   ELSE
       "DB198_eventos_generados_routing_JDT1".evento[#posicion] :=CONCAT(IN1 := '{WARN[RUET]', IN2 := #codigo_string, IN3 := '[ERRO]BBDD[MOTI]FULL',  IN4 := "DB921_DATOS_FECHA_HORA".TIME_STAMP, IN5 := '}');

   END_IF;
END_REGION
END_FUNCTION

FUNCTION "FC887_Obtener_StringDelAtributo_Ulint" : Void   // FC887, LAD
TITLE = "ObtenerStringAtributo" - Convertir a String un Doble Entero
{ S7_Optimized_Access := 'FALSE' }
AUTHOR : TRACKING
NAME : 20130301
VERSION : 3.0
// stored: AutoNumber false, SetENOAutomatically false
   VAR_INPUT
      DB_String : UInt;   // DB donde esta la String
      OffsetIni : UInt;   // Numero de byte de la String donde empieza
      Valor : ULInt;   // Valor a Convertir
   END_VAR
   VAR_OUTPUT
      OffsetFin : UInt;   // Numero de byte de la String donde acaba
   END_VAR
   VAR_TEMP
      PunteroDB : DWord;   // Puntero al DB de la String
      NumDB : Word;   // Num. del DB de la String
      ValorRestante : ULInt;   // Valor a convertir que va quedando
      OffsetActual : UInt;   // Numero de byte que estoy desplazando de la String
      Digito : UInt;   // Valor Convertiodo a Guardar en la String
      Temporal : UInt;
      TEMP_OffsetFin : UInt;
      fin_conversion : Bool;
   END_VAR
BEGIN

REGION Network 1 (SCL): INICIALIZACIONES
   #ValorRestante := #Valor;
   #NumDB := #DB_String;
   #OffsetActual := #TEMP_OffsetFin := #OffsetIni;
   #fin_conversion := false;
END_REGION

NETWORK
TITLE = 
InicioBucle:NOP   0;



REGION Network 3 (SCL): Valor Convertiodo a Guardar en la String

   #Digito := (#ValorRestante MOD 10) + 48;
   // le sumo 48 porque en la tabla ASCII el 0 caracter en decimal es 48 (o 30 en hexadecimal)
END_REGION

NETWORK
TITLE = Conversion
// - Mirar si queda numero a convertir
// - Coger digito
// - Guardarlo en la String
// - Conseguir el Valor Restante


// -----------------------------------------------------------------------------------------------
// Guardarlo en la String

      OPN   DB [#NumDB];

      L     #OffsetIni;  // Miro si es el Primer digito
      L     #TEMP_OffsetFin;
      ==I;
      JC    FinalDesplazar;  // Lo es

// Despalzar en la String para meter un nuevo digito

      L     #TEMP_OffsetFin;  // Inicializo al final
      T     #OffsetActual;  // Primer destino del desplazamiento
InicioDesPlazar:L     #OffsetActual;  // Recogo el dato del Byte Origen
      L     1;
      -I;
      SLD   3;
      T     #PunteroDB;
      L     DBB [#PunteroDB];
      T     #Temporal;

      L     #OffsetActual;  // Dejo el dato del Byte Destino
      SLD   3;
      T     #PunteroDB;
      L     #Temporal;
      T     DBB [#PunteroDB];

      L     #OffsetActual;  // Quito un digito para pasra el Siguiente
      L     1;
      -I;
      T     #OffsetActual;

      L     #OffsetActual;  // Se mira si estan todos desplazados
      L     #OffsetIni;
      ==I;
      JC    FinalDesplazar;  // Si estan todos
      JU    InicioDesPlazar;

// Guardo el ultimo digito guardado - Es el más significativo por ahora

FinalDesplazar:L     #OffsetIni;  // Guardo el digito convertido
      SLD   3;
      T     #PunteroDB;
      L     #Digito;
      T     DBB [#PunteroDB];

      L     #TEMP_OffsetFin;  // Incremento el Puntero Final de la String
      L     1;
      +I;
      T     #TEMP_OffsetFin;



REGION Network 5 (SCL): Valor a convertir que va quedando
   #ValorRestante := #ValorRestante / 10;

   IF #ValorRestante <= 0 THEN
       #fin_conversion := TRUE;
   END_IF;
END_REGION

NETWORK
TITLE = 
      SET;
      A     #fin_conversion;
      JC    Final;

      JU    InicioBucle;


NETWORK
TITLE = Final
// Final de la Funcion
Final:NOP   0;

      L     #TEMP_OffsetFin;  // - Devuelvo el Offset Temporal
      T     #OffsetFin;


END_FUNCTION

FUNCTION_BLOCK "FB101_GIRO_Mesa"   // FB101, LAD
TITLE = FB101
{ S7_Optimized_Access := 'FALSE' }
// FB complementaria a cualquier FB de mesa, solo gestiona el giro.
// stored: AutoNumber false, SetENOAutomatically false
   VAR_INPUT
      Mesa : UInt;   // Mesa de la FB
      Error_Tx : Bool;   // Error en el Tx
      EnTension : Bool;   // Existe Tension en la Mesa
      FalloVar_MG : Bool;   // Señal VAR ok
      MG_EnMovimiento : Bool;   // Señal VAR giro en curso
      PosMG_0 : Bool;   // Detector Posicion 0
      PosMG_90 : Bool;   // Detector Posicion 90
      PosMG_180 : Bool;   // Detector Posicion 180
      PosMG_270 : Bool;   // Detector Posicion 270
      pHsPR : Bool;   // pHs de Protrusion de la Mesa. Nota: No existe >> ON
      Movhabi0_90 : Bool;   // Habilitar zona movimiento entre 0 y 90º
      Movhabi90_180 : Bool;   // Habilitar zona movimiento entre 90 y 180º
      Movhabi180_270 : Bool;   // Habilitar zona movimiento entre 180 y 270º
      Movhabi270_0 : Bool;   // Habilitar zona movimiento entre 270 y 0º
      Mx_VelocidadLenta_In : Bool;   // Forzar velocidad lenta
      OrdPos_0 : Bool;   // Orden ir a Posicion 0
      OrdPos_90 : Bool;   // Orden ir a Posicion 90
      OrdPos_180 : Bool;   // Orden ir a Posicion 180
      OrdPos_270 : Bool;   // Orden ir a Posicion 270
      V_TOut_MG_90º : Int := 15;   // Timeout para un movimiento de 90º
      V_TOut_MG_180º : Int := 30;   // Timeout para un movimiento de 180º
      V_TOut_MG_270º : Int := 45;   // Timeout para un movimiento de 270º
      V_TOut_MG_BusqPos : Int := 15;   // Timeout para busqueda de posición en velo lenta
      V_CNT_PerdidaPos : Int := 5000;   // Perdida de posición
      V_PasoLenta_Mov90 : Int := 800;   // Cambio de velocidad durante un movimiento de 90º
      V_PasoLenta_Mov180 : Int := 1800;   // Cambio de velocidad durante un movimiento de 180º
      V_PasoLenta_Mov270 : Int := 2800;   // Cambio de velocidad durante un movimiento de 270º
      V_CNTSeg_AusPos : Int := 3000;   // Contador de seguridade posicionamiento
   END_VAR
   VAR
      MGiro_EnPos0 : Bool;   // Mesa Giro en posición 0º
      MGiro_EnPos90 : Bool;   // Mesa Giro en posición 90º
      MGiro_EnPos180 : Bool;   // Mesa Giro en posición 180º
      MGiro_EnPos270 : Bool;   // Mesa Giro en posición 270º
      PosOK { ExternalVisible := 'False'} : Bool;
      Orden_AvGiro : Bool;   // Orden de Avance (sentido agujas reloj)
      Orden_RtGiro : Bool;   // Orden de Retroceso (sentido inverso agujas reloj)
      DestinoPos0 : Bool;   // Destino a la posición 0º
      DestinoPos90 : Bool;   // Destino a la posición 90º
      DestinoPos180 : Bool;   // Destino a la posición 180º
      DestinoPos270 : Bool;   // Destino a la posición 270º
      Giro90º : Bool;   // Distancia de giro en grados desde origen hasta destino
      Giro180º : Bool;   // Distancia de giro en grados desde origen hasta destino
      Giro270º : Bool;   // Distancia de giro en grados desde origen hasta destino
      Pos_Desconocida : Bool;
      Pos_Conocida : Bool;
      Destino_Desconocido : Bool;
      Busq_Posicion : Bool;
      Mem_Busq_Posicion : Bool;
      VelocidadLenta { ExternalAccessible := 'False'; ExternalVisible := 'False'; ExternalWritable := 'False'} : Bool;
      MA_Avance_MG : Bool;   // Avance = ir de 0º a 360º
      MA_Retroceso_MG : Bool;   // Retroceso = volver de 360º a 0
      VelocidadRapida_MG : Bool;
      CNT_Paso_Lenta : Int;
      CNTSeg_AusPos { S7_SetPoint := 'True'} : "FB910_CNT_UHS";
      TMP_EnTension { S7_SetPoint := 'True'} : "FB910_CNT_UHS";
      TOut_MG { S7_SetPoint := 'True'} : "FB910_CNT_UHS";
      TOut_MG_BusPos { S7_SetPoint := 'True'} : "FB910_CNT_UHS";
      CNT_PerdidaPos { S7_SetPoint := 'True'} : "FB910_CNT_UHS";
   END_VAR
   VAR_TEMP
      EstadoZona : "EstadoZona";   // Estado de Zona de la Mesa
      EstadoVI : "EstadosMesa";   // Estado del Vehiculo Inteliguente de la Mesa
      ConfigFB : "UDT_ConfigFB";   // Configuracion de la FB de la Mesa
      V_TOut_MG : Int;
      Basura : Bool;
   END_VAR
   VAR_TEMP   // added for the SCL form of the ladder/FBD networks
      _w1 : Bool;
   END_VAR
BEGIN

REGION Network 1: INICIALIZAR - Recoger las Variables de Estado de la Mesa
   // Se recoge - Estado_CBx
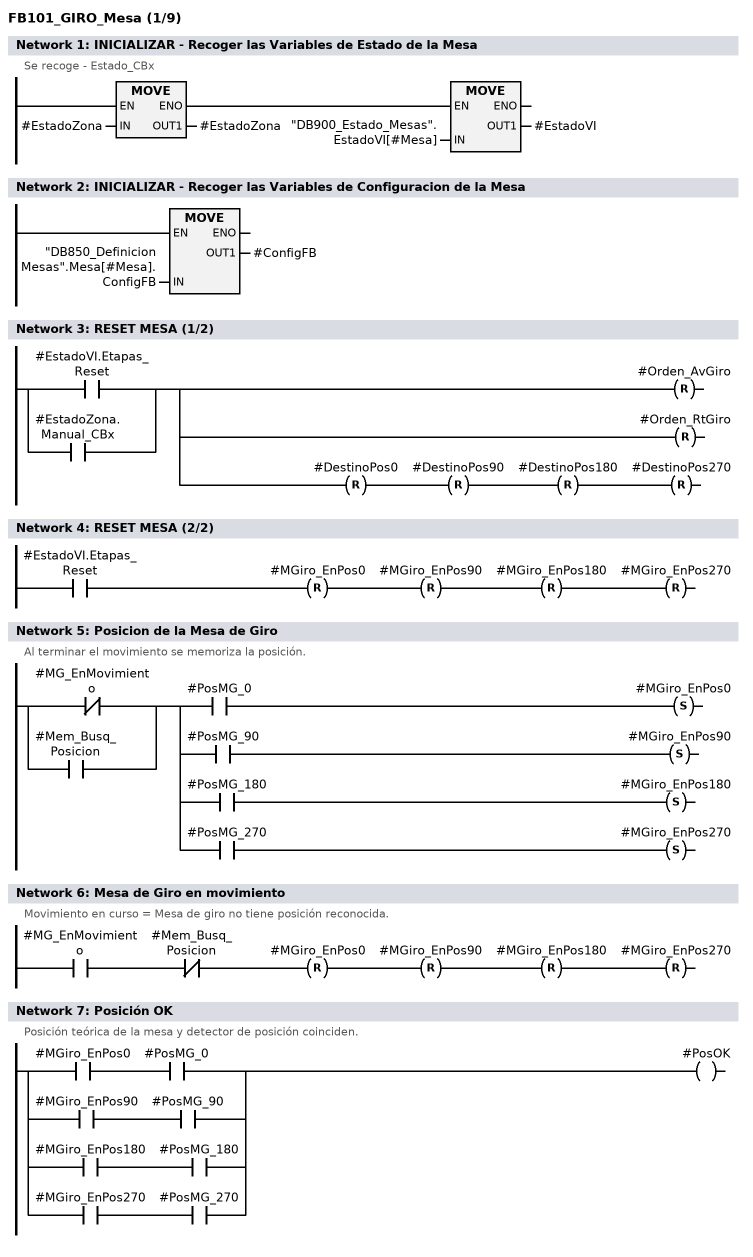
   RUNG wire#powerrail
      Move(in := #EstadoZona, out1 => #EstadoZona)
      Move(in := "DB900_Estado_Mesas".EstadoVI[#Mesa], out1 => #EstadoVI)
   END_RUNG
   // the same network as SCL:
   #EstadoZona := #EstadoZona;
   #EstadoVI := "DB900_Estado_Mesas".EstadoVI[#Mesa];
END_REGION

REGION Network 2: INICIALIZAR - Recoger las Variables de Configuracion de la Mesa
   RUNG wire#powerrail
      Move(in := "DB850_DefinicionMesas".Mesa[#Mesa].ConfigFB, out1 => #ConfigFB)
   END_RUNG
   // the same network as SCL:
   #ConfigFB := "DB850_DefinicionMesas".Mesa[#Mesa].ConfigFB;
END_REGION

REGION Network 3: RESET MESA (1/2)
   RUNG wire#powerrail
      Contact( #EstadoVI.Etapas_Reset )
      wire#w1
      R_Coil( #Orden_AvGiro )
   END_RUNG
   RUNG wire#powerrail
      Contact( #EstadoZona.Manual_CBx )
   END_RUNG wire#w1
   RUNG wire#w1
      R_Coil( #Orden_RtGiro )
   END_RUNG
   RUNG wire#w1
      R_Coil( #DestinoPos0 )
      R_Coil( #DestinoPos90 )
      R_Coil( #DestinoPos180 )
      R_Coil( #DestinoPos270 )
   END_RUNG
   // the same network as SCL:
   IF #EstadoVI.Etapas_Reset OR #EstadoZona.Manual_CBx THEN
       #Orden_AvGiro := FALSE;
       #Orden_RtGiro := FALSE;
       #DestinoPos0 := FALSE;
       #DestinoPos90 := FALSE;
       #DestinoPos180 := FALSE;
       #DestinoPos270 := FALSE;
   END_IF;
END_REGION

REGION Network 4: RESET MESA (2/2)
   RUNG wire#powerrail
      Contact( #EstadoVI.Etapas_Reset )
      R_Coil( #MGiro_EnPos0 )
      R_Coil( #MGiro_EnPos90 )
      R_Coil( #MGiro_EnPos180 )
      R_Coil( #MGiro_EnPos270 )
   END_RUNG
   // the same network as SCL:
   IF #EstadoVI.Etapas_Reset THEN
       #MGiro_EnPos0 := FALSE;
       #MGiro_EnPos90 := FALSE;
       #MGiro_EnPos180 := FALSE;
       #MGiro_EnPos270 := FALSE;
   END_IF;
END_REGION

REGION Network 5: Posicion de la Mesa de Giro
   // Al terminar el movimiento se memoriza la posición.
   RUNG wire#powerrail
      I_Contact( #MG_EnMovimiento )
      wire#w1
      Contact( #PosMG_0 )
      S_Coil( #MGiro_EnPos0 )
   END_RUNG
   RUNG wire#powerrail
      Contact( #Mem_Busq_Posicion )
   END_RUNG wire#w1
   RUNG wire#w1
      Contact( #PosMG_90 )
      S_Coil( #MGiro_EnPos90 )
   END_RUNG
   RUNG wire#w1
      Contact( #PosMG_180 )
      S_Coil( #MGiro_EnPos180 )
   END_RUNG
   RUNG wire#w1
      Contact( #PosMG_270 )
      S_Coil( #MGiro_EnPos270 )
   END_RUNG
   // the same network as SCL:
   #_w1 := NOT #MG_EnMovimiento OR #Mem_Busq_Posicion;
   IF #_w1 AND #PosMG_0 THEN #MGiro_EnPos0 := TRUE; END_IF;
   IF #_w1 AND #PosMG_90 THEN #MGiro_EnPos90 := TRUE; END_IF;
   IF #_w1 AND #PosMG_180 THEN #MGiro_EnPos180 := TRUE; END_IF;
   IF #_w1 AND #PosMG_270 THEN #MGiro_EnPos270 := TRUE; END_IF;
END_REGION

REGION Network 6: Mesa de Giro en movimiento
   // Movimiento en curso = Mesa de giro no tiene posición reconocida.
   RUNG wire#powerrail
      Contact( #MG_EnMovimiento )
      I_Contact( #Mem_Busq_Posicion )
      R_Coil( #MGiro_EnPos0 )
      R_Coil( #MGiro_EnPos90 )
      R_Coil( #MGiro_EnPos180 )
      R_Coil( #MGiro_EnPos270 )
   END_RUNG
   // the same network as SCL:
   IF #MG_EnMovimiento AND NOT #Mem_Busq_Posicion THEN
       #MGiro_EnPos0 := FALSE;
       #MGiro_EnPos90 := FALSE;
       #MGiro_EnPos180 := FALSE;
       #MGiro_EnPos270 := FALSE;
   END_IF;
END_REGION

REGION Network 7: Posición OK
   // Posición teórica de la mesa y detector de posición coinciden.
   RUNG wire#powerrail
      Contact( #MGiro_EnPos0 )
      Contact( #PosMG_0 )
      wire#w1
      Coil( #PosOK )
   END_RUNG
   RUNG wire#powerrail
      Contact( #MGiro_EnPos90 )
      Contact( #PosMG_90 )
   END_RUNG wire#w1
   RUNG wire#powerrail
      Contact( #MGiro_EnPos180 )
      Contact( #PosMG_180 )
   END_RUNG wire#w1
   RUNG wire#powerrail
      Contact( #MGiro_EnPos270 )
      Contact( #PosMG_270 )
   END_RUNG wire#w1
   // the same network as SCL:
   #PosOK := (#MGiro_EnPos0 AND #PosMG_0) OR (#MGiro_EnPos90 AND #PosMG_90) OR (#MGiro_EnPos180 AND #PosMG_180) OR (#MGiro_EnPos270 AND #PosMG_270);
END_REGION

REGION Network 8: Destino Desconocido // Posicion desconocida // Posicion Conocida
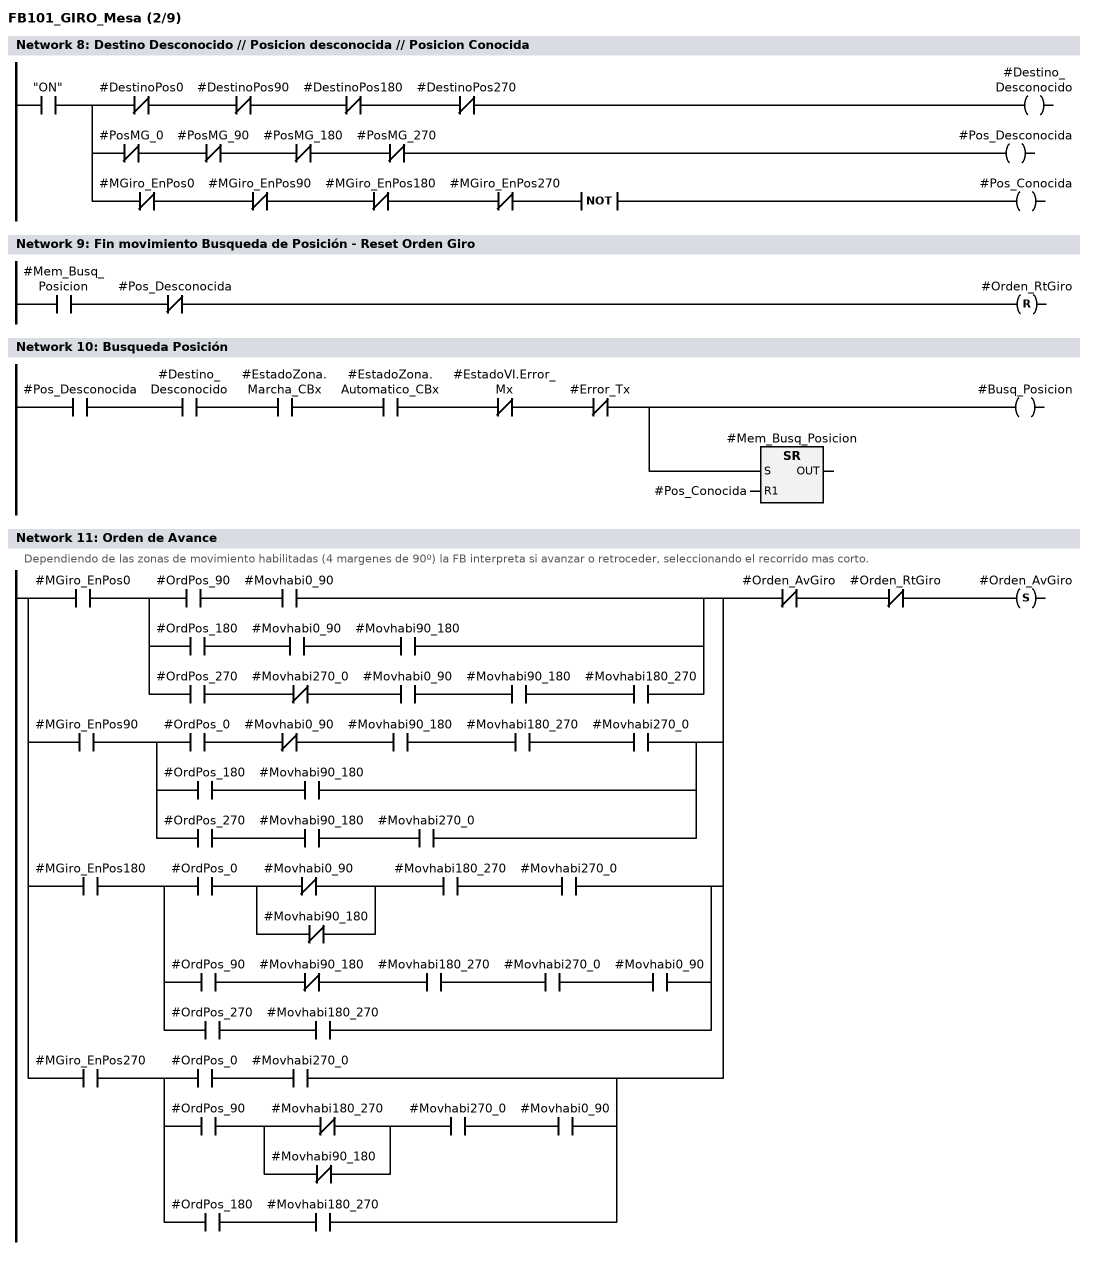
   RUNG wire#powerrail
      Contact( "ON" )
      wire#w1
      I_Contact( #DestinoPos0 )
      I_Contact( #DestinoPos90 )
      I_Contact( #DestinoPos180 )
      I_Contact( #DestinoPos270 )
      Coil( #Destino_Desconocido )
   END_RUNG
   RUNG wire#w1
      I_Contact( #PosMG_0 )
      I_Contact( #PosMG_90 )
      I_Contact( #PosMG_180 )
      I_Contact( #PosMG_270 )
      Coil( #Pos_Desconocida )
   END_RUNG
   RUNG wire#w1
      I_Contact( #MGiro_EnPos0 )
      I_Contact( #MGiro_EnPos90 )
      I_Contact( #MGiro_EnPos180 )
      I_Contact( #MGiro_EnPos270 )
      Not()
      Coil( #Pos_Conocida )
   END_RUNG
   // the same network as SCL:
   #Destino_Desconocido := "ON" AND NOT #DestinoPos0 AND NOT #DestinoPos90 AND NOT #DestinoPos180 AND NOT #DestinoPos270;
   #Pos_Desconocida := "ON" AND NOT #PosMG_0 AND NOT #PosMG_90 AND NOT #PosMG_180 AND NOT #PosMG_270;
   #Pos_Conocida := NOT ("ON" AND NOT #MGiro_EnPos0 AND NOT #MGiro_EnPos90 AND NOT #MGiro_EnPos180 AND NOT #MGiro_EnPos270);
END_REGION

REGION Network 9: Fin movimiento Busqueda de Posición - Reset Orden Giro
   RUNG wire#powerrail
      Contact( #Mem_Busq_Posicion )
      I_Contact( #Pos_Desconocida )
      R_Coil( #Orden_RtGiro )
   END_RUNG
   // the same network as SCL:
   IF #Mem_Busq_Posicion AND NOT #Pos_Desconocida THEN #Orden_RtGiro := FALSE; END_IF;
END_REGION

REGION Network 10: Busqueda Posición
   RUNG wire#powerrail
      Contact( #Pos_Desconocida )
      Contact( #Destino_Desconocido )
      Contact( #EstadoZona.Marcha_CBx )
      Contact( #EstadoZona.Automatico_CBx )
      I_Contact( #EstadoVI.Error_Mx )
      I_Contact( #Error_Tx )
      wire#w1
      Coil( #Busq_Posicion )
   END_RUNG
   RUNG wire#w1
      S_SR(operand := #Mem_Busq_Posicion, r1 := #Pos_Conocida)
   END_RUNG
   // the same network as SCL:
   #Busq_Posicion := #Pos_Desconocida AND #Destino_Desconocido AND #EstadoZona.Marcha_CBx AND #EstadoZona.Automatico_CBx AND NOT #EstadoVI.Error_Mx AND NOT #Error_Tx;
   IF #Busq_Posicion THEN
       #Mem_Busq_Posicion := TRUE;   // SR flip-flop
   END_IF;
   IF #Pos_Conocida THEN #Mem_Busq_Posicion := FALSE; END_IF;
END_REGION

REGION Network 11: Orden de Avance
   // Dependiendo de las zonas de movimiento habilitadas (4 margenes de 90º) la FB interpreta si avanzar o retroceder, seleccionando el recorrido mas corto.
   RUNG wire#powerrail
      Contact( #MGiro_EnPos0 )
      wire#w1
      Contact( #OrdPos_90 )
      Contact( #Movhabi0_90 )
      wire#w2
      I_Contact( #Orden_AvGiro )
      I_Contact( #Orden_RtGiro )
      S_Coil( #Orden_AvGiro )
   END_RUNG
   RUNG wire#w1
      Contact( #OrdPos_180 )
      Contact( #Movhabi0_90 )
      Contact( #Movhabi90_180 )
   END_RUNG wire#w2
   RUNG wire#w1
      Contact( #OrdPos_270 )
      I_Contact( #Movhabi270_0 )
      Contact( #Movhabi0_90 )
      Contact( #Movhabi90_180 )
      Contact( #Movhabi180_270 )
   END_RUNG wire#w2
   RUNG wire#powerrail
      Contact( #MGiro_EnPos90 )
      wire#w3
      Contact( #OrdPos_0 )
      I_Contact( #Movhabi0_90 )
      Contact( #Movhabi90_180 )
      Contact( #Movhabi180_270 )
      Contact( #Movhabi270_0 )
   END_RUNG wire#w2
   RUNG wire#w3
      Contact( #OrdPos_180 )
      Contact( #Movhabi90_180 )
   END_RUNG wire#w2
   RUNG wire#w3
      Contact( #OrdPos_270 )
      Contact( #Movhabi90_180 )
      Contact( #Movhabi270_0 )
   END_RUNG wire#w2
   RUNG wire#powerrail
      Contact( #MGiro_EnPos180 )
      wire#w4
      Contact( #OrdPos_0 )
      wire#w5
      I_Contact( #Movhabi0_90 )
      wire#w6
      Contact( #Movhabi180_270 )
      Contact( #Movhabi270_0 )
   END_RUNG wire#w2
   RUNG wire#w5
      I_Contact( #Movhabi90_180 )
   END_RUNG wire#w6
   RUNG wire#w4
      Contact( #OrdPos_90 )
      I_Contact( #Movhabi90_180 )
      Contact( #Movhabi180_270 )
      Contact( #Movhabi270_0 )
      Contact( #Movhabi0_90 )
   END_RUNG wire#w2
   RUNG wire#w4
      Contact( #OrdPos_270 )
      Contact( #Movhabi180_270 )
   END_RUNG wire#w2
   RUNG wire#powerrail
      Contact( #MGiro_EnPos270 )
      wire#w7
      Contact( #OrdPos_0 )
      Contact( #Movhabi270_0 )
   END_RUNG wire#w2
   RUNG wire#w7
      Contact( #OrdPos_90 )
      wire#w8
      I_Contact( #Movhabi180_270 )
      wire#w9
      Contact( #Movhabi270_0 )
      Contact( #Movhabi0_90 )
   END_RUNG wire#w2
   RUNG wire#w8
      I_Contact( #Movhabi90_180 )
   END_RUNG wire#w9
   RUNG wire#w7
      Contact( #OrdPos_180 )
      Contact( #Movhabi180_270 )
   END_RUNG wire#w2
   // the same network as SCL:
   IF ((#MGiro_EnPos0 AND ((#OrdPos_90 AND #Movhabi0_90) OR (#OrdPos_180 AND #Movhabi0_90 AND #Movhabi90_180) OR (#OrdPos_270 AND NOT #Movhabi270_0 AND #Movhabi0_90 AND #Movhabi90_180 AND #Movhabi180_270))) OR (#MGiro_EnPos90 AND ((#OrdPos_0 AND NOT #Movhabi0_90 AND #Movhabi90_180 AND #Movhabi180_270 AND #Movhabi270_0) OR (#OrdPos_180 AND #Movhabi90_180) OR (#OrdPos_270 AND #Movhabi90_180 AND #Movhabi270_0))) OR (#MGiro_EnPos180 AND ((#OrdPos_0 AND (NOT #Movhabi0_90 OR NOT #Movhabi90_180) AND #Movhabi180_270 AND #Movhabi270_0) OR (#OrdPos_90 AND NOT #Movhabi90_180 AND #Movhabi180_270 AND #Movhabi270_0 AND #Movhabi0_90) OR (#OrdPos_270 AND #Movhabi180_270))) OR (#MGiro_EnPos270 AND ((#OrdPos_0 AND #Movhabi270_0) OR (#OrdPos_90 AND (NOT #Movhabi180_270 OR NOT #Movhabi90_180) AND #Movhabi270_0 AND #Movhabi0_90) OR (#OrdPos_180 AND #Movhabi180_270)))) AND NOT #Orden_AvGiro AND NOT #Orden_RtGiro THEN
       #Orden_AvGiro := TRUE;
   END_IF;
END_REGION

REGION Network 12: Orden de Retroceso
   // Dependiendo de las zonas de movimiento habilitadas (4 margenes de 90º) la FB interpreta si avanzar o retroceder, seleccionando el recorrido mas corto.
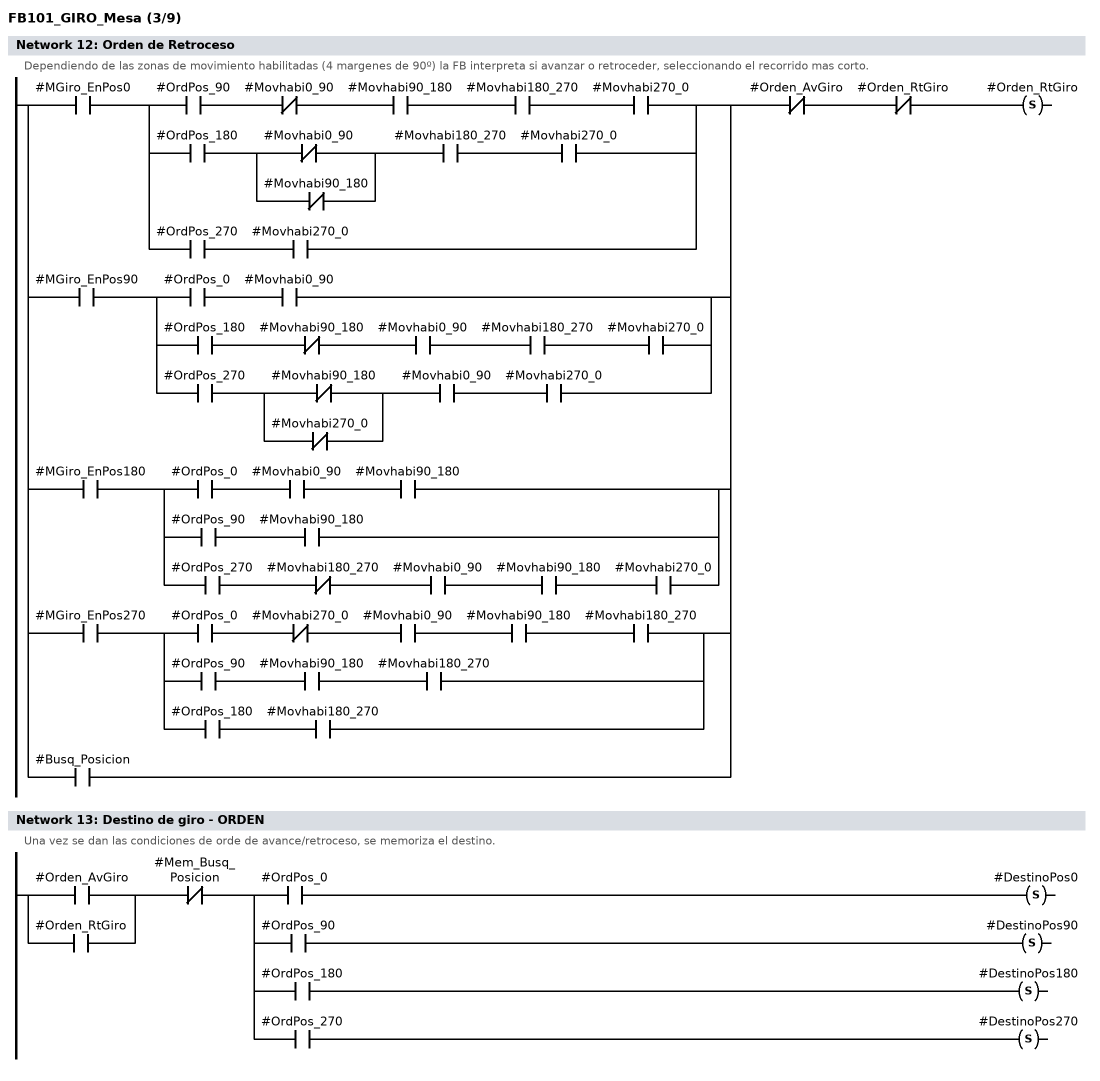
   RUNG wire#powerrail
      Contact( #MGiro_EnPos0 )
      wire#w1
      Contact( #OrdPos_90 )
      I_Contact( #Movhabi0_90 )
      Contact( #Movhabi90_180 )
      Contact( #Movhabi180_270 )
      Contact( #Movhabi270_0 )
      wire#w2
      I_Contact( #Orden_AvGiro )
      I_Contact( #Orden_RtGiro )
      S_Coil( #Orden_RtGiro )
   END_RUNG
   RUNG wire#w1
      Contact( #OrdPos_180 )
      wire#w3
      I_Contact( #Movhabi0_90 )
      wire#w4
      Contact( #Movhabi180_270 )
      Contact( #Movhabi270_0 )
   END_RUNG wire#w2
   RUNG wire#w3
      I_Contact( #Movhabi90_180 )
   END_RUNG wire#w4
   RUNG wire#w1
      Contact( #OrdPos_270 )
      Contact( #Movhabi270_0 )
   END_RUNG wire#w2
   RUNG wire#powerrail
      Contact( #MGiro_EnPos90 )
      wire#w5
      Contact( #OrdPos_0 )
      Contact( #Movhabi0_90 )
   END_RUNG wire#w2
   RUNG wire#w5
      Contact( #OrdPos_180 )
      I_Contact( #Movhabi90_180 )
      Contact( #Movhabi0_90 )
      Contact( #Movhabi180_270 )
      Contact( #Movhabi270_0 )
   END_RUNG wire#w2
   RUNG wire#w5
      Contact( #OrdPos_270 )
      wire#w6
      I_Contact( #Movhabi90_180 )
      wire#w7
      Contact( #Movhabi0_90 )
      Contact( #Movhabi270_0 )
   END_RUNG wire#w2
   RUNG wire#w6
      I_Contact( #Movhabi270_0 )
   END_RUNG wire#w7
   RUNG wire#powerrail
      Contact( #MGiro_EnPos180 )
      wire#w8
      Contact( #OrdPos_0 )
      Contact( #Movhabi0_90 )
      Contact( #Movhabi90_180 )
   END_RUNG wire#w2
   RUNG wire#w8
      Contact( #OrdPos_90 )
      Contact( #Movhabi90_180 )
   END_RUNG wire#w2
   RUNG wire#w8
      Contact( #OrdPos_270 )
      I_Contact( #Movhabi180_270 )
      Contact( #Movhabi0_90 )
      Contact( #Movhabi90_180 )
      Contact( #Movhabi270_0 )
   END_RUNG wire#w2
   RUNG wire#powerrail
      Contact( #MGiro_EnPos270 )
      wire#w9
      Contact( #OrdPos_0 )
      I_Contact( #Movhabi270_0 )
      Contact( #Movhabi0_90 )
      Contact( #Movhabi90_180 )
      Contact( #Movhabi180_270 )
   END_RUNG wire#w2
   RUNG wire#w9
      Contact( #OrdPos_90 )
      Contact( #Movhabi90_180 )
      Contact( #Movhabi180_270 )
   END_RUNG wire#w2
   RUNG wire#w9
      Contact( #OrdPos_180 )
      Contact( #Movhabi180_270 )
   END_RUNG wire#w2
   RUNG wire#powerrail
      Contact( #Busq_Posicion )
   END_RUNG wire#w2
   // the same network as SCL:
   IF ((#MGiro_EnPos0 AND ((#OrdPos_90 AND NOT #Movhabi0_90 AND #Movhabi90_180 AND #Movhabi180_270 AND #Movhabi270_0) OR (#OrdPos_180 AND (NOT #Movhabi0_90 OR NOT #Movhabi90_180) AND #Movhabi180_270 AND #Movhabi270_0) OR (#OrdPos_270 AND #Movhabi270_0))) OR (#MGiro_EnPos90 AND ((#OrdPos_0 AND #Movhabi0_90) OR (#OrdPos_180 AND NOT #Movhabi90_180 AND #Movhabi0_90 AND #Movhabi180_270 AND #Movhabi270_0) OR (#OrdPos_270 AND (NOT #Movhabi90_180 OR NOT #Movhabi270_0) AND #Movhabi0_90 AND #Movhabi270_0))) OR (#MGiro_EnPos180 AND ((#OrdPos_0 AND #Movhabi0_90 AND #Movhabi90_180) OR (#OrdPos_90 AND #Movhabi90_180) OR (#OrdPos_270 AND NOT #Movhabi180_270 AND #Movhabi0_90 AND #Movhabi90_180 AND #Movhabi270_0))) OR (#MGiro_EnPos270 AND ((#OrdPos_0 AND NOT #Movhabi270_0 AND #Movhabi0_90 AND #Movhabi90_180 AND #Movhabi180_270) OR (#OrdPos_90 AND #Movhabi90_180 AND #Movhabi180_270) OR (#OrdPos_180 AND #Movhabi180_270))) OR #Busq_Posicion) AND NOT #Orden_AvGiro AND NOT #Orden_RtGiro THEN
       #Orden_RtGiro := TRUE;
   END_IF;
END_REGION

REGION Network 13: Destino de giro - ORDEN
   // Una vez se dan las condiciones de orde de avance/retroceso, se memoriza el destino.
   RUNG wire#powerrail
      Contact( #Orden_AvGiro )
      wire#w1
      I_Contact( #Mem_Busq_Posicion )
      wire#w2
      Contact( #OrdPos_0 )
      S_Coil( #DestinoPos0 )
   END_RUNG
   RUNG wire#powerrail
      Contact( #Orden_RtGiro )
   END_RUNG wire#w1
   RUNG wire#w2
      Contact( #OrdPos_90 )
      S_Coil( #DestinoPos90 )
   END_RUNG
   RUNG wire#w2
      Contact( #OrdPos_180 )
      S_Coil( #DestinoPos180 )
   END_RUNG
   RUNG wire#w2
      Contact( #OrdPos_270 )
      S_Coil( #DestinoPos270 )
   END_RUNG
   // the same network as SCL:
   #_w1 := (#Orden_AvGiro OR #Orden_RtGiro) AND NOT #Mem_Busq_Posicion;
   IF #_w1 AND #OrdPos_0 THEN #DestinoPos0 := TRUE; END_IF;
   IF #_w1 AND #OrdPos_90 THEN #DestinoPos90 := TRUE; END_IF;
   IF #_w1 AND #OrdPos_180 THEN #DestinoPos180 := TRUE; END_IF;
   IF #_w1 AND #OrdPos_270 THEN #DestinoPos270 := TRUE; END_IF;
END_REGION

REGION Network 14: Destino de giro - FIN
   // Al llegar a posición el destino se borra.
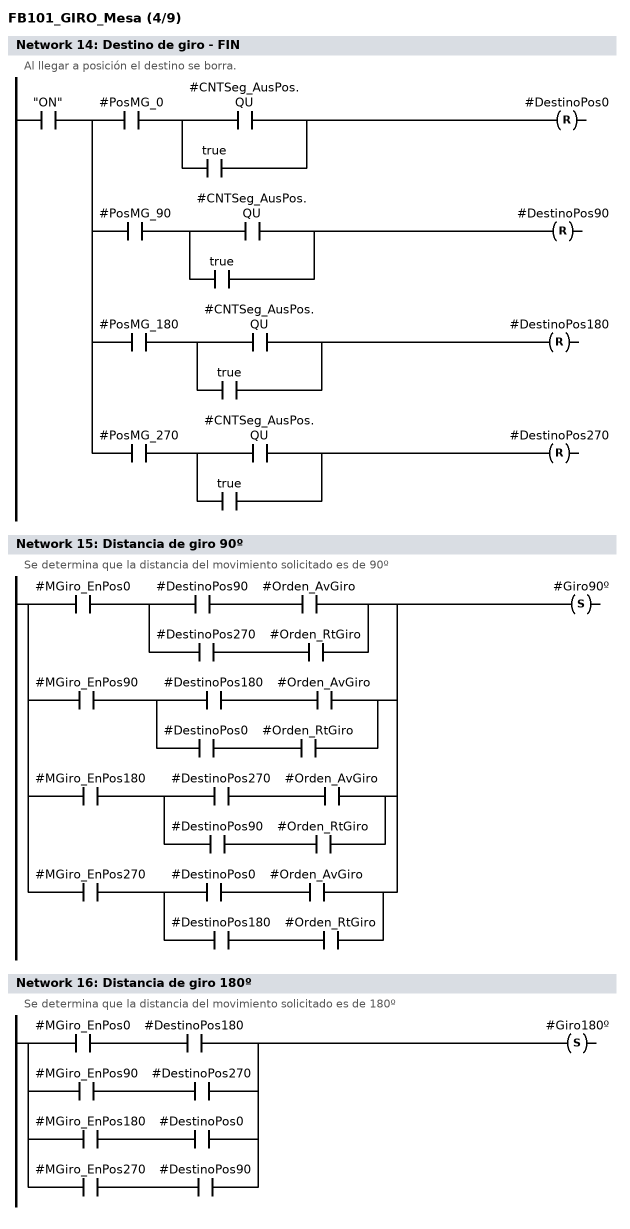
   RUNG wire#powerrail
      Contact( "ON" )
      wire#w1
      Contact( #PosMG_0 )
      wire#w2
      Contact( #CNTSeg_AusPos.QU )
      wire#w3
      R_Coil( #DestinoPos0 )
   END_RUNG
   RUNG wire#w2
      Contact( true )
   END_RUNG wire#w3
   RUNG wire#w1
      Contact( #PosMG_90 )
      wire#w4
      Contact( #CNTSeg_AusPos.QU )
      wire#w5
      R_Coil( #DestinoPos90 )
   END_RUNG
   RUNG wire#w4
      Contact( true )
   END_RUNG wire#w5
   RUNG wire#w1
      Contact( #PosMG_180 )
      wire#w6
      Contact( #CNTSeg_AusPos.QU )
      wire#w7
      R_Coil( #DestinoPos180 )
   END_RUNG
   RUNG wire#w6
      Contact( true )
   END_RUNG wire#w7
   RUNG wire#w1
      Contact( #PosMG_270 )
      wire#w8
      Contact( #CNTSeg_AusPos.QU )
      wire#w9
      R_Coil( #DestinoPos270 )
   END_RUNG
   RUNG wire#w8
      Contact( true )
   END_RUNG wire#w9
   // the same network as SCL:
   IF "ON" AND #PosMG_0 AND (#CNTSeg_AusPos.QU OR true) THEN #DestinoPos0 := FALSE; END_IF;
   IF "ON" AND #PosMG_90 AND (#CNTSeg_AusPos.QU OR true) THEN #DestinoPos90 := FALSE; END_IF;
   IF "ON" AND #PosMG_180 AND (#CNTSeg_AusPos.QU OR true) THEN #DestinoPos180 := FALSE; END_IF;
   IF "ON" AND #PosMG_270 AND (#CNTSeg_AusPos.QU OR true) THEN #DestinoPos270 := FALSE; END_IF;
END_REGION

REGION Network 15: Distancia de giro 90º
   // Se determina que la distancia del movimiento solicitado es de 90º
   RUNG wire#powerrail
      Contact( #MGiro_EnPos0 )
      wire#w1
      Contact( #DestinoPos90 )
      Contact( #Orden_AvGiro )
      wire#w2
      S_Coil( #Giro90º )
   END_RUNG
   RUNG wire#w1
      Contact( #DestinoPos270 )
      Contact( #Orden_RtGiro )
   END_RUNG wire#w2
   RUNG wire#powerrail
      Contact( #MGiro_EnPos90 )
      wire#w3
      Contact( #DestinoPos180 )
      Contact( #Orden_AvGiro )
   END_RUNG wire#w2
   RUNG wire#w3
      Contact( #DestinoPos0 )
      Contact( #Orden_RtGiro )
   END_RUNG wire#w2
   RUNG wire#powerrail
      Contact( #MGiro_EnPos180 )
      wire#w4
      Contact( #DestinoPos270 )
      Contact( #Orden_AvGiro )
   END_RUNG wire#w2
   RUNG wire#w4
      Contact( #DestinoPos90 )
      Contact( #Orden_RtGiro )
   END_RUNG wire#w2
   RUNG wire#powerrail
      Contact( #MGiro_EnPos270 )
      wire#w5
      Contact( #DestinoPos0 )
      Contact( #Orden_AvGiro )
   END_RUNG wire#w2
   RUNG wire#w5
      Contact( #DestinoPos180 )
      Contact( #Orden_RtGiro )
   END_RUNG wire#w2
   // the same network as SCL:
   IF (#MGiro_EnPos0 AND ((#DestinoPos90 AND #Orden_AvGiro) OR (#DestinoPos270 AND #Orden_RtGiro))) OR (#MGiro_EnPos90 AND ((#DestinoPos180 AND #Orden_AvGiro) OR (#DestinoPos0 AND #Orden_RtGiro))) OR (#MGiro_EnPos180 AND ((#DestinoPos270 AND #Orden_AvGiro) OR (#DestinoPos90 AND #Orden_RtGiro))) OR (#MGiro_EnPos270 AND ((#DestinoPos0 AND #Orden_AvGiro) OR (#DestinoPos180 AND #Orden_RtGiro))) THEN
       #Giro90º := TRUE;
   END_IF;
END_REGION

REGION Network 16: Distancia de giro 180º
   // Se determina que la distancia del movimiento solicitado es de 180º
   RUNG wire#powerrail
      Contact( #MGiro_EnPos0 )
      Contact( #DestinoPos180 )
      wire#w1
      S_Coil( #Giro180º )
   END_RUNG
   RUNG wire#powerrail
      Contact( #MGiro_EnPos90 )
      Contact( #DestinoPos270 )
   END_RUNG wire#w1
   RUNG wire#powerrail
      Contact( #MGiro_EnPos180 )
      Contact( #DestinoPos0 )
   END_RUNG wire#w1
   RUNG wire#powerrail
      Contact( #MGiro_EnPos270 )
      Contact( #DestinoPos90 )
   END_RUNG wire#w1
   // the same network as SCL:
   IF (#MGiro_EnPos0 AND #DestinoPos180) OR (#MGiro_EnPos90 AND #DestinoPos270) OR (#MGiro_EnPos180 AND #DestinoPos0) OR (#MGiro_EnPos270 AND #DestinoPos90) THEN
       #Giro180º := TRUE;
   END_IF;
END_REGION

REGION Network 17: Distancia de giro 270º
   // Se determina que la distancia del movimiento solicitado es de 270º
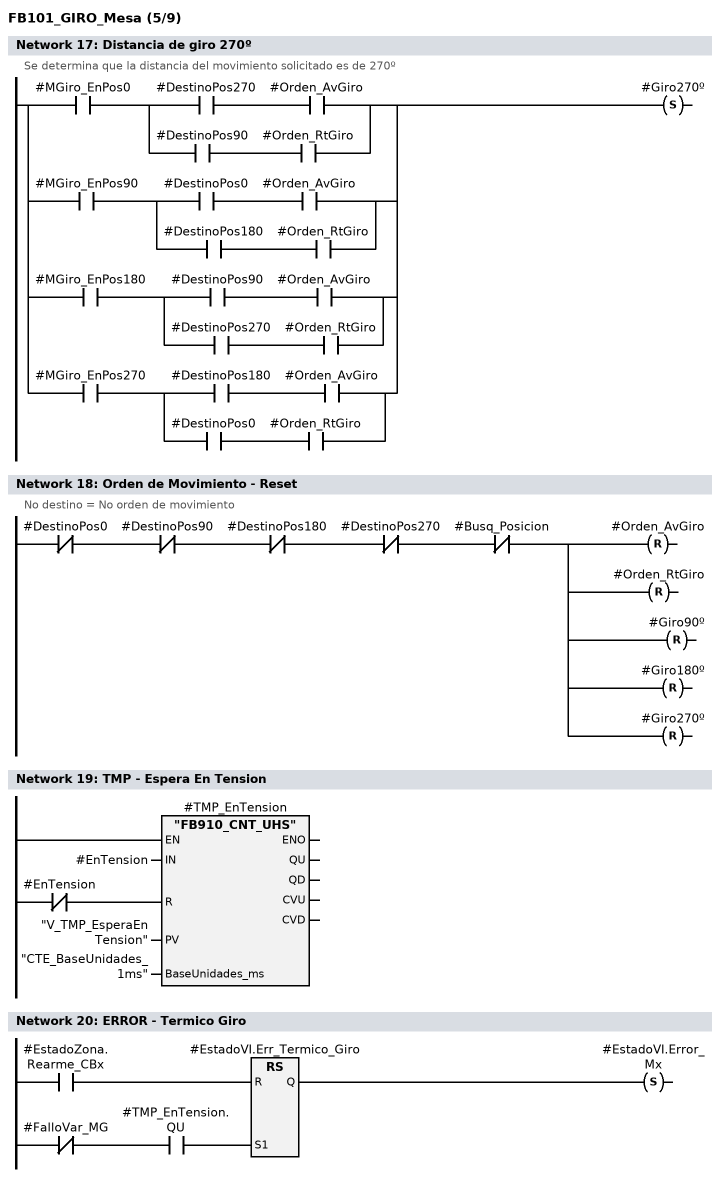
   RUNG wire#powerrail
      Contact( #MGiro_EnPos0 )
      wire#w1
      Contact( #DestinoPos270 )
      Contact( #Orden_AvGiro )
      wire#w2
      S_Coil( #Giro270º )
   END_RUNG
   RUNG wire#w1
      Contact( #DestinoPos90 )
      Contact( #Orden_RtGiro )
   END_RUNG wire#w2
   RUNG wire#powerrail
      Contact( #MGiro_EnPos90 )
      wire#w3
      Contact( #DestinoPos0 )
      Contact( #Orden_AvGiro )
   END_RUNG wire#w2
   RUNG wire#w3
      Contact( #DestinoPos180 )
      Contact( #Orden_RtGiro )
   END_RUNG wire#w2
   RUNG wire#powerrail
      Contact( #MGiro_EnPos180 )
      wire#w4
      Contact( #DestinoPos90 )
      Contact( #Orden_AvGiro )
   END_RUNG wire#w2
   RUNG wire#w4
      Contact( #DestinoPos270 )
      Contact( #Orden_RtGiro )
   END_RUNG wire#w2
   RUNG wire#powerrail
      Contact( #MGiro_EnPos270 )
      wire#w5
      Contact( #DestinoPos180 )
      Contact( #Orden_AvGiro )
   END_RUNG wire#w2
   RUNG wire#w5
      Contact( #DestinoPos0 )
      Contact( #Orden_RtGiro )
   END_RUNG wire#w2
   // the same network as SCL:
   IF (#MGiro_EnPos0 AND ((#DestinoPos270 AND #Orden_AvGiro) OR (#DestinoPos90 AND #Orden_RtGiro))) OR (#MGiro_EnPos90 AND ((#DestinoPos0 AND #Orden_AvGiro) OR (#DestinoPos180 AND #Orden_RtGiro))) OR (#MGiro_EnPos180 AND ((#DestinoPos90 AND #Orden_AvGiro) OR (#DestinoPos270 AND #Orden_RtGiro))) OR (#MGiro_EnPos270 AND ((#DestinoPos180 AND #Orden_AvGiro) OR (#DestinoPos0 AND #Orden_RtGiro))) THEN
       #Giro270º := TRUE;
   END_IF;
END_REGION

REGION Network 18: Orden de Movimiento - Reset
   // No destino = No orden de movimiento
   RUNG wire#powerrail
      I_Contact( #DestinoPos0 )
      I_Contact( #DestinoPos90 )
      I_Contact( #DestinoPos180 )
      I_Contact( #DestinoPos270 )
      I_Contact( #Busq_Posicion )
      wire#w1
      R_Coil( #Orden_AvGiro )
   END_RUNG
   RUNG wire#w1
      R_Coil( #Orden_RtGiro )
   END_RUNG
   RUNG wire#w1
      R_Coil( #Giro90º )
   END_RUNG
   RUNG wire#w1
      R_Coil( #Giro180º )
   END_RUNG
   RUNG wire#w1
      R_Coil( #Giro270º )
   END_RUNG
   // the same network as SCL:
   IF NOT #DestinoPos0 AND NOT #DestinoPos90 AND NOT #DestinoPos180 AND NOT #DestinoPos270 AND NOT #Busq_Posicion THEN
       #Orden_AvGiro := FALSE;
       #Orden_RtGiro := FALSE;
       #Giro90º := FALSE;
       #Giro180º := FALSE;
       #Giro270º := FALSE;
   END_IF;
END_REGION

REGION Network 19: TMP - Espera En Tension
   RUNG wire#powerrail
      #TMP_EnTension(R := wire#w1, IN := #EnTension, PV := "V_TMP_EsperaEnTension", BaseUnidades_ms := "CTE_BaseUnidades_1ms", QU =>, QD =>, CVU =>, CVD =>)
   END_RUNG
   RUNG wire#powerrail
      I_Contact( #EnTension )
   END_RUNG wire#w1
   // the same network as SCL:
   #TMP_EnTension(IN := #EnTension,   // "FB910_CNT_UHS"
                  R := NOT #EnTension,
                  PV := "V_TMP_EsperaEnTension",
                  BaseUnidades_ms := "CTE_BaseUnidades_1ms");
END_REGION

REGION Network 20: ERROR - Termico Giro
   RUNG wire#powerrail
      Contact( #EstadoZona.Rearme_CBx )
      S_RS(operand := #EstadoVI.Err_Termico_Giro, s1 := wire#w1)
      S_Coil( #EstadoVI.Error_Mx )
   END_RUNG
   RUNG wire#powerrail
      I_Contact( #FalloVar_MG )
      Contact( #TMP_EnTension.QU )
   END_RUNG wire#w1
   // the same network as SCL:
   IF #EstadoZona.Rearme_CBx THEN
       #EstadoVI.Err_Termico_Giro := FALSE;   // RS flip-flop
   END_IF;
   IF NOT #FalloVar_MG AND #TMP_EnTension.QU THEN #EstadoVI.Err_Termico_Giro := TRUE; END_IF;
   IF #EstadoVI.Err_Termico_Giro THEN #EstadoVI.Error_Mx := TRUE; END_IF;
END_REGION

REGION Network 21: ERROR - Protusion
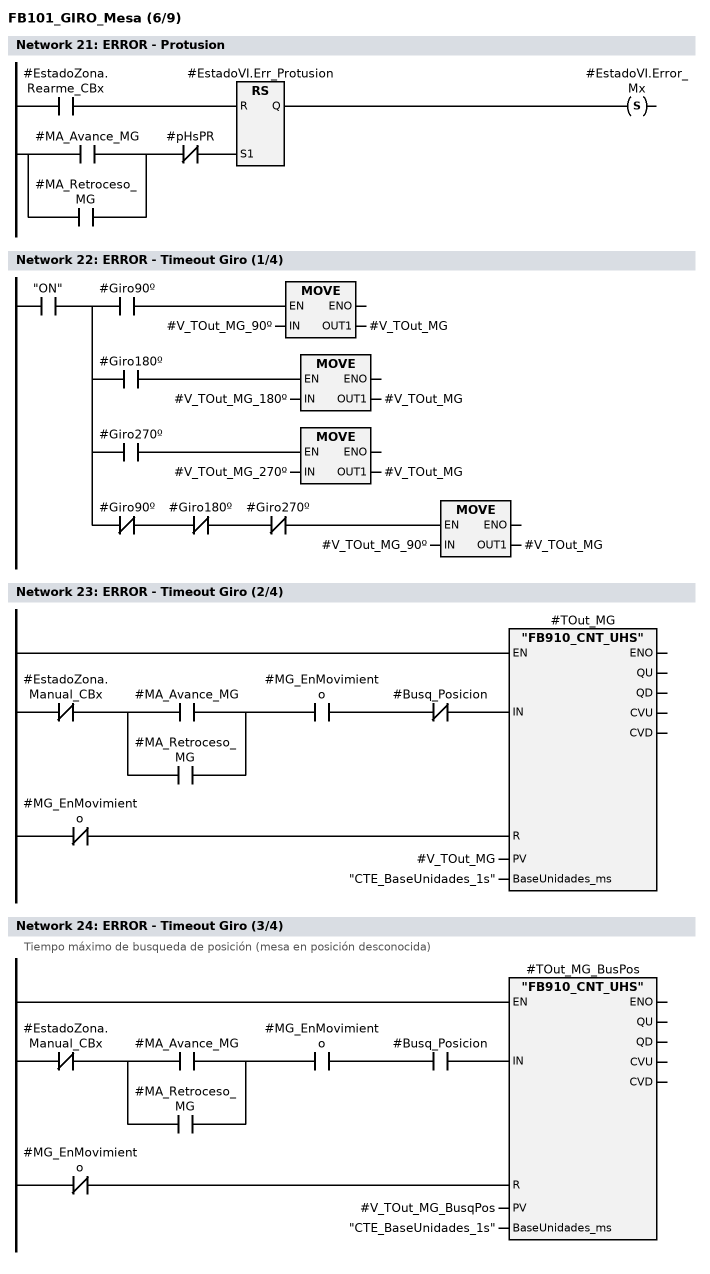
   RUNG wire#powerrail
      Contact( #EstadoZona.Rearme_CBx )
      S_RS(operand := #EstadoVI.Err_Protusion, s1 := wire#w2)
      S_Coil( #EstadoVI.Error_Mx )
   END_RUNG
   RUNG wire#powerrail
      Contact( #MA_Avance_MG )
      wire#w1
      I_Contact( #pHsPR )
   END_RUNG wire#w2
   RUNG wire#powerrail
      Contact( #MA_Retroceso_MG )
   END_RUNG wire#w1
   // the same network as SCL:
   IF #EstadoZona.Rearme_CBx THEN
       #EstadoVI.Err_Protusion := FALSE;   // RS flip-flop
   END_IF;
   IF (#MA_Avance_MG OR #MA_Retroceso_MG) AND NOT #pHsPR THEN #EstadoVI.Err_Protusion := TRUE; END_IF;
   IF #EstadoVI.Err_Protusion THEN #EstadoVI.Error_Mx := TRUE; END_IF;
END_REGION

REGION Network 22: ERROR - Timeout Giro (1/4)
   RUNG wire#powerrail
      Contact( "ON" )
      wire#w1
      Contact( #Giro90º )
      Move(in := #V_TOut_MG_90º, out1 => #V_TOut_MG)
   END_RUNG
   RUNG wire#w1
      Contact( #Giro180º )
      Move(in := #V_TOut_MG_180º, out1 => #V_TOut_MG)
   END_RUNG
   RUNG wire#w1
      Contact( #Giro270º )
      Move(in := #V_TOut_MG_270º, out1 => #V_TOut_MG)
   END_RUNG
   RUNG wire#w1
      I_Contact( #Giro90º )
      I_Contact( #Giro180º )
      I_Contact( #Giro270º )
      Move(in := #V_TOut_MG_90º, out1 => #V_TOut_MG)
   END_RUNG
   // the same network as SCL:
   IF "ON" AND #Giro90º THEN #V_TOut_MG := #V_TOut_MG_90º; END_IF;
   IF "ON" AND #Giro180º THEN #V_TOut_MG := #V_TOut_MG_180º; END_IF;
   IF "ON" AND #Giro270º THEN #V_TOut_MG := #V_TOut_MG_270º; END_IF;
   IF "ON" AND NOT #Giro90º AND NOT #Giro180º AND NOT #Giro270º THEN #V_TOut_MG := #V_TOut_MG_90º; END_IF;
END_REGION

REGION Network 23: ERROR - Timeout Giro (2/4)
   RUNG wire#powerrail
      #TOut_MG(IN := wire#w3, R := wire#w4, PV := #V_TOut_MG, BaseUnidades_ms := "CTE_BaseUnidades_1s", QU =>, QD =>, CVU =>, CVD =>)
   END_RUNG
   RUNG wire#powerrail
      I_Contact( #EstadoZona.Manual_CBx )
      wire#w1
      Contact( #MA_Avance_MG )
      wire#w2
      Contact( #MG_EnMovimiento )
      I_Contact( #Busq_Posicion )
   END_RUNG wire#w3
   RUNG wire#w1
      Contact( #MA_Retroceso_MG )
   END_RUNG wire#w2
   RUNG wire#powerrail
      I_Contact( #MG_EnMovimiento )
   END_RUNG wire#w4
   // the same network as SCL:
   #TOut_MG(IN := NOT #EstadoZona.Manual_CBx AND (#MA_Avance_MG OR #MA_Retroceso_MG) AND #MG_EnMovimiento AND NOT #Busq_Posicion,   // "FB910_CNT_UHS"
            R := NOT #MG_EnMovimiento,
            PV := #V_TOut_MG,
            BaseUnidades_ms := "CTE_BaseUnidades_1s");
END_REGION

REGION Network 24: ERROR - Timeout Giro (3/4)
   // Tiempo máximo de busqueda de posición (mesa en posición desconocida)
   RUNG wire#powerrail
      #TOut_MG_BusPos(IN := wire#w3, R := wire#w4, PV := #V_TOut_MG_BusqPos, BaseUnidades_ms := "CTE_BaseUnidades_1s", QU =>, QD =>, CVU =>, CVD =>)
   END_RUNG
   RUNG wire#powerrail
      I_Contact( #EstadoZona.Manual_CBx )
      wire#w1
      Contact( #MA_Avance_MG )
      wire#w2
      Contact( #MG_EnMovimiento )
      Contact( #Busq_Posicion )
   END_RUNG wire#w3
   RUNG wire#w1
      Contact( #MA_Retroceso_MG )
   END_RUNG wire#w2
   RUNG wire#powerrail
      I_Contact( #MG_EnMovimiento )
   END_RUNG wire#w4
   // the same network as SCL:
   #TOut_MG_BusPos(IN := NOT #EstadoZona.Manual_CBx AND (#MA_Avance_MG OR #MA_Retroceso_MG) AND #MG_EnMovimiento AND #Busq_Posicion,   // "FB910_CNT_UHS"
                   R := NOT #MG_EnMovimiento,
                   PV := #V_TOut_MG_BusqPos,
                   BaseUnidades_ms := "CTE_BaseUnidades_1s");
END_REGION

REGION Network 25: ERROR - Timeout Giro (4/4)
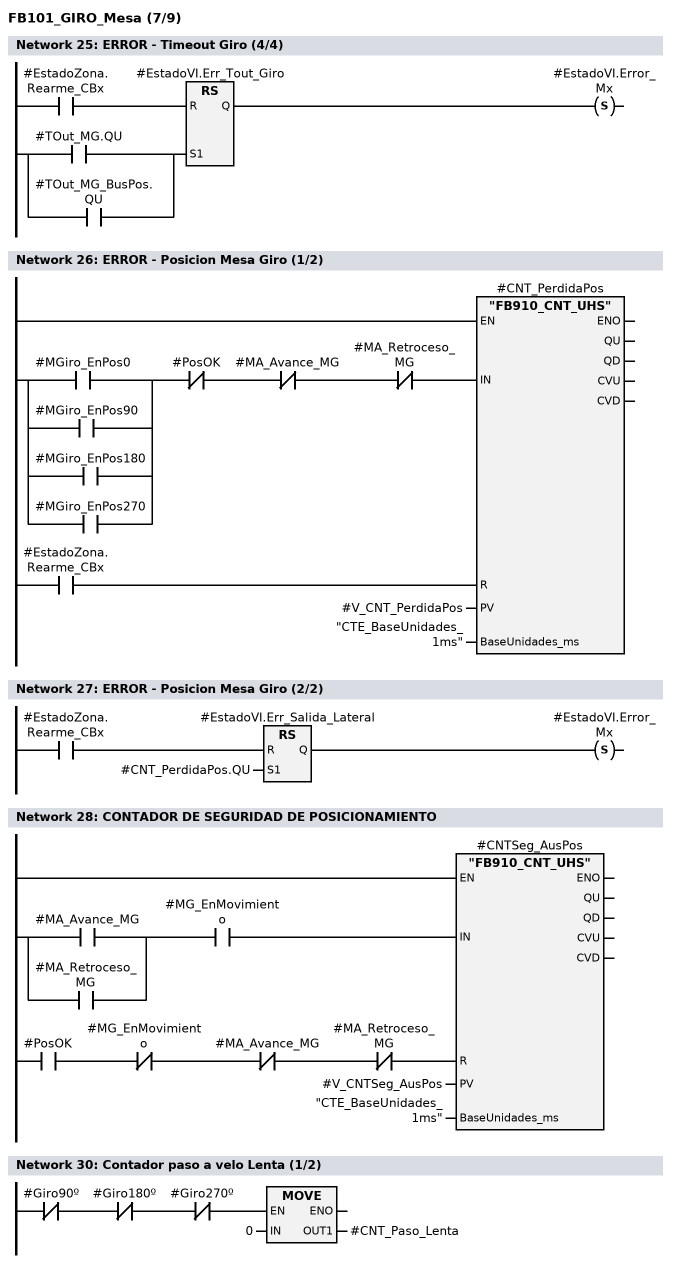
   RUNG wire#powerrail
      Contact( #EstadoZona.Rearme_CBx )
      S_RS(operand := #EstadoVI.Err_Tout_Giro, s1 := wire#w1)
      S_Coil( #EstadoVI.Error_Mx )
   END_RUNG
   RUNG wire#powerrail
      Contact( #TOut_MG.QU )
   END_RUNG wire#w1
   RUNG wire#powerrail
      Contact( #TOut_MG_BusPos.QU )
   END_RUNG wire#w1
   // the same network as SCL:
   IF #EstadoZona.Rearme_CBx THEN
       #EstadoVI.Err_Tout_Giro := FALSE;   // RS flip-flop
   END_IF;
   IF #TOut_MG.QU OR #TOut_MG_BusPos.QU THEN #EstadoVI.Err_Tout_Giro := TRUE; END_IF;
   IF #EstadoVI.Err_Tout_Giro THEN #EstadoVI.Error_Mx := TRUE; END_IF;
END_REGION

REGION Network 26: ERROR - Posicion Mesa Giro (1/2)
   RUNG wire#powerrail
      #CNT_PerdidaPos(IN := wire#w2, R := wire#w3, PV := #V_CNT_PerdidaPos, BaseUnidades_ms := "CTE_BaseUnidades_1ms", QU =>, QD =>, CVU =>, CVD =>)
   END_RUNG
   RUNG wire#powerrail
      Contact( #MGiro_EnPos0 )
      wire#w1
      I_Contact( #PosOK )
      I_Contact( #MA_Avance_MG )
      I_Contact( #MA_Retroceso_MG )
   END_RUNG wire#w2
   RUNG wire#powerrail
      Contact( #MGiro_EnPos90 )
   END_RUNG wire#w1
   RUNG wire#powerrail
      Contact( #MGiro_EnPos180 )
   END_RUNG wire#w1
   RUNG wire#powerrail
      Contact( #MGiro_EnPos270 )
   END_RUNG wire#w1
   RUNG wire#powerrail
      Contact( #EstadoZona.Rearme_CBx )
   END_RUNG wire#w3
   // the same network as SCL:
   #CNT_PerdidaPos(IN := (#MGiro_EnPos0 OR #MGiro_EnPos90 OR #MGiro_EnPos180 OR #MGiro_EnPos270) AND NOT #PosOK AND NOT #MA_Avance_MG AND NOT #MA_Retroceso_MG,   // "FB910_CNT_UHS"
                   R := #EstadoZona.Rearme_CBx,
                   PV := #V_CNT_PerdidaPos,
                   BaseUnidades_ms := "CTE_BaseUnidades_1ms");
END_REGION

REGION Network 27: ERROR - Posicion Mesa Giro (2/2)
   RUNG wire#powerrail
      Contact( #EstadoZona.Rearme_CBx )
      S_RS(operand := #EstadoVI.Err_Salida_Lateral, s1 := #CNT_PerdidaPos.QU)
      S_Coil( #EstadoVI.Error_Mx )
   END_RUNG
   // the same network as SCL:
   IF #EstadoZona.Rearme_CBx THEN
       #EstadoVI.Err_Salida_Lateral := FALSE;   // RS flip-flop
   END_IF;
   IF #CNT_PerdidaPos.QU THEN #EstadoVI.Err_Salida_Lateral := TRUE; END_IF;
   IF #EstadoVI.Err_Salida_Lateral THEN #EstadoVI.Error_Mx := TRUE; END_IF;
END_REGION

REGION Network 28: CONTADOR DE SEGURIDAD DE POSICIONAMIENTO
   RUNG wire#powerrail
      #CNTSeg_AusPos(IN := wire#w2, R := wire#w3, PV := #V_CNTSeg_AusPos, BaseUnidades_ms := "CTE_BaseUnidades_1ms", QU =>, QD =>, CVU =>, CVD =>)
   END_RUNG
   RUNG wire#powerrail
      Contact( #MA_Avance_MG )
      wire#w1
      Contact( #MG_EnMovimiento )
   END_RUNG wire#w2
   RUNG wire#powerrail
      Contact( #MA_Retroceso_MG )
   END_RUNG wire#w1
   RUNG wire#powerrail
      Contact( #PosOK )
      I_Contact( #MG_EnMovimiento )
      I_Contact( #MA_Avance_MG )
      I_Contact( #MA_Retroceso_MG )
   END_RUNG wire#w3
   // the same network as SCL:
   #CNTSeg_AusPos(IN := (#MA_Avance_MG OR #MA_Retroceso_MG) AND #MG_EnMovimiento,   // "FB910_CNT_UHS"
                  R := #PosOK AND NOT #MG_EnMovimiento AND NOT #MA_Avance_MG AND NOT #MA_Retroceso_MG,
                  PV := #V_CNTSeg_AusPos,
                  BaseUnidades_ms := "CTE_BaseUnidades_1ms");
END_REGION

REGION Network 29: CONTADOR DE VELOCIDAD LENTA
END_REGION

REGION Network 30: Contador paso a velo Lenta (1/2)
   RUNG wire#powerrail
      I_Contact( #Giro90º )
      I_Contact( #Giro180º )
      I_Contact( #Giro270º )
      { S7_GenerateENO := "TRUE" } Move(in := 0, out1 => #CNT_Paso_Lenta)
   END_RUNG
   // the same network as SCL:
   IF NOT #Giro90º AND NOT #Giro180º AND NOT #Giro270º THEN #CNT_Paso_Lenta := 0; END_IF;
END_REGION

REGION Network 31: Contador paso a velo Lenta (2/2)
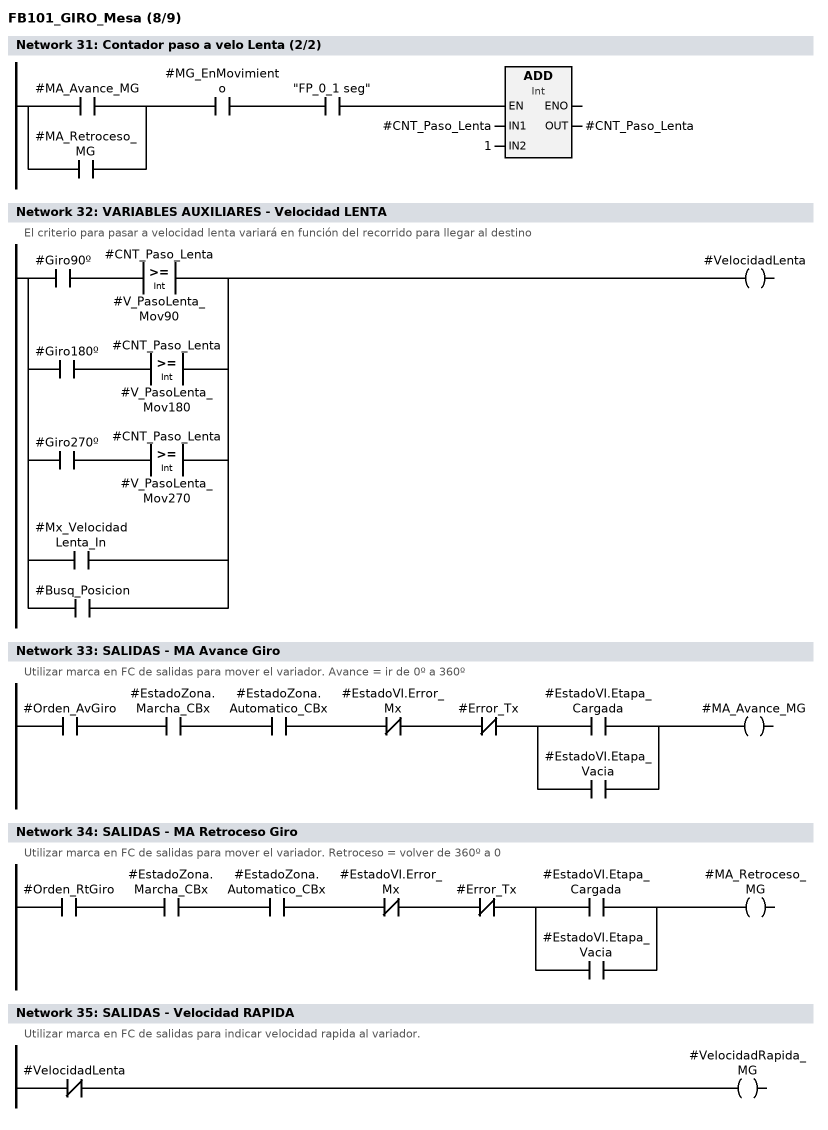
   RUNG wire#powerrail
      Contact( #MA_Avance_MG )
      wire#w1
      Contact( #MG_EnMovimiento )
      Contact( "FP_0_1 seg" )
      { S7_Templates := "SrcType := Int"; S7_GenerateENO := "TRUE" } Add(in1 := #CNT_Paso_Lenta, in2 := 1, out => #CNT_Paso_Lenta)
   END_RUNG
   RUNG wire#powerrail
      Contact( #MA_Retroceso_MG )
   END_RUNG wire#w1
   // the same network as SCL:
   IF (#MA_Avance_MG OR #MA_Retroceso_MG) AND #MG_EnMovimiento AND "FP_0_1 seg" THEN
       #CNT_Paso_Lenta := #CNT_Paso_Lenta + 1;
   END_IF;
END_REGION

REGION Network 32: VARIABLES AUXILIARES - Velocidad LENTA
   // El criterio para pasar a velocidad lenta variará en función del recorrido para llegar al destino
   RUNG wire#powerrail
      Contact( #Giro90º )
      { S7_Templates := "SrcType := Int" } GE_Contact(in1 := #CNT_Paso_Lenta, in2 := #V_PasoLenta_Mov90)
      wire#w1
      Coil( #VelocidadLenta )
   END_RUNG
   RUNG wire#powerrail
      Contact( #Giro180º )
      { S7_Templates := "SrcType := Int" } GE_Contact(in1 := #CNT_Paso_Lenta, in2 := #V_PasoLenta_Mov180)
   END_RUNG wire#w1
   RUNG wire#powerrail
      Contact( #Giro270º )
      { S7_Templates := "SrcType := Int" } GE_Contact(in1 := #CNT_Paso_Lenta, in2 := #V_PasoLenta_Mov270)
   END_RUNG wire#w1
   RUNG wire#powerrail
      Contact( #Mx_VelocidadLenta_In )
   END_RUNG wire#w1
   RUNG wire#powerrail
      Contact( #Busq_Posicion )
   END_RUNG wire#w1
   // the same network as SCL:
   #VelocidadLenta := (#Giro90º AND (#CNT_Paso_Lenta >= #V_PasoLenta_Mov90)) OR (#Giro180º AND (#CNT_Paso_Lenta >= #V_PasoLenta_Mov180)) OR (#Giro270º AND (#CNT_Paso_Lenta >= #V_PasoLenta_Mov270)) OR #Mx_VelocidadLenta_In OR #Busq_Posicion;
END_REGION

REGION Network 33: SALIDAS - MA Avance Giro
   // Utilizar marca en FC de salidas para mover el variador. Avance = ir de 0º a 360º
   RUNG wire#powerrail
      Contact( #Orden_AvGiro )
      Contact( #EstadoZona.Marcha_CBx )
      Contact( #EstadoZona.Automatico_CBx )
      I_Contact( #EstadoVI.Error_Mx )
      I_Contact( #Error_Tx )
      wire#w1
      Contact( #EstadoVI.Etapa_Cargada )
      wire#w2
      Coil( #MA_Avance_MG )
   END_RUNG
   RUNG wire#w1
      Contact( #EstadoVI.Etapa_Vacia )
   END_RUNG wire#w2
   // the same network as SCL:
   #MA_Avance_MG := #Orden_AvGiro AND #EstadoZona.Marcha_CBx AND #EstadoZona.Automatico_CBx AND NOT #EstadoVI.Error_Mx AND NOT #Error_Tx AND (#EstadoVI.Etapa_Cargada OR #EstadoVI.Etapa_Vacia);
END_REGION

REGION Network 34: SALIDAS - MA Retroceso Giro
   // Utilizar marca en FC de salidas para mover el variador. Retroceso = volver de 360º a 0
   RUNG wire#powerrail
      Contact( #Orden_RtGiro )
      Contact( #EstadoZona.Marcha_CBx )
      Contact( #EstadoZona.Automatico_CBx )
      I_Contact( #EstadoVI.Error_Mx )
      I_Contact( #Error_Tx )
      wire#w1
      Contact( #EstadoVI.Etapa_Cargada )
      wire#w2
      Coil( #MA_Retroceso_MG )
   END_RUNG
   RUNG wire#w1
      Contact( #EstadoVI.Etapa_Vacia )
   END_RUNG wire#w2
   // the same network as SCL:
   #MA_Retroceso_MG := #Orden_RtGiro AND #EstadoZona.Marcha_CBx AND #EstadoZona.Automatico_CBx AND NOT #EstadoVI.Error_Mx AND NOT #Error_Tx AND (#EstadoVI.Etapa_Cargada OR #EstadoVI.Etapa_Vacia);
END_REGION

REGION Network 35: SALIDAS - Velocidad RAPIDA
   // Utilizar marca en FC de salidas para indicar velocidad rapida al variador.
   RUNG wire#powerrail
      I_Contact( #VelocidadLenta )
      Coil( #VelocidadRapida_MG )
   END_RUNG
   // the same network as SCL:
   #VelocidadRapida_MG := NOT #VelocidadLenta;
END_REGION

REGION Network 36: ENTRADAS DE LA MESA
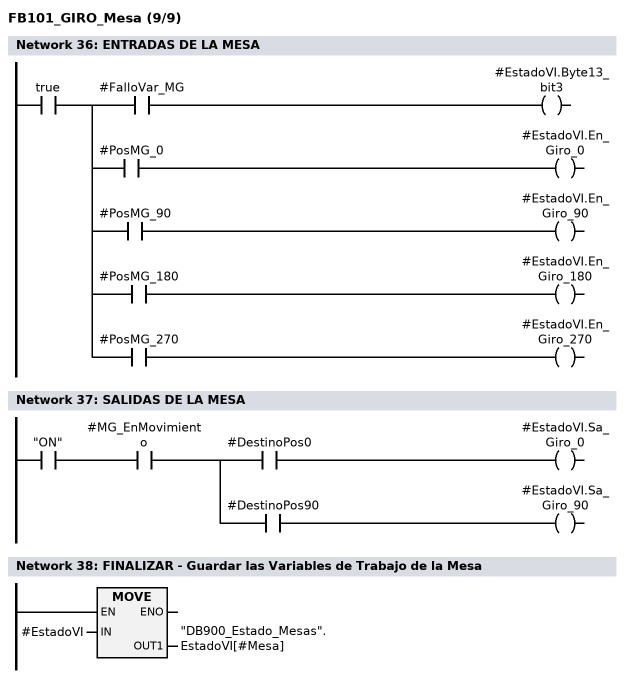
   RUNG wire#powerrail
      Contact( true )
      wire#w1
      Contact( #FalloVar_MG )
      Coil( #EstadoVI.Byte13_bit3 )
   END_RUNG
   RUNG wire#w1
      Contact( #PosMG_0 )
      Coil( #EstadoVI.En_Giro_0 )
   END_RUNG
   RUNG wire#w1
      Contact( #PosMG_90 )
      Coil( #EstadoVI.En_Giro_90 )
   END_RUNG
   RUNG wire#w1
      Contact( #PosMG_180 )
      Coil( #EstadoVI.En_Giro_180 )
   END_RUNG
   RUNG wire#w1
      Contact( #PosMG_270 )
      Coil( #EstadoVI.En_Giro_270 )
   END_RUNG
   // the same network as SCL:
   #EstadoVI.Byte13_bit3 := true AND #FalloVar_MG;
   #EstadoVI.En_Giro_0 := true AND #PosMG_0;
   #EstadoVI.En_Giro_90 := true AND #PosMG_90;
   #EstadoVI.En_Giro_180 := true AND #PosMG_180;
   #EstadoVI.En_Giro_270 := true AND #PosMG_270;
END_REGION

REGION Network 37: SALIDAS DE LA MESA
   RUNG wire#powerrail
      Contact( "ON" )
      Contact( #MG_EnMovimiento )
      wire#w1
      Contact( #DestinoPos0 )
      Coil( #EstadoVI.Sa_Giro_0 )
   END_RUNG
   RUNG wire#w1
      Contact( #DestinoPos90 )
      Coil( #EstadoVI.Sa_Giro_90 )
   END_RUNG
   // the same network as SCL:
   #_w1 := "ON" AND #MG_EnMovimiento;
   #EstadoVI.Sa_Giro_0 := #_w1 AND #DestinoPos0;
   #EstadoVI.Sa_Giro_90 := #_w1 AND #DestinoPos90;
END_REGION

REGION Network 38: FINALIZAR - Guardar las Variables de Trabajo de la Mesa
   RUNG wire#powerrail
      Move(in := #EstadoVI, out1 => "DB900_Estado_Mesas".EstadoVI[#Mesa])
   END_RUNG
   // the same network as SCL:
   "DB900_Estado_Mesas".EstadoVI[#Mesa] := #EstadoVI;
END_REGION
END_FUNCTION_BLOCK

FUNCTION_BLOCK "FB12_M_PASO_ELEV_E1E2E3E4_S1S2S3S4_UPDW"   // FB12, LAD
TITLE = Control del Ramal de Salidas
{ S7_Optimized_Access := 'FALSE' }
AUTHOR : M_ELEVA
NAME : 20160509
VERSION : 3.7
// stored: AutoNumber false, SetENOAutomatically false
   VAR_INPUT
      Mesa : UInt;   // Mesa de la FB
      Error_Tx : Bool;   // Error en el Tx
      EnTension : Bool;   // Existe Tension en la Mesa
      Termico_Tx : Bool;   // Proteccion del Tx
      pHsMx_1 : Bool;   // pHs de la Mesa (Para Entrada por E3E4)
      pHsMx_2 : Bool;   // pHs de la Mesa (Para Entrada por E1E2)
      pHsMx_PR1 : Bool;   // pHs de Protrusion de la Mesa. Nota: No existe >> ON
      pHsMx_PR3 : Bool;   // pHs de Protrusion de la Mesa. Nota: No existe >> ON
      Avance_Tx : Bool;   // Avance del Tx
      Retroceso_Tx : Bool;   // Retroceso del Tx
      Termico_MELEV : Bool;   // Protecion de la Mesa Elevadora
      MELEV_DetectorSeg : Bool;   // Detector de Seguridad >>> Mesa Elevadora
      MELEV_UP : Bool;   // Posicion Arriba >>> Mesa Elevadora
      MELEV_DW : Bool;   // Posicion Abajo >>> Mesa Elevadora
      MELEV_EnMovimiento : Bool;   // EnMovimiento >>> Mesa Elevadora
      Pos_Rep_Vacio_DW : Bool;   // Pos. Reposo Vacia DW >>> Config
      Pos_Rep_Vacio_UP : Bool;   // Pos. Reposo Vacia UP >>> Config
      Pos_Rep_Carga_DW : Bool;   // Pos. Reposo Cargada DW >>> Config
      Pos_Rep_Carga_UP : Bool;   // Pos. Reposo Cargada UP >>> Config
      MAnt_DescargaAct_M1_DW : Bool;   // E1 >> Mesa Anterior DescargaAct
      AVTF_Ent_M1_DW : Bool;   // E1 >> Mesa Anterior AVTF
      P_Mens_Ent_M1_DW : Bool;   // E1 >> Mesa Anterior P_Mens
      MAnt_DescargaAct_M3_DW : Bool;   // E3 >> Mesa Anterior DescargaAct
      AVTF_Ent_M3_DW : Bool;   // E3 >> Mesa Anterior AVTF
      P_Mens_Ent_M3_DW : Bool;   // E3 >> Mesa Anterior P_Mens
      PTF_Sal_M1_DW : Bool;   // S1 >> Mesa Siguiente PTF
      FTF_Sal_M1_DW : Bool;   // S1 >> Mesa Siguiente FTF
      PTF_Sal_M3_DW : Bool;   // S3 >> Mesa Siguiente PTF
      FTF_Sal_M3_DW : Bool;   // S3 >> Mesa Siguiente FTF
      MSig_CargaAct_M1_DW : Bool;
      MSig_CargaAct_M3_DW : Bool;
      MAnt_DescargaAct_M2_UP : Bool;   // E2 >> Mesa Anterior DescargaAct
      AVF_Ent_M2_UP : Bool;   // E2 >> Mesa Anterior AVTF
      P_Mens_Ent_M2_UP : Bool;   // E2 >> Mesa Anterior P_Mens
      MAnt_DescargaAct_M4_UP : Bool;   // E4 >> Mesa Anterior DescargaAct
      AVTF_Ent_M4_UP : Bool;   // E4 >> Mesa Anterior AVTF
      P_Mens_Ent_M4_UP : Bool;   // E4 >> Mesa Anterior P_Mens
      PTF_Sal_M2_UP : Bool;   // S2 >> Mesa Siguiente PTF
      FTF_Sal_M2_UP : Bool;   // S2 >> Mesa Siguiente FTF
      PTF_Sal_M4_UP : Bool;   // S4 >> Mesa Siguiente PTF
      FTF_Sal_M4_UP : Bool;   // S4 >> Mesa Siguiente FTF
      MSig_CargaAct_M2_UP : Bool;
      MSig_CargaAct_M4_UP : Bool;
      Mx_VelocidadLenta_In : Bool;   // Forzar a Velociada Lenta
      F_ENV_MENS_Mx : Bool;   // Fin de Envio de Mensaje
      OrdSal_M1_DW : Bool;   // Orden de Salida por S1
      OrdSal_M3_DW : Bool;   // Orden de Salida por S3
      OrdSal_M2_UP : Bool;   // Orden de Salida por S2
      OrdSal_M4_UP : Bool;   // Orden de Salida por S4
      V_CNT_pHsMx : Int := 1000;   // Valor de Presencia
      V_CNT_pHsMx_FTF : Int := 200;   // Valor para activar FTF. Nota: < = V_CNT_pHsMx.
      V_CNTSeg_pHsMx : Int := 2000;   // Valor de Seguriadad para Presencia
      V_CNT_PasoLenta : Int := 2000;   // Valor de Paso a Lenta
      V_CNT_ApHsMx : Int := 200;   // Valor de Ausencia
      V_CNTSeg_ApHsMx : Int := 2000;   // Valor de Seguriadad para Ausencia
      V_TOut_Tx_Mx : Int := 30000;   // TimeOut de Entrada por E1
      V_TOut_MELEV : Int := 5000;   // TimeOut de Mesa Elevadora
      V_TMP_Protrusion : Int := 200;   // TMP de Protrusion
      V_CNT_PerdidapHs : Int := 1000;   // CNT de Perdida de pHs
   END_VAR
   VAR_OUTPUT
      P_EnvMens_PMx : Bool;   // Permiso de Enviar Mensaje de Presencia
      P_RecepOK_Mx : Bool;   // Recepcion OK
      PTF_Ent_M1_DW : Bool;   // E1 >> Mesa Anterior PTF
      FTF_Ent_M1_DW : Bool;   // E1 >> Mesa Anterior FTF
      PTF_Ent_M3_DW : Bool;   // E3 >> Mesa Anterior PTF
      FTF_Ent_M3_DW : Bool;   // E3 >> Mesa Anterior FTF
      AVTF_Sal_M1_DW : Bool;   // S1 >> Mesa Siguiente AVTF
      P_Mens_Sal_M1_DW : Bool;   // S1 >> Mesa Siguiente P_Mens
      AVTF_Sal_M3_DW : Bool;   // S3 >> Mesa Siguiente AVTF
      P_Mens_Sal_M3_DW : Bool;   // S3 >> Mesa Siguiente P_Mens
      PTF_Ent_M2_UP : Bool;   // E2 >> Mesa Anterior PTF
      FTF_Ent_M2_UP : Bool;   // E2 >> Mesa Anterior FTF
      PTF_Ent_M4_UP : Bool;   // E4 >> Mesa Anterior PTF
      FTF_Ent_M4_UP : Bool;   // E4 >> Mesa Anterior FTF
      AVTF_Sal_M2_UP : Bool;   // S2 >> Mesa Siguiente AVTF
      P_Mens_Sal_M2_UP : Bool;   // S2 >> Mesa Siguiente P_Mens
      AVTF_Sal_M4_UP : Bool;   // S4 >> Mesa Siguiente AVTF
      P_Mens_Sal_M4_UP : Bool;   // S4 >> Mesa Siguiente P_Mens
   END_VAR
   VAR
      Anular_pr1 : Bool;   // ???
      Anular_pr3 : Bool;   // ???
      Mx_ET00 : Bool;
      Mx_ET01 { ExternalWritable := 'False'} : Bool;
      Mx_ET02 : Bool;
      Mx_ET08 : Bool;
      Mx_ET09 : Bool;
      Mx_ET10 : Bool;
      Mx_ET11 : Bool;
      Mx_ET12 : Bool;
      Mx_ET110 : Bool;
      Mx_ET111 : Bool;
      Mx_ET50 : Bool;
      Mx_ET51 : Bool;
      Mx_ET150 : Bool;
      Mx_ET151 : Bool;
      Selec_UP : Bool;   // Seleccionado UP de la Mesa Elevadora
      Selec_DW : Bool;   // Seleccionado DW de la Mesa Elevadora
      Selec_M1M2_Entrada : Bool;   // Seleccionado Entrada E1_DW y E2_UP
      Selec_M3M4_Entrada : Bool;   // Seleccionado Entrada E3_DW y E4_UP
      Selec_M1M2_Salida : Bool;   // Seleccionado Salida E1_DW y E2_UP
      Selec_M3M4_Salida : Bool;   // Seleccionado Salida E3_DW y E4_UP
      MEnt_DescargaAct : Bool;   // Interlock >> DesCargaAct de MAnt >> Mx
      AVTF_MEnt : Bool;   // Interlock >> AVTF de MAnt >> Mx
      P_Mens_MEnt : Bool;   // Interlock >> P_Mens de MAnt >> Mx
      PTF_MEnt : Bool;   // Interlock >> PTF de MAnt >> Mx
      FTF_MEnt : Bool;   // Interlock >> FTF de MAnt >> Mx
      AVTF_MSal : Bool;   // Interlock >> AVTF de Mx >> MSig
      P_Mens_MSal : Bool;   // Interlock >> P_Mens de Mx >> MSig
      PTF_MSal : Bool;   // Interlock >> PTF de Mx >> MSig
      FTF_MSal : Bool;   // Interlock >> FTF de Mx >> MSig
      ProtocoloInciado : Bool;   // Iniciado el Envio del Mensaje de Presencia
      STAT_EnvMens_PMx : Bool;   // Interna >> Envio del Mensaje de Presencia
      CNT_pHsMx_FTF_OK : Bool;   // Enviar ya FTF
      CNT_pHsMx { S7_SetPoint := 'True'} : "FB910_CNT_UHS";   // CNT de la Presencia
      CNTSeg_pHsMx { S7_SetPoint := 'True'} : "FB910_CNT_UHS";   // CNT de Seguridad de la Presencia
      CNT_ApHsMx { S7_SetPoint := 'True'} : "FB910_CNT_UHS";   // CNT de la Ausencia
      CNTSeg_ApHsMx { S7_SetPoint := 'True'} : "FB910_CNT_UHS";   // CNT de Seguridad de la Ausencia
      TMP_EnTension { S7_SetPoint := 'True'} : "FB910_CNT_UHS";
      TOut_Av_Mx { S7_SetPoint := 'True'} : "FB910_CNT_UHS";   // Time Out de Entrada de E1 o E2
      TOut_Rt_Mx { S7_SetPoint := 'True'} : "FB910_CNT_UHS";   // Time Out de Entrada de E3 o E4
      TOut_Subir_MELEV { S7_SetPoint := 'True'} : "FB910_CNT_UHS";   // Time Out de Subida de Mesa Elevadora
      TOut_Bajar_MELEV { S7_SetPoint := 'True'} : "FB910_CNT_UHS";   // Time Out de Bajada de Mesa Elevadora
      TMP_Protrusion { S7_SetPoint := 'True'} : "FB910_CNT_UHS";   // TMP de la Protrusion
      CNT_PerdidapHs { S7_SetPoint := 'True'} : "FB910_CNT_UHS";   // CNT de Perdida de pHs
   END_VAR
   VAR_TEMP
      EstadoZona : "EstadoZona";   // Estado de Zona de la Mesa
      EstadoVI : "EstadosMesa";   // Estado del Vehiculo Inteliguente de la Mesa
      ConfigFB : "UDT_ConfigFB";   // Configuracion de la FB de la Mesa
      V_Protrusion : Int;
      Aux_ET00 : Bool;
   END_VAR
   VAR_TEMP   // added for the SCL form of the ladder/FBD networks
      _w1 : Bool;
      _w2 : Bool;
      _w3 : Bool;
      _w4 : Bool;
      _w5 : Bool;
      _w6 : Bool;
   END_VAR
BEGIN

REGION Network 1: INICIALIZAR - Recoger las Variables de Estado de la Mesa
   // Se recoge - Estado_CBx
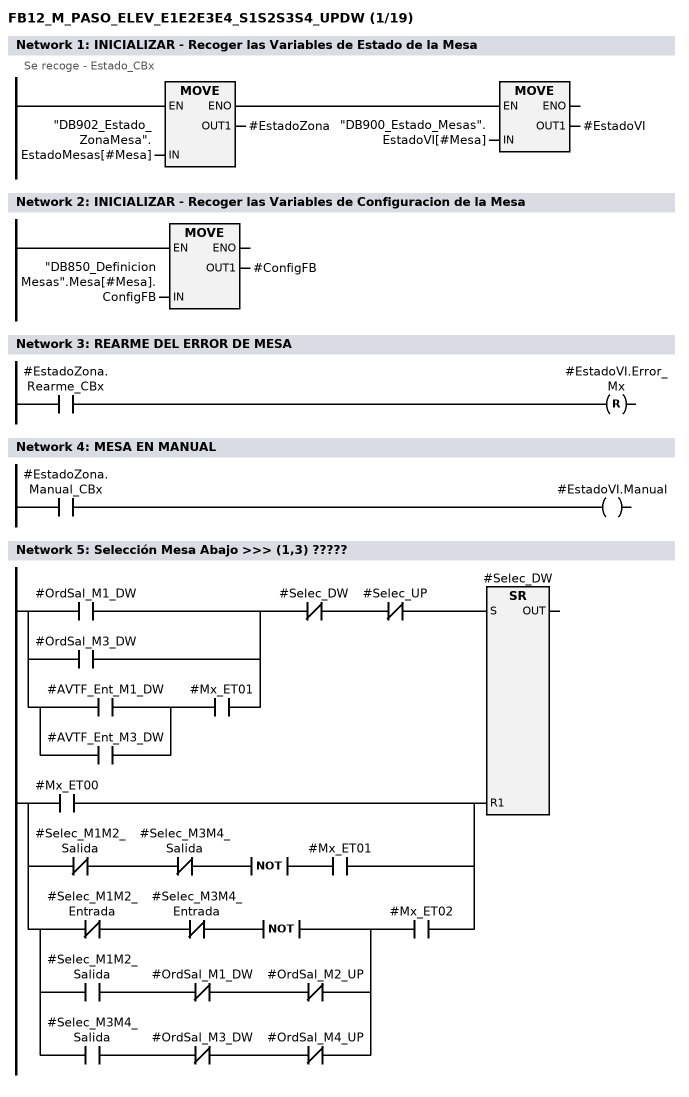
   RUNG wire#powerrail
      Move(in := "DB902_Estado_ZonaMesa".EstadoMesas[#Mesa], out1 => #EstadoZona)
      Move(in := "DB900_Estado_Mesas".EstadoVI[#Mesa], out1 => #EstadoVI)
   END_RUNG
   // the same network as SCL:
   #EstadoZona := "DB902_Estado_ZonaMesa".EstadoMesas[#Mesa];
   #EstadoVI := "DB900_Estado_Mesas".EstadoVI[#Mesa];
END_REGION

REGION Network 2: INICIALIZAR - Recoger las Variables de Configuracion de la Mesa
   RUNG wire#powerrail
      Move(in := "DB850_DefinicionMesas".Mesa[#Mesa].ConfigFB, out1 => #ConfigFB)
   END_RUNG
   // the same network as SCL:
   #ConfigFB := "DB850_DefinicionMesas".Mesa[#Mesa].ConfigFB;
END_REGION

REGION Network 3: REARME DEL ERROR DE MESA
   RUNG wire#powerrail
      Contact( #EstadoZona.Rearme_CBx )
      R_Coil( #EstadoVI.Error_Mx )
   END_RUNG
   // the same network as SCL:
   IF #EstadoZona.Rearme_CBx THEN #EstadoVI.Error_Mx := FALSE; END_IF;
END_REGION

REGION Network 4: MESA EN MANUAL
   RUNG wire#powerrail
      Contact( #EstadoZona.Manual_CBx )
      Coil( #EstadoVI.Manual )
   END_RUNG
   // the same network as SCL:
   #EstadoVI.Manual := #EstadoZona.Manual_CBx;
END_REGION

REGION Network 5: Selección Mesa Abajo >>> (1,3) ?????
   RUNG wire#powerrail
      Contact( #OrdSal_M1_DW )
      wire#w1
      I_Contact( #Selec_DW )
      I_Contact( #Selec_UP )
      S_SR(operand := #Selec_DW, r1 := wire#w4)
   END_RUNG
   RUNG wire#powerrail
      Contact( #OrdSal_M3_DW )
   END_RUNG wire#w1
   RUNG wire#powerrail
      Contact( #AVTF_Ent_M1_DW )
      wire#w2
      Contact( #Mx_ET01 )
   END_RUNG wire#w1
   RUNG wire#powerrail
      Contact( #AVTF_Ent_M3_DW )
   END_RUNG wire#w2
   RUNG wire#powerrail
      Contact( #Mx_ET00 )
   END_RUNG wire#w4
   RUNG wire#powerrail
      I_Contact( #Selec_M1M2_Salida )
      I_Contact( #Selec_M3M4_Salida )
      Not()
      Contact( #Mx_ET01 )
   END_RUNG wire#w4
   RUNG wire#powerrail
      I_Contact( #Selec_M1M2_Entrada )
      I_Contact( #Selec_M3M4_Entrada )
      Not()
      wire#w3
      Contact( #Mx_ET02 )
   END_RUNG wire#w4
   RUNG wire#powerrail
      Contact( #Selec_M1M2_Salida )
      I_Contact( #OrdSal_M1_DW )
      I_Contact( #OrdSal_M2_UP )
   END_RUNG wire#w3
   RUNG wire#powerrail
      Contact( #Selec_M3M4_Salida )
      I_Contact( #OrdSal_M3_DW )
      I_Contact( #OrdSal_M4_UP )
   END_RUNG wire#w3
   // the same network as SCL:
   IF (#OrdSal_M1_DW OR #OrdSal_M3_DW OR ((#AVTF_Ent_M1_DW OR #AVTF_Ent_M3_DW) AND #Mx_ET01)) AND NOT #Selec_DW AND NOT #Selec_UP THEN
       #Selec_DW := TRUE;   // SR flip-flop
   END_IF;
   IF #Mx_ET00 OR (NOT (NOT #Selec_M1M2_Salida AND NOT #Selec_M3M4_Salida) AND #Mx_ET01) OR ((NOT (NOT #Selec_M1M2_Entrada AND NOT #Selec_M3M4_Entrada) OR (#Selec_M1M2_Salida AND NOT #OrdSal_M1_DW AND NOT #OrdSal_M2_UP) OR (#Selec_M3M4_Salida AND NOT #OrdSal_M3_DW AND NOT #OrdSal_M4_UP)) AND #Mx_ET02) THEN
       #Selec_DW := FALSE;
   END_IF;
END_REGION

REGION Network 6: Selección Mesa Arriba >>> (2,4) ?????
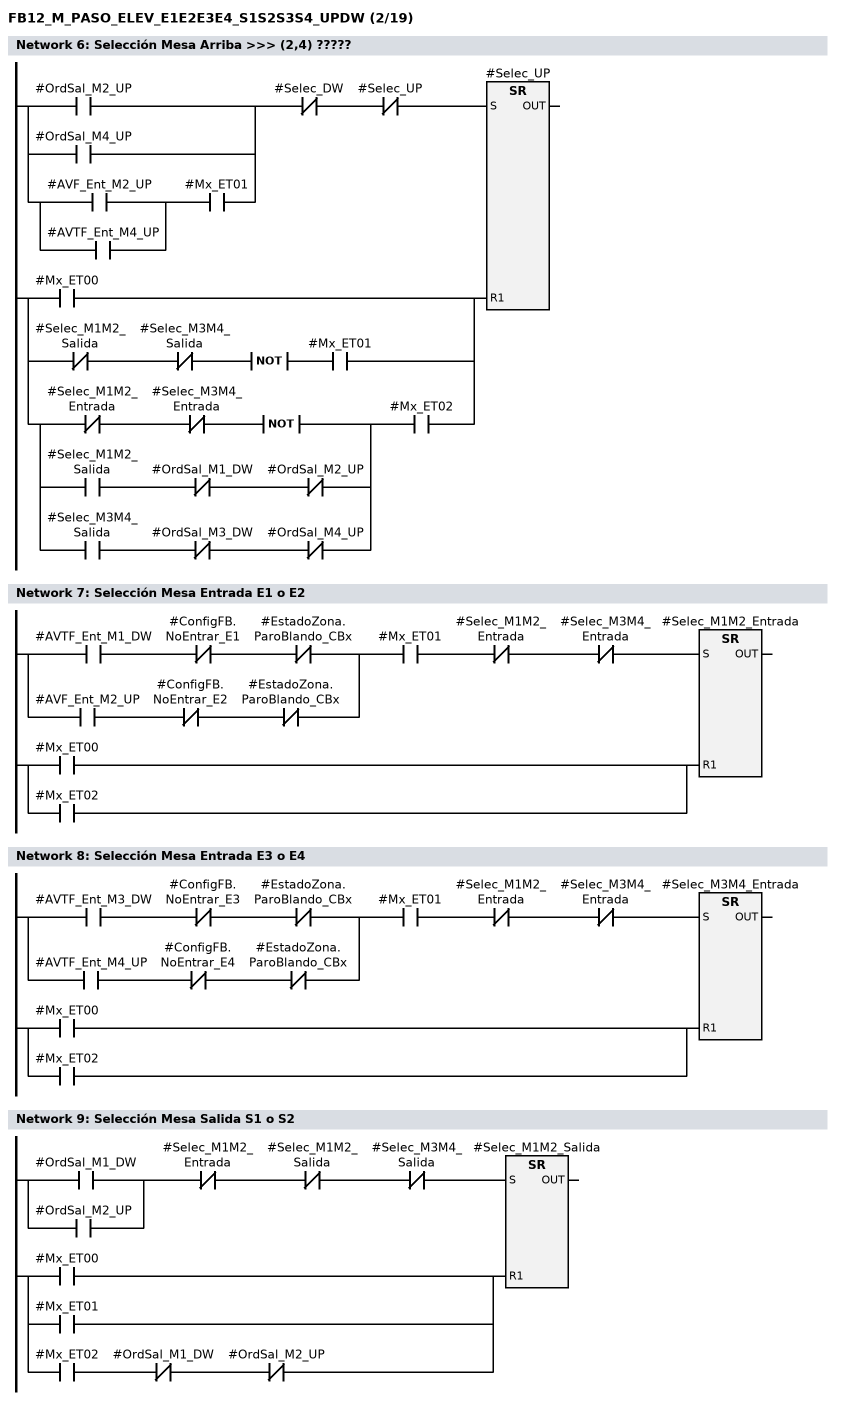
   RUNG wire#powerrail
      Contact( #OrdSal_M2_UP )
      wire#w1
      I_Contact( #Selec_DW )
      I_Contact( #Selec_UP )
      S_SR(operand := #Selec_UP, r1 := wire#w4)
   END_RUNG
   RUNG wire#powerrail
      Contact( #OrdSal_M4_UP )
   END_RUNG wire#w1
   RUNG wire#powerrail
      Contact( #AVF_Ent_M2_UP )
      wire#w2
      Contact( #Mx_ET01 )
   END_RUNG wire#w1
   RUNG wire#powerrail
      Contact( #AVTF_Ent_M4_UP )
   END_RUNG wire#w2
   RUNG wire#powerrail
      Contact( #Mx_ET00 )
   END_RUNG wire#w4
   RUNG wire#powerrail
      I_Contact( #Selec_M1M2_Salida )
      I_Contact( #Selec_M3M4_Salida )
      Not()
      Contact( #Mx_ET01 )
   END_RUNG wire#w4
   RUNG wire#powerrail
      I_Contact( #Selec_M1M2_Entrada )
      I_Contact( #Selec_M3M4_Entrada )
      Not()
      wire#w3
      Contact( #Mx_ET02 )
   END_RUNG wire#w4
   RUNG wire#powerrail
      Contact( #Selec_M1M2_Salida )
      I_Contact( #OrdSal_M1_DW )
      I_Contact( #OrdSal_M2_UP )
   END_RUNG wire#w3
   RUNG wire#powerrail
      Contact( #Selec_M3M4_Salida )
      I_Contact( #OrdSal_M3_DW )
      I_Contact( #OrdSal_M4_UP )
   END_RUNG wire#w3
   // the same network as SCL:
   IF (#OrdSal_M2_UP OR #OrdSal_M4_UP OR ((#AVF_Ent_M2_UP OR #AVTF_Ent_M4_UP) AND #Mx_ET01)) AND NOT #Selec_DW AND NOT #Selec_UP THEN
       #Selec_UP := TRUE;   // SR flip-flop
   END_IF;
   IF #Mx_ET00 OR (NOT (NOT #Selec_M1M2_Salida AND NOT #Selec_M3M4_Salida) AND #Mx_ET01) OR ((NOT (NOT #Selec_M1M2_Entrada AND NOT #Selec_M3M4_Entrada) OR (#Selec_M1M2_Salida AND NOT #OrdSal_M1_DW AND NOT #OrdSal_M2_UP) OR (#Selec_M3M4_Salida AND NOT #OrdSal_M3_DW AND NOT #OrdSal_M4_UP)) AND #Mx_ET02) THEN
       #Selec_UP := FALSE;
   END_IF;
END_REGION

REGION Network 7: Selección Mesa Entrada E1 o E2
   RUNG wire#powerrail
      Contact( #AVTF_Ent_M1_DW )
      I_Contact( #ConfigFB.NoEntrar_E1 )
      I_Contact( #EstadoZona.ParoBlando_CBx )
      wire#w1
      Contact( #Mx_ET01 )
      I_Contact( #Selec_M1M2_Entrada )
      I_Contact( #Selec_M3M4_Entrada )
      S_SR(operand := #Selec_M1M2_Entrada, r1 := wire#w2)
   END_RUNG
   RUNG wire#powerrail
      Contact( #AVF_Ent_M2_UP )
      I_Contact( #ConfigFB.NoEntrar_E2 )
      I_Contact( #EstadoZona.ParoBlando_CBx )
   END_RUNG wire#w1
   RUNG wire#powerrail
      Contact( #Mx_ET00 )
   END_RUNG wire#w2
   RUNG wire#powerrail
      Contact( #Mx_ET02 )
   END_RUNG wire#w2
   // the same network as SCL:
   IF ((#AVTF_Ent_M1_DW AND NOT #ConfigFB.NoEntrar_E1 AND NOT #EstadoZona.ParoBlando_CBx) OR (#AVF_Ent_M2_UP AND NOT #ConfigFB.NoEntrar_E2 AND NOT #EstadoZona.ParoBlando_CBx)) AND #Mx_ET01 AND NOT #Selec_M1M2_Entrada AND NOT #Selec_M3M4_Entrada THEN
       #Selec_M1M2_Entrada := TRUE;   // SR flip-flop
   END_IF;
   IF #Mx_ET00 OR #Mx_ET02 THEN #Selec_M1M2_Entrada := FALSE; END_IF;
END_REGION

REGION Network 8: Selección Mesa Entrada E3 o E4
   RUNG wire#powerrail
      Contact( #AVTF_Ent_M3_DW )
      I_Contact( #ConfigFB.NoEntrar_E3 )
      I_Contact( #EstadoZona.ParoBlando_CBx )
      wire#w1
      Contact( #Mx_ET01 )
      I_Contact( #Selec_M1M2_Entrada )
      I_Contact( #Selec_M3M4_Entrada )
      S_SR(operand := #Selec_M3M4_Entrada, r1 := wire#w2)
   END_RUNG
   RUNG wire#powerrail
      Contact( #AVTF_Ent_M4_UP )
      I_Contact( #ConfigFB.NoEntrar_E4 )
      I_Contact( #EstadoZona.ParoBlando_CBx )
   END_RUNG wire#w1
   RUNG wire#powerrail
      Contact( #Mx_ET00 )
   END_RUNG wire#w2
   RUNG wire#powerrail
      Contact( #Mx_ET02 )
   END_RUNG wire#w2
   // the same network as SCL:
   IF ((#AVTF_Ent_M3_DW AND NOT #ConfigFB.NoEntrar_E3 AND NOT #EstadoZona.ParoBlando_CBx) OR (#AVTF_Ent_M4_UP AND NOT #ConfigFB.NoEntrar_E4 AND NOT #EstadoZona.ParoBlando_CBx)) AND #Mx_ET01 AND NOT #Selec_M1M2_Entrada AND NOT #Selec_M3M4_Entrada THEN
       #Selec_M3M4_Entrada := TRUE;   // SR flip-flop
   END_IF;
   IF #Mx_ET00 OR #Mx_ET02 THEN #Selec_M3M4_Entrada := FALSE; END_IF;
END_REGION

REGION Network 9: Selección Mesa Salida S1 o S2
   RUNG wire#powerrail
      Contact( #OrdSal_M1_DW )
      wire#w1
      I_Contact( #Selec_M1M2_Entrada )
      I_Contact( #Selec_M1M2_Salida )
      I_Contact( #Selec_M3M4_Salida )
      S_SR(operand := #Selec_M1M2_Salida, r1 := wire#w2)
   END_RUNG
   RUNG wire#powerrail
      Contact( #OrdSal_M2_UP )
   END_RUNG wire#w1
   RUNG wire#powerrail
      Contact( #Mx_ET00 )
   END_RUNG wire#w2
   RUNG wire#powerrail
      Contact( #Mx_ET01 )
   END_RUNG wire#w2
   RUNG wire#powerrail
      Contact( #Mx_ET02 )
      I_Contact( #OrdSal_M1_DW )
      I_Contact( #OrdSal_M2_UP )
   END_RUNG wire#w2
   // the same network as SCL:
   IF (#OrdSal_M1_DW OR #OrdSal_M2_UP) AND NOT #Selec_M1M2_Entrada AND NOT #Selec_M1M2_Salida AND NOT #Selec_M3M4_Salida THEN
       #Selec_M1M2_Salida := TRUE;   // SR flip-flop
   END_IF;
   IF #Mx_ET00 OR #Mx_ET01 OR (#Mx_ET02 AND NOT #OrdSal_M1_DW AND NOT #OrdSal_M2_UP) THEN
       #Selec_M1M2_Salida := FALSE;
   END_IF;
END_REGION

REGION Network 10: Selección Mesa Salida S3 o S4
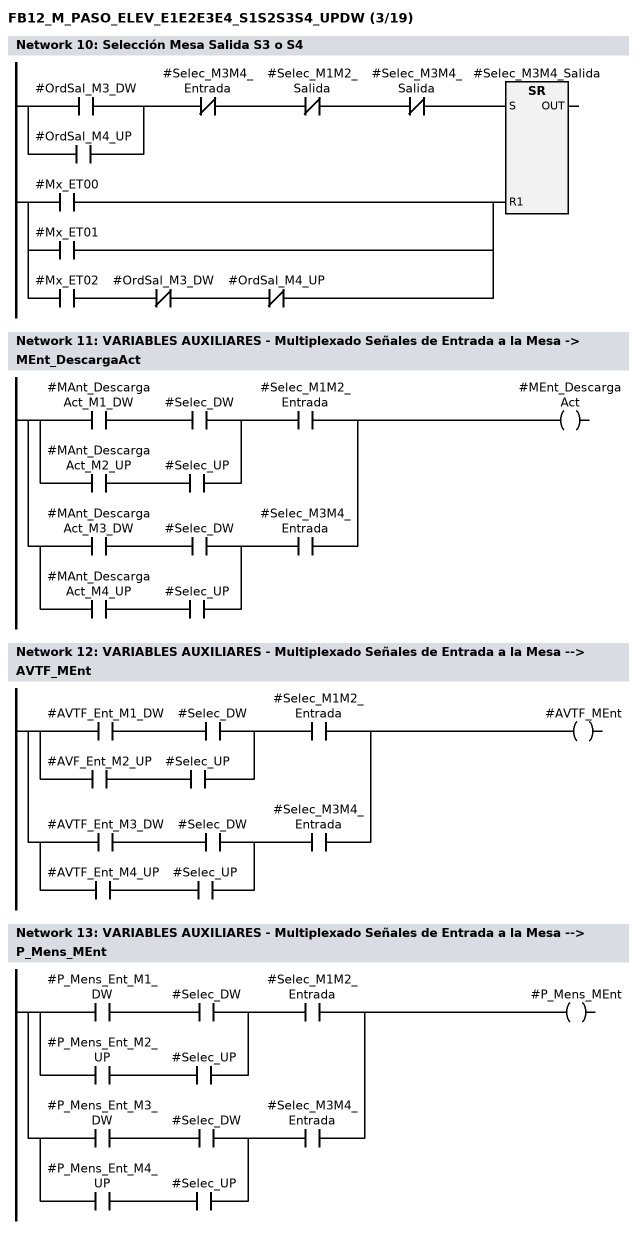
   RUNG wire#powerrail
      Contact( #OrdSal_M3_DW )
      wire#w1
      I_Contact( #Selec_M3M4_Entrada )
      I_Contact( #Selec_M1M2_Salida )
      I_Contact( #Selec_M3M4_Salida )
      S_SR(operand := #Selec_M3M4_Salida, r1 := wire#w2)
   END_RUNG
   RUNG wire#powerrail
      Contact( #OrdSal_M4_UP )
   END_RUNG wire#w1
   RUNG wire#powerrail
      Contact( #Mx_ET00 )
   END_RUNG wire#w2
   RUNG wire#powerrail
      Contact( #Mx_ET01 )
   END_RUNG wire#w2
   RUNG wire#powerrail
      Contact( #Mx_ET02 )
      I_Contact( #OrdSal_M3_DW )
      I_Contact( #OrdSal_M4_UP )
   END_RUNG wire#w2
   // the same network as SCL:
   IF (#OrdSal_M3_DW OR #OrdSal_M4_UP) AND NOT #Selec_M3M4_Entrada AND NOT #Selec_M1M2_Salida AND NOT #Selec_M3M4_Salida THEN
       #Selec_M3M4_Salida := TRUE;   // SR flip-flop
   END_IF;
   IF #Mx_ET00 OR #Mx_ET01 OR (#Mx_ET02 AND NOT #OrdSal_M3_DW AND NOT #OrdSal_M4_UP) THEN
       #Selec_M3M4_Salida := FALSE;
   END_IF;
END_REGION

REGION Network 11: VARIABLES AUXILIARES - Multiplexado Señales de Entrada a la Mesa -> MEnt_DescargaAct
   RUNG wire#powerrail
      Contact( #MAnt_DescargaAct_M1_DW )
      Contact( #Selec_DW )
      wire#w1
      Contact( #Selec_M1M2_Entrada )
      wire#w2
      Coil( #MEnt_DescargaAct )
   END_RUNG
   RUNG wire#powerrail
      Contact( #MAnt_DescargaAct_M2_UP )
      Contact( #Selec_UP )
   END_RUNG wire#w1
   RUNG wire#powerrail
      Contact( #MAnt_DescargaAct_M3_DW )
      Contact( #Selec_DW )
      wire#w3
      Contact( #Selec_M3M4_Entrada )
   END_RUNG wire#w2
   RUNG wire#powerrail
      Contact( #MAnt_DescargaAct_M4_UP )
      Contact( #Selec_UP )
   END_RUNG wire#w3
   // the same network as SCL:
   #MEnt_DescargaAct := (((#MAnt_DescargaAct_M1_DW AND #Selec_DW) OR (#MAnt_DescargaAct_M2_UP AND #Selec_UP)) AND #Selec_M1M2_Entrada) OR (((#MAnt_DescargaAct_M3_DW AND #Selec_DW) OR (#MAnt_DescargaAct_M4_UP AND #Selec_UP)) AND #Selec_M3M4_Entrada);
END_REGION

REGION Network 12: VARIABLES AUXILIARES - Multiplexado Señales de Entrada a la Mesa --> AVTF_MEnt
   RUNG wire#powerrail
      Contact( #AVTF_Ent_M1_DW )
      Contact( #Selec_DW )
      wire#w1
      Contact( #Selec_M1M2_Entrada )
      wire#w2
      Coil( #AVTF_MEnt )
   END_RUNG
   RUNG wire#powerrail
      Contact( #AVF_Ent_M2_UP )
      Contact( #Selec_UP )
   END_RUNG wire#w1
   RUNG wire#powerrail
      Contact( #AVTF_Ent_M3_DW )
      Contact( #Selec_DW )
      wire#w3
      Contact( #Selec_M3M4_Entrada )
   END_RUNG wire#w2
   RUNG wire#powerrail
      Contact( #AVTF_Ent_M4_UP )
      Contact( #Selec_UP )
   END_RUNG wire#w3
   // the same network as SCL:
   #AVTF_MEnt := (((#AVTF_Ent_M1_DW AND #Selec_DW) OR (#AVF_Ent_M2_UP AND #Selec_UP)) AND #Selec_M1M2_Entrada) OR (((#AVTF_Ent_M3_DW AND #Selec_DW) OR (#AVTF_Ent_M4_UP AND #Selec_UP)) AND #Selec_M3M4_Entrada);
END_REGION

REGION Network 13: VARIABLES AUXILIARES - Multiplexado Señales de Entrada a la Mesa --> P_Mens_MEnt
   RUNG wire#powerrail
      Contact( #P_Mens_Ent_M1_DW )
      Contact( #Selec_DW )
      wire#w1
      Contact( #Selec_M1M2_Entrada )
      wire#w2
      Coil( #P_Mens_MEnt )
   END_RUNG
   RUNG wire#powerrail
      Contact( #P_Mens_Ent_M2_UP )
      Contact( #Selec_UP )
   END_RUNG wire#w1
   RUNG wire#powerrail
      Contact( #P_Mens_Ent_M3_DW )
      Contact( #Selec_DW )
      wire#w3
      Contact( #Selec_M3M4_Entrada )
   END_RUNG wire#w2
   RUNG wire#powerrail
      Contact( #P_Mens_Ent_M4_UP )
      Contact( #Selec_UP )
   END_RUNG wire#w3
   // the same network as SCL:
   #P_Mens_MEnt := (((#P_Mens_Ent_M1_DW AND #Selec_DW) OR (#P_Mens_Ent_M2_UP AND #Selec_UP)) AND #Selec_M1M2_Entrada) OR (((#P_Mens_Ent_M3_DW AND #Selec_DW) OR (#P_Mens_Ent_M4_UP AND #Selec_UP)) AND #Selec_M3M4_Entrada);
END_REGION

REGION Network 14: VARIABLES AUXILIARES - Multiplexado Señales de Salida de la Mesa--> PTF_MSal
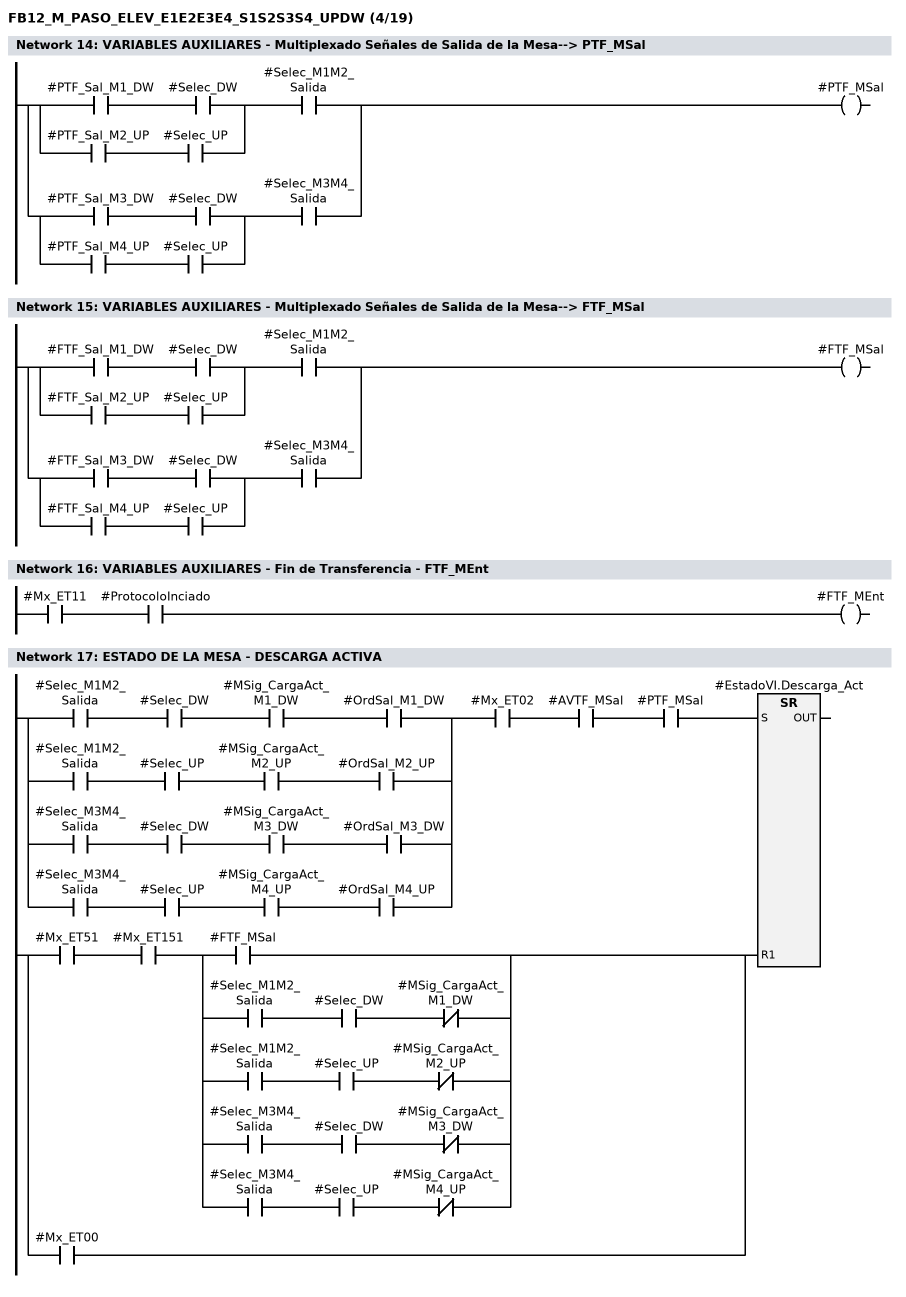
   RUNG wire#powerrail
      Contact( #PTF_Sal_M1_DW )
      Contact( #Selec_DW )
      wire#w1
      Contact( #Selec_M1M2_Salida )
      wire#w2
      Coil( #PTF_MSal )
   END_RUNG
   RUNG wire#powerrail
      Contact( #PTF_Sal_M2_UP )
      Contact( #Selec_UP )
   END_RUNG wire#w1
   RUNG wire#powerrail
      Contact( #PTF_Sal_M3_DW )
      Contact( #Selec_DW )
      wire#w3
      Contact( #Selec_M3M4_Salida )
   END_RUNG wire#w2
   RUNG wire#powerrail
      Contact( #PTF_Sal_M4_UP )
      Contact( #Selec_UP )
   END_RUNG wire#w3
   // the same network as SCL:
   #PTF_MSal := (((#PTF_Sal_M1_DW AND #Selec_DW) OR (#PTF_Sal_M2_UP AND #Selec_UP)) AND #Selec_M1M2_Salida) OR (((#PTF_Sal_M3_DW AND #Selec_DW) OR (#PTF_Sal_M4_UP AND #Selec_UP)) AND #Selec_M3M4_Salida);
END_REGION

REGION Network 15: VARIABLES AUXILIARES - Multiplexado Señales de Salida de la Mesa--> FTF_MSal
   RUNG wire#powerrail
      Contact( #FTF_Sal_M1_DW )
      Contact( #Selec_DW )
      wire#w1
      Contact( #Selec_M1M2_Salida )
      wire#w2
      Coil( #FTF_MSal )
   END_RUNG
   RUNG wire#powerrail
      Contact( #FTF_Sal_M2_UP )
      Contact( #Selec_UP )
   END_RUNG wire#w1
   RUNG wire#powerrail
      Contact( #FTF_Sal_M3_DW )
      Contact( #Selec_DW )
      wire#w3
      Contact( #Selec_M3M4_Salida )
   END_RUNG wire#w2
   RUNG wire#powerrail
      Contact( #FTF_Sal_M4_UP )
      Contact( #Selec_UP )
   END_RUNG wire#w3
   // the same network as SCL:
   #FTF_MSal := (((#FTF_Sal_M1_DW AND #Selec_DW) OR (#FTF_Sal_M2_UP AND #Selec_UP)) AND #Selec_M1M2_Salida) OR (((#FTF_Sal_M3_DW AND #Selec_DW) OR (#FTF_Sal_M4_UP AND #Selec_UP)) AND #Selec_M3M4_Salida);
END_REGION

REGION Network 16: VARIABLES AUXILIARES - Fin de Transferencia - FTF_MEnt
   RUNG wire#powerrail
      Contact( #Mx_ET11 )
      Contact( #ProtocoloInciado )
      Coil( #FTF_MEnt )
   END_RUNG
   // the same network as SCL:
   #FTF_MEnt := #Mx_ET11 AND #ProtocoloInciado;
END_REGION

REGION Network 17: ESTADO DE LA MESA - DESCARGA ACTIVA
   RUNG wire#powerrail
      Contact( #Selec_M1M2_Salida )
      Contact( #Selec_DW )
      Contact( #MSig_CargaAct_M1_DW )
      Contact( #OrdSal_M1_DW )
      wire#w1
      Contact( #Mx_ET02 )
      Contact( #AVTF_MSal )
      Contact( #PTF_MSal )
      S_SR(operand := #EstadoVI.Descarga_Act, r1 := wire#w3)
   END_RUNG
   RUNG wire#powerrail
      Contact( #Selec_M1M2_Salida )
      Contact( #Selec_UP )
      Contact( #MSig_CargaAct_M2_UP )
      Contact( #OrdSal_M2_UP )
   END_RUNG wire#w1
   RUNG wire#powerrail
      Contact( #Selec_M3M4_Salida )
      Contact( #Selec_DW )
      Contact( #MSig_CargaAct_M3_DW )
      Contact( #OrdSal_M3_DW )
   END_RUNG wire#w1
   RUNG wire#powerrail
      Contact( #Selec_M3M4_Salida )
      Contact( #Selec_UP )
      Contact( #MSig_CargaAct_M4_UP )
      Contact( #OrdSal_M4_UP )
   END_RUNG wire#w1
   RUNG wire#powerrail
      Contact( #Mx_ET51 )
      Contact( #Mx_ET151 )
      wire#w2
      Contact( #FTF_MSal )
   END_RUNG wire#w3
   RUNG wire#w2
      Contact( #Selec_M1M2_Salida )
      Contact( #Selec_DW )
      I_Contact( #MSig_CargaAct_M1_DW )
   END_RUNG wire#w3
   RUNG wire#w2
      Contact( #Selec_M1M2_Salida )
      Contact( #Selec_UP )
      I_Contact( #MSig_CargaAct_M2_UP )
   END_RUNG wire#w3
   RUNG wire#w2
      Contact( #Selec_M3M4_Salida )
      Contact( #Selec_DW )
      I_Contact( #MSig_CargaAct_M3_DW )
   END_RUNG wire#w3
   RUNG wire#w2
      Contact( #Selec_M3M4_Salida )
      Contact( #Selec_UP )
      I_Contact( #MSig_CargaAct_M4_UP )
   END_RUNG wire#w3
   RUNG wire#powerrail
      Contact( #Mx_ET00 )
   END_RUNG wire#w3
   // the same network as SCL:
   IF ((#Selec_M1M2_Salida AND #Selec_DW AND #MSig_CargaAct_M1_DW AND #OrdSal_M1_DW) OR (#Selec_M1M2_Salida AND #Selec_UP AND #MSig_CargaAct_M2_UP AND #OrdSal_M2_UP) OR (#Selec_M3M4_Salida AND #Selec_DW AND #MSig_CargaAct_M3_DW AND #OrdSal_M3_DW) OR (#Selec_M3M4_Salida AND #Selec_UP AND #MSig_CargaAct_M4_UP AND #OrdSal_M4_UP)) AND #Mx_ET02 AND #AVTF_MSal AND #PTF_MSal THEN
       #EstadoVI.Descarga_Act := TRUE;   // SR flip-flop
   END_IF;
   IF (#Mx_ET51 AND #Mx_ET151 AND (#FTF_MSal OR (#Selec_M1M2_Salida AND #Selec_DW AND NOT #MSig_CargaAct_M1_DW) OR (#Selec_M1M2_Salida AND #Selec_UP AND NOT #MSig_CargaAct_M2_UP) OR (#Selec_M3M4_Salida AND #Selec_DW AND NOT #MSig_CargaAct_M3_DW) OR (#Selec_M3M4_Salida AND #Selec_UP AND NOT #MSig_CargaAct_M4_UP))) OR #Mx_ET00 THEN
       #EstadoVI.Descarga_Act := FALSE;
   END_IF;
END_REGION

REGION Network 18: ET151 - CONTROL DESCARGA MESA - PROTOCOLO ORDEN
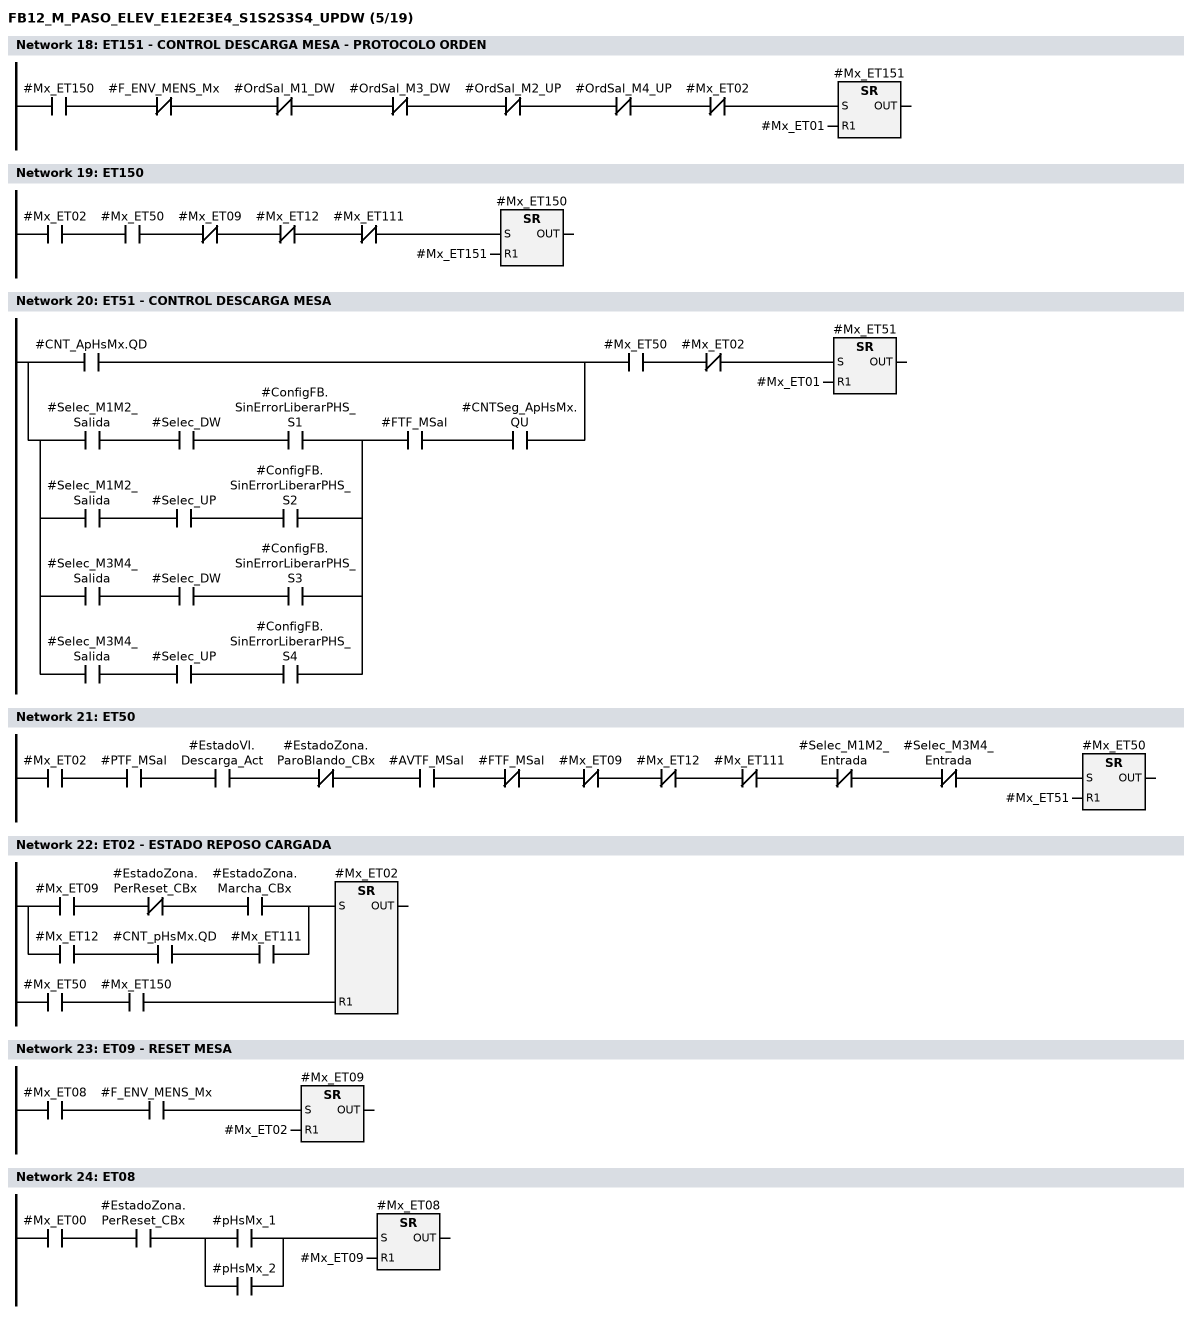
   RUNG wire#powerrail
      Contact( #Mx_ET150 )
      I_Contact( #F_ENV_MENS_Mx )
      I_Contact( #OrdSal_M1_DW )
      I_Contact( #OrdSal_M3_DW )
      I_Contact( #OrdSal_M2_UP )
      I_Contact( #OrdSal_M4_UP )
      I_Contact( #Mx_ET02 )
      S_SR(operand := #Mx_ET151, r1 := #Mx_ET01)
   END_RUNG
   // the same network as SCL:
   IF #Mx_ET150 AND NOT #F_ENV_MENS_Mx AND NOT #OrdSal_M1_DW AND NOT #OrdSal_M3_DW AND NOT #OrdSal_M2_UP AND NOT #OrdSal_M4_UP AND NOT #Mx_ET02 THEN
       #Mx_ET151 := TRUE;   // SR flip-flop
   END_IF;
   IF #Mx_ET01 THEN #Mx_ET151 := FALSE; END_IF;
END_REGION

REGION Network 19: ET150
   RUNG wire#powerrail
      Contact( #Mx_ET02 )
      Contact( #Mx_ET50 )
      I_Contact( #Mx_ET09 )
      I_Contact( #Mx_ET12 )
      I_Contact( #Mx_ET111 )
      S_SR(operand := #Mx_ET150, r1 := #Mx_ET151)
   END_RUNG
   // the same network as SCL:
   IF #Mx_ET02 AND #Mx_ET50 AND NOT #Mx_ET09 AND NOT #Mx_ET12 AND NOT #Mx_ET111 THEN
       #Mx_ET150 := TRUE;   // SR flip-flop
   END_IF;
   IF #Mx_ET151 THEN #Mx_ET150 := FALSE; END_IF;
END_REGION

REGION Network 20: ET51 - CONTROL DESCARGA MESA
   RUNG wire#powerrail
      Contact( #CNT_ApHsMx.QD )
      wire#w1
      Contact( #Mx_ET50 )
      I_Contact( #Mx_ET02 )
      S_SR(operand := #Mx_ET51, r1 := #Mx_ET01)
   END_RUNG
   RUNG wire#powerrail
      Contact( #Selec_M1M2_Salida )
      Contact( #Selec_DW )
      Contact( #ConfigFB.SinErrorLiberarPHS_S1 )
      wire#w2
      Contact( #FTF_MSal )
      Contact( #CNTSeg_ApHsMx.QU )
   END_RUNG wire#w1
   RUNG wire#powerrail
      Contact( #Selec_M1M2_Salida )
      Contact( #Selec_UP )
      Contact( #ConfigFB.SinErrorLiberarPHS_S2 )
   END_RUNG wire#w2
   RUNG wire#powerrail
      Contact( #Selec_M3M4_Salida )
      Contact( #Selec_DW )
      Contact( #ConfigFB.SinErrorLiberarPHS_S3 )
   END_RUNG wire#w2
   RUNG wire#powerrail
      Contact( #Selec_M3M4_Salida )
      Contact( #Selec_UP )
      Contact( #ConfigFB.SinErrorLiberarPHS_S4 )
   END_RUNG wire#w2
   // the same network as SCL:
   IF (#CNT_ApHsMx.QD OR (((#Selec_M1M2_Salida AND #Selec_DW AND #ConfigFB.SinErrorLiberarPHS_S1) OR (#Selec_M1M2_Salida AND #Selec_UP AND #ConfigFB.SinErrorLiberarPHS_S2) OR (#Selec_M3M4_Salida AND #Selec_DW AND #ConfigFB.SinErrorLiberarPHS_S3) OR (#Selec_M3M4_Salida AND #Selec_UP AND #ConfigFB.SinErrorLiberarPHS_S4)) AND #FTF_MSal AND #CNTSeg_ApHsMx.QU)) AND #Mx_ET50 AND NOT #Mx_ET02 THEN
       #Mx_ET51 := TRUE;   // SR flip-flop
   END_IF;
   IF #Mx_ET01 THEN #Mx_ET51 := FALSE; END_IF;
END_REGION

REGION Network 21: ET50
   RUNG wire#powerrail
      Contact( #Mx_ET02 )
      Contact( #PTF_MSal )
      Contact( #EstadoVI.Descarga_Act )
      I_Contact( #EstadoZona.ParoBlando_CBx )
      Contact( #AVTF_MSal )
      I_Contact( #FTF_MSal )
      I_Contact( #Mx_ET09 )
      I_Contact( #Mx_ET12 )
      I_Contact( #Mx_ET111 )
      I_Contact( #Selec_M1M2_Entrada )
      I_Contact( #Selec_M3M4_Entrada )
      S_SR(operand := #Mx_ET50, r1 := #Mx_ET51)
   END_RUNG
   // the same network as SCL:
   IF #Mx_ET02 AND #PTF_MSal AND #EstadoVI.Descarga_Act AND NOT #EstadoZona.ParoBlando_CBx AND #AVTF_MSal AND NOT #FTF_MSal AND NOT #Mx_ET09 AND NOT #Mx_ET12 AND NOT #Mx_ET111 AND NOT #Selec_M1M2_Entrada AND NOT #Selec_M3M4_Entrada THEN
       #Mx_ET50 := TRUE;   // SR flip-flop
   END_IF;
   IF #Mx_ET51 THEN #Mx_ET50 := FALSE; END_IF;
END_REGION

REGION Network 22: ET02 - ESTADO REPOSO CARGADA
   RUNG wire#powerrail
      Contact( #Mx_ET09 )
      I_Contact( #EstadoZona.PerReset_CBx )
      Contact( #EstadoZona.Marcha_CBx )
      wire#w1
      S_SR(operand := #Mx_ET02, r1 := wire#w2)
   END_RUNG
   RUNG wire#powerrail
      Contact( #Mx_ET12 )
      Contact( #CNT_pHsMx.QD )
      Contact( #Mx_ET111 )
   END_RUNG wire#w1
   RUNG wire#powerrail
      Contact( #Mx_ET50 )
      Contact( #Mx_ET150 )
   END_RUNG wire#w2
   // the same network as SCL:
   IF (#Mx_ET09 AND NOT #EstadoZona.PerReset_CBx AND #EstadoZona.Marcha_CBx) OR (#Mx_ET12 AND #CNT_pHsMx.QD AND #Mx_ET111) THEN
       #Mx_ET02 := TRUE;   // SR flip-flop
   END_IF;
   IF #Mx_ET50 AND #Mx_ET150 THEN #Mx_ET02 := FALSE; END_IF;
END_REGION

REGION Network 23: ET09 - RESET MESA
   RUNG wire#powerrail
      Contact( #Mx_ET08 )
      Contact( #F_ENV_MENS_Mx )
      S_SR(operand := #Mx_ET09, r1 := #Mx_ET02)
   END_RUNG
   // the same network as SCL:
   IF #Mx_ET08 AND #F_ENV_MENS_Mx THEN
       #Mx_ET09 := TRUE;   // SR flip-flop
   END_IF;
   IF #Mx_ET02 THEN #Mx_ET09 := FALSE; END_IF;
END_REGION

REGION Network 24: ET08
   RUNG wire#powerrail
      Contact( #Mx_ET00 )
      Contact( #EstadoZona.PerReset_CBx )
      wire#w1
      Contact( #pHsMx_1 )
      wire#w2
      S_SR(operand := #Mx_ET08, r1 := #Mx_ET09)
   END_RUNG
   RUNG wire#w1
      Contact( #pHsMx_2 )
   END_RUNG wire#w2
   // the same network as SCL:
   IF #Mx_ET00 AND #EstadoZona.PerReset_CBx AND (#pHsMx_1 OR #pHsMx_2) THEN
       #Mx_ET08 := TRUE;   // SR flip-flop
   END_IF;
   IF #Mx_ET09 THEN #Mx_ET08 := FALSE; END_IF;
END_REGION

REGION Network 25: ET111 - CONTROL CARGA MESA - MENSAJE DE PRESENCIA
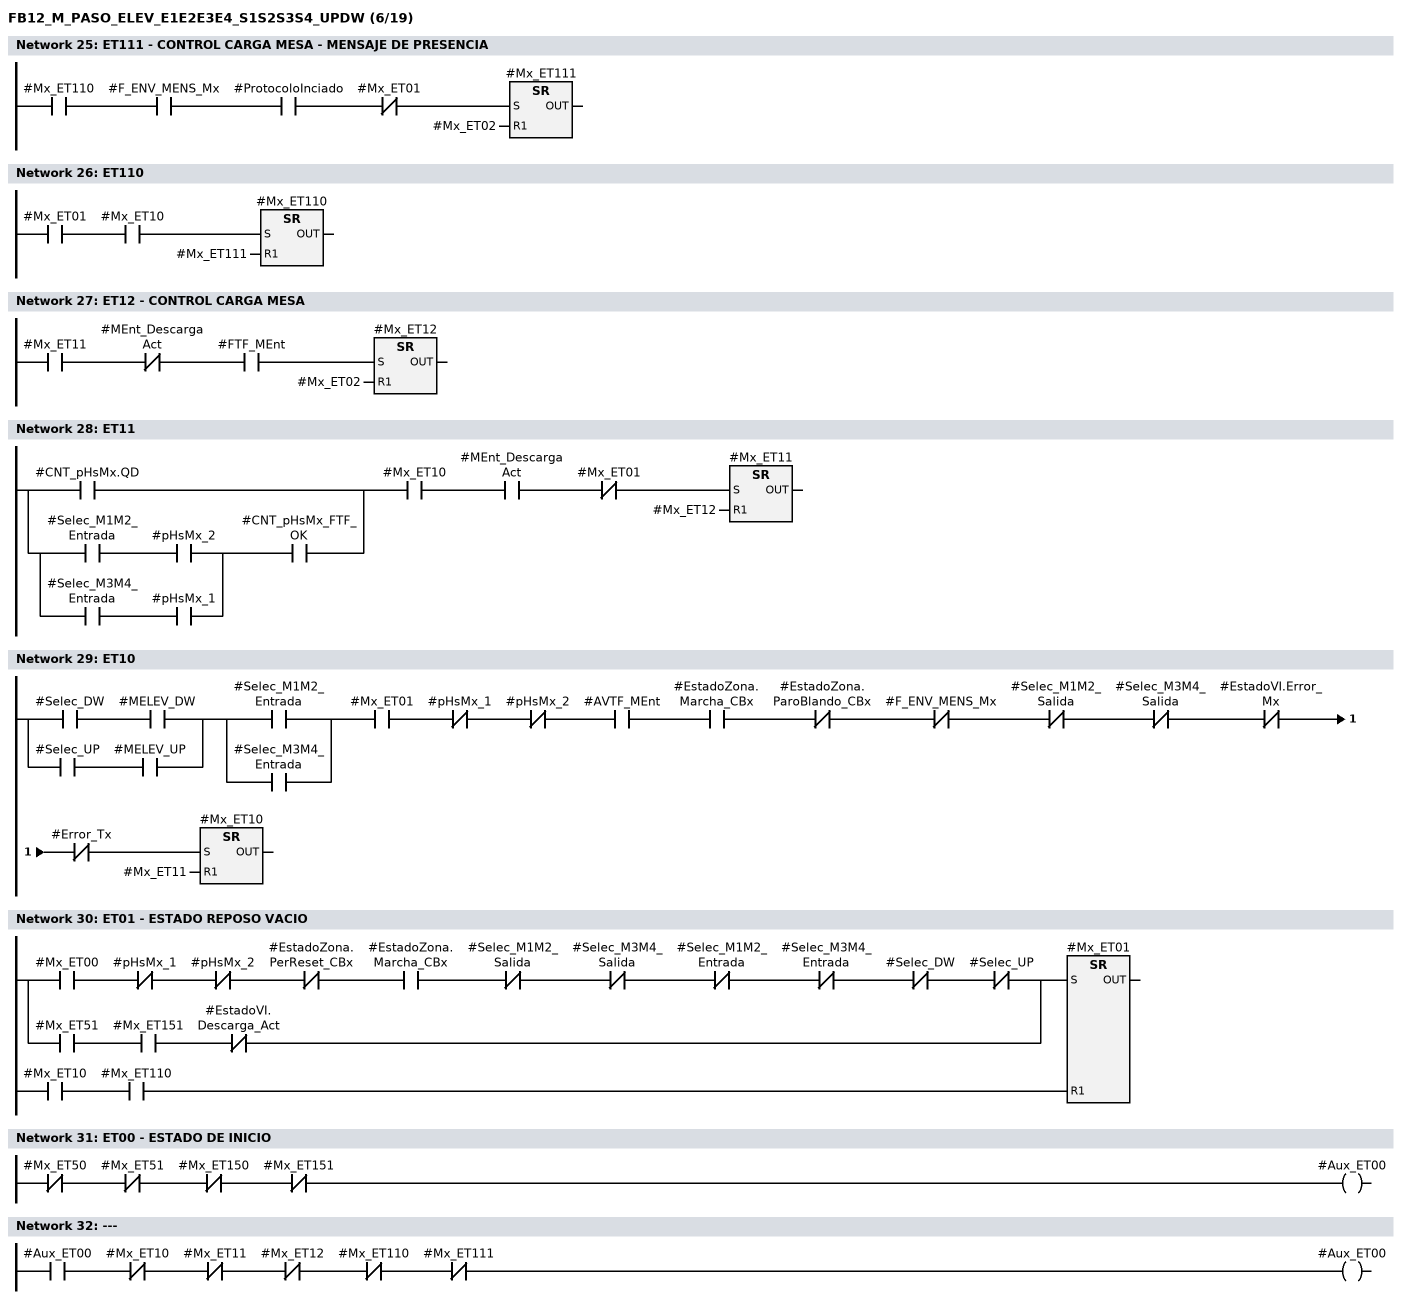
   RUNG wire#powerrail
      Contact( #Mx_ET110 )
      Contact( #F_ENV_MENS_Mx )
      Contact( #ProtocoloInciado )
      I_Contact( #Mx_ET01 )
      S_SR(operand := #Mx_ET111, r1 := #Mx_ET02)
   END_RUNG
   // the same network as SCL:
   IF #Mx_ET110 AND #F_ENV_MENS_Mx AND #ProtocoloInciado AND NOT #Mx_ET01 THEN
       #Mx_ET111 := TRUE;   // SR flip-flop
   END_IF;
   IF #Mx_ET02 THEN #Mx_ET111 := FALSE; END_IF;
END_REGION

REGION Network 26: ET110
   RUNG wire#powerrail
      Contact( #Mx_ET01 )
      Contact( #Mx_ET10 )
      S_SR(operand := #Mx_ET110, r1 := #Mx_ET111)
   END_RUNG
   // the same network as SCL:
   IF #Mx_ET01 AND #Mx_ET10 THEN
       #Mx_ET110 := TRUE;   // SR flip-flop
   END_IF;
   IF #Mx_ET111 THEN #Mx_ET110 := FALSE; END_IF;
END_REGION

REGION Network 27: ET12 - CONTROL CARGA MESA
   RUNG wire#powerrail
      Contact( #Mx_ET11 )
      I_Contact( #MEnt_DescargaAct )
      Contact( #FTF_MEnt )
      S_SR(operand := #Mx_ET12, r1 := #Mx_ET02)
   END_RUNG
   // the same network as SCL:
   IF #Mx_ET11 AND NOT #MEnt_DescargaAct AND #FTF_MEnt THEN
       #Mx_ET12 := TRUE;   // SR flip-flop
   END_IF;
   IF #Mx_ET02 THEN #Mx_ET12 := FALSE; END_IF;
END_REGION

REGION Network 28: ET11
   RUNG wire#powerrail
      Contact( #CNT_pHsMx.QD )
      wire#w1
      Contact( #Mx_ET10 )
      Contact( #MEnt_DescargaAct )
      I_Contact( #Mx_ET01 )
      S_SR(operand := #Mx_ET11, r1 := #Mx_ET12)
   END_RUNG
   RUNG wire#powerrail
      Contact( #Selec_M1M2_Entrada )
      Contact( #pHsMx_2 )
      wire#w2
      Contact( #CNT_pHsMx_FTF_OK )
   END_RUNG wire#w1
   RUNG wire#powerrail
      Contact( #Selec_M3M4_Entrada )
      Contact( #pHsMx_1 )
   END_RUNG wire#w2
   // the same network as SCL:
   IF (#CNT_pHsMx.QD OR (((#Selec_M1M2_Entrada AND #pHsMx_2) OR (#Selec_M3M4_Entrada AND #pHsMx_1)) AND #CNT_pHsMx_FTF_OK)) AND #Mx_ET10 AND #MEnt_DescargaAct AND NOT #Mx_ET01 THEN
       #Mx_ET11 := TRUE;   // SR flip-flop
   END_IF;
   IF #Mx_ET12 THEN #Mx_ET11 := FALSE; END_IF;
END_REGION

REGION Network 29: ET10
   RUNG wire#powerrail
      Contact( #Selec_DW )
      Contact( #MELEV_DW )
      wire#w1
      Contact( #Selec_M1M2_Entrada )
      wire#w2
      Contact( #Mx_ET01 )
      I_Contact( #pHsMx_1 )
      I_Contact( #pHsMx_2 )
      Contact( #AVTF_MEnt )
      Contact( #EstadoZona.Marcha_CBx )
      I_Contact( #EstadoZona.ParoBlando_CBx )
      I_Contact( #F_ENV_MENS_Mx )
      I_Contact( #Selec_M1M2_Salida )
      I_Contact( #Selec_M3M4_Salida )
      I_Contact( #EstadoVI.Error_Mx )
      I_Contact( #Error_Tx )
      S_SR(operand := #Mx_ET10, r1 := #Mx_ET11)
   END_RUNG
   RUNG wire#powerrail
      Contact( #Selec_UP )
      Contact( #MELEV_UP )
   END_RUNG wire#w1
   RUNG wire#w1
      Contact( #Selec_M3M4_Entrada )
   END_RUNG wire#w2
   // the same network as SCL:
   IF ((#Selec_DW AND #MELEV_DW) OR (#Selec_UP AND #MELEV_UP)) AND (#Selec_M1M2_Entrada OR #Selec_M3M4_Entrada) AND #Mx_ET01 AND NOT #pHsMx_1 AND NOT #pHsMx_2 AND #AVTF_MEnt AND #EstadoZona.Marcha_CBx AND NOT #EstadoZona.ParoBlando_CBx AND NOT #F_ENV_MENS_Mx AND NOT #Selec_M1M2_Salida AND NOT #Selec_M3M4_Salida AND NOT #EstadoVI.Error_Mx AND NOT #Error_Tx THEN
       #Mx_ET10 := TRUE;   // SR flip-flop
   END_IF;
   IF #Mx_ET11 THEN #Mx_ET10 := FALSE; END_IF;
END_REGION

REGION Network 30: ET01 - ESTADO REPOSO VACIO
   RUNG wire#powerrail
      Contact( #Mx_ET00 )
      I_Contact( #pHsMx_1 )
      I_Contact( #pHsMx_2 )
      I_Contact( #EstadoZona.PerReset_CBx )
      Contact( #EstadoZona.Marcha_CBx )
      I_Contact( #Selec_M1M2_Salida )
      I_Contact( #Selec_M3M4_Salida )
      I_Contact( #Selec_M1M2_Entrada )
      I_Contact( #Selec_M3M4_Entrada )
      I_Contact( #Selec_DW )
      I_Contact( #Selec_UP )
      wire#w1
      S_SR(operand := #Mx_ET01, r1 := wire#w2)
   END_RUNG
   RUNG wire#powerrail
      Contact( #Mx_ET51 )
      Contact( #Mx_ET151 )
      I_Contact( #EstadoVI.Descarga_Act )
   END_RUNG wire#w1
   RUNG wire#powerrail
      Contact( #Mx_ET10 )
      Contact( #Mx_ET110 )
   END_RUNG wire#w2
   // the same network as SCL:
   IF (#Mx_ET00 AND NOT #pHsMx_1 AND NOT #pHsMx_2 AND NOT #EstadoZona.PerReset_CBx AND #EstadoZona.Marcha_CBx AND NOT #Selec_M1M2_Salida AND NOT #Selec_M3M4_Salida AND NOT #Selec_M1M2_Entrada AND NOT #Selec_M3M4_Entrada AND NOT #Selec_DW AND NOT #Selec_UP) OR (#Mx_ET51 AND #Mx_ET151 AND NOT #EstadoVI.Descarga_Act) THEN
       #Mx_ET01 := TRUE;   // SR flip-flop
   END_IF;
   IF #Mx_ET10 AND #Mx_ET110 THEN #Mx_ET01 := FALSE; END_IF;
END_REGION

REGION Network 31: ET00 - ESTADO DE INICIO
   RUNG wire#powerrail
      I_Contact( #Mx_ET50 )
      I_Contact( #Mx_ET51 )
      I_Contact( #Mx_ET150 )
      I_Contact( #Mx_ET151 )
      Coil( #Aux_ET00 )
   END_RUNG
   // the same network as SCL:
   #Aux_ET00 := NOT #Mx_ET50 AND NOT #Mx_ET51 AND NOT #Mx_ET150 AND NOT #Mx_ET151;
END_REGION

REGION Network 32: ---
   RUNG wire#powerrail
      Contact( #Aux_ET00 )
      I_Contact( #Mx_ET10 )
      I_Contact( #Mx_ET11 )
      I_Contact( #Mx_ET12 )
      I_Contact( #Mx_ET110 )
      I_Contact( #Mx_ET111 )
      Coil( #Aux_ET00 )
   END_RUNG
   // the same network as SCL:
   #Aux_ET00 := #Aux_ET00 AND NOT #Mx_ET10 AND NOT #Mx_ET11 AND NOT #Mx_ET12 AND NOT #Mx_ET110 AND NOT #Mx_ET111;
END_REGION

REGION Network 33: ---
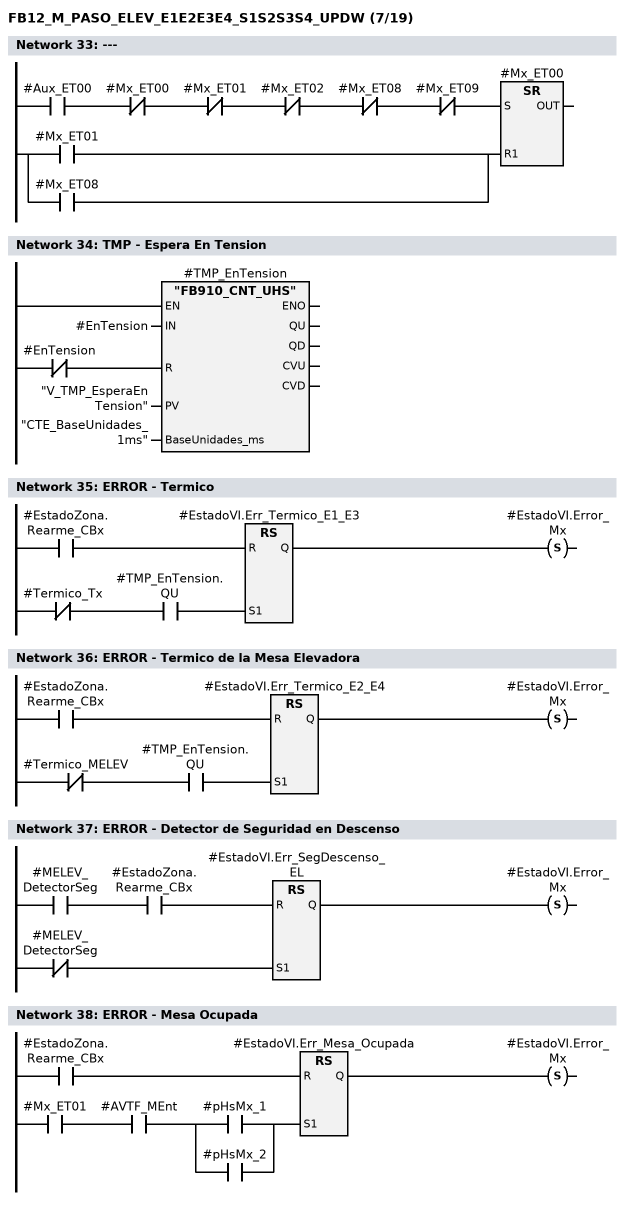
   RUNG wire#powerrail
      Contact( #Aux_ET00 )
      I_Contact( #Mx_ET00 )
      I_Contact( #Mx_ET01 )
      I_Contact( #Mx_ET02 )
      I_Contact( #Mx_ET08 )
      I_Contact( #Mx_ET09 )
      S_SR(operand := #Mx_ET00, r1 := wire#w1)
   END_RUNG
   RUNG wire#powerrail
      Contact( #Mx_ET01 )
   END_RUNG wire#w1
   RUNG wire#powerrail
      Contact( #Mx_ET08 )
   END_RUNG wire#w1
   // the same network as SCL:
   IF #Aux_ET00 AND NOT #Mx_ET00 AND NOT #Mx_ET01 AND NOT #Mx_ET02 AND NOT #Mx_ET08 AND NOT #Mx_ET09 THEN
       #Mx_ET00 := TRUE;   // SR flip-flop
   END_IF;
   IF #Mx_ET01 OR #Mx_ET08 THEN #Mx_ET00 := FALSE; END_IF;
END_REGION

REGION Network 34: TMP - Espera En Tension
   RUNG wire#powerrail
      #TMP_EnTension(R := wire#w1, IN := #EnTension, PV := "V_TMP_EsperaEnTension", BaseUnidades_ms := "CTE_BaseUnidades_1ms", QU =>, QD =>, CVU =>, CVD =>)
   END_RUNG
   RUNG wire#powerrail
      I_Contact( #EnTension )
   END_RUNG wire#w1
   // the same network as SCL:
   #TMP_EnTension(IN := #EnTension,   // "FB910_CNT_UHS"
                  R := NOT #EnTension,
                  PV := "V_TMP_EsperaEnTension",
                  BaseUnidades_ms := "CTE_BaseUnidades_1ms");
END_REGION

REGION Network 35: ERROR - Termico
   RUNG wire#powerrail
      Contact( #EstadoZona.Rearme_CBx )
      S_RS(operand := #EstadoVI.Err_Termico_E1_E3, s1 := wire#w1)
      S_Coil( #EstadoVI.Error_Mx )
   END_RUNG
   RUNG wire#powerrail
      I_Contact( #Termico_Tx )
      Contact( #TMP_EnTension.QU )
   END_RUNG wire#w1
   // the same network as SCL:
   IF #EstadoZona.Rearme_CBx THEN
       #EstadoVI.Err_Termico_E1_E3 := FALSE;   // RS flip-flop
   END_IF;
   IF NOT #Termico_Tx AND #TMP_EnTension.QU THEN #EstadoVI.Err_Termico_E1_E3 := TRUE; END_IF;
   IF #EstadoVI.Err_Termico_E1_E3 THEN #EstadoVI.Error_Mx := TRUE; END_IF;
END_REGION

REGION Network 36: ERROR - Termico de la Mesa Elevadora
   RUNG wire#powerrail
      Contact( #EstadoZona.Rearme_CBx )
      S_RS(operand := #EstadoVI.Err_Termico_E2_E4, s1 := wire#w1)
      S_Coil( #EstadoVI.Error_Mx )
   END_RUNG
   RUNG wire#powerrail
      I_Contact( #Termico_MELEV )
      Contact( #TMP_EnTension.QU )
   END_RUNG wire#w1
   // the same network as SCL:
   IF #EstadoZona.Rearme_CBx THEN
       #EstadoVI.Err_Termico_E2_E4 := FALSE;   // RS flip-flop
   END_IF;
   IF NOT #Termico_MELEV AND #TMP_EnTension.QU THEN #EstadoVI.Err_Termico_E2_E4 := TRUE; END_IF;
   IF #EstadoVI.Err_Termico_E2_E4 THEN #EstadoVI.Error_Mx := TRUE; END_IF;
END_REGION

REGION Network 37: ERROR - Detector de Seguridad en Descenso
   RUNG wire#powerrail
      Contact( #MELEV_DetectorSeg )
      Contact( #EstadoZona.Rearme_CBx )
      S_RS(operand := #EstadoVI.Err_SegDescenso_EL, s1 := wire#w1)
      S_Coil( #EstadoVI.Error_Mx )
   END_RUNG
   RUNG wire#powerrail
      I_Contact( #MELEV_DetectorSeg )
   END_RUNG wire#w1
   // the same network as SCL:
   IF #MELEV_DetectorSeg AND #EstadoZona.Rearme_CBx THEN
       #EstadoVI.Err_SegDescenso_EL := FALSE;   // RS flip-flop
   END_IF;
   IF NOT #MELEV_DetectorSeg THEN #EstadoVI.Err_SegDescenso_EL := TRUE; END_IF;
   IF #EstadoVI.Err_SegDescenso_EL THEN #EstadoVI.Error_Mx := TRUE; END_IF;
END_REGION

REGION Network 38: ERROR - Mesa Ocupada
   RUNG wire#powerrail
      Contact( #EstadoZona.Rearme_CBx )
      S_RS(operand := #EstadoVI.Err_Mesa_Ocupada, s1 := wire#w2)
      S_Coil( #EstadoVI.Error_Mx )
   END_RUNG
   RUNG wire#powerrail
      Contact( #Mx_ET01 )
      Contact( #AVTF_MEnt )
      wire#w1
      Contact( #pHsMx_1 )
   END_RUNG wire#w2
   RUNG wire#w1
      Contact( #pHsMx_2 )
   END_RUNG wire#w2
   // the same network as SCL:
   IF #EstadoZona.Rearme_CBx THEN
       #EstadoVI.Err_Mesa_Ocupada := FALSE;   // RS flip-flop
   END_IF;
   IF #Mx_ET01 AND #AVTF_MEnt AND (#pHsMx_1 OR #pHsMx_2) THEN #EstadoVI.Err_Mesa_Ocupada := TRUE; END_IF;
   IF #EstadoVI.Err_Mesa_Ocupada THEN #EstadoVI.Error_Mx := TRUE; END_IF;
END_REGION

REGION Network 39: CNT - ERROR - Arrastre
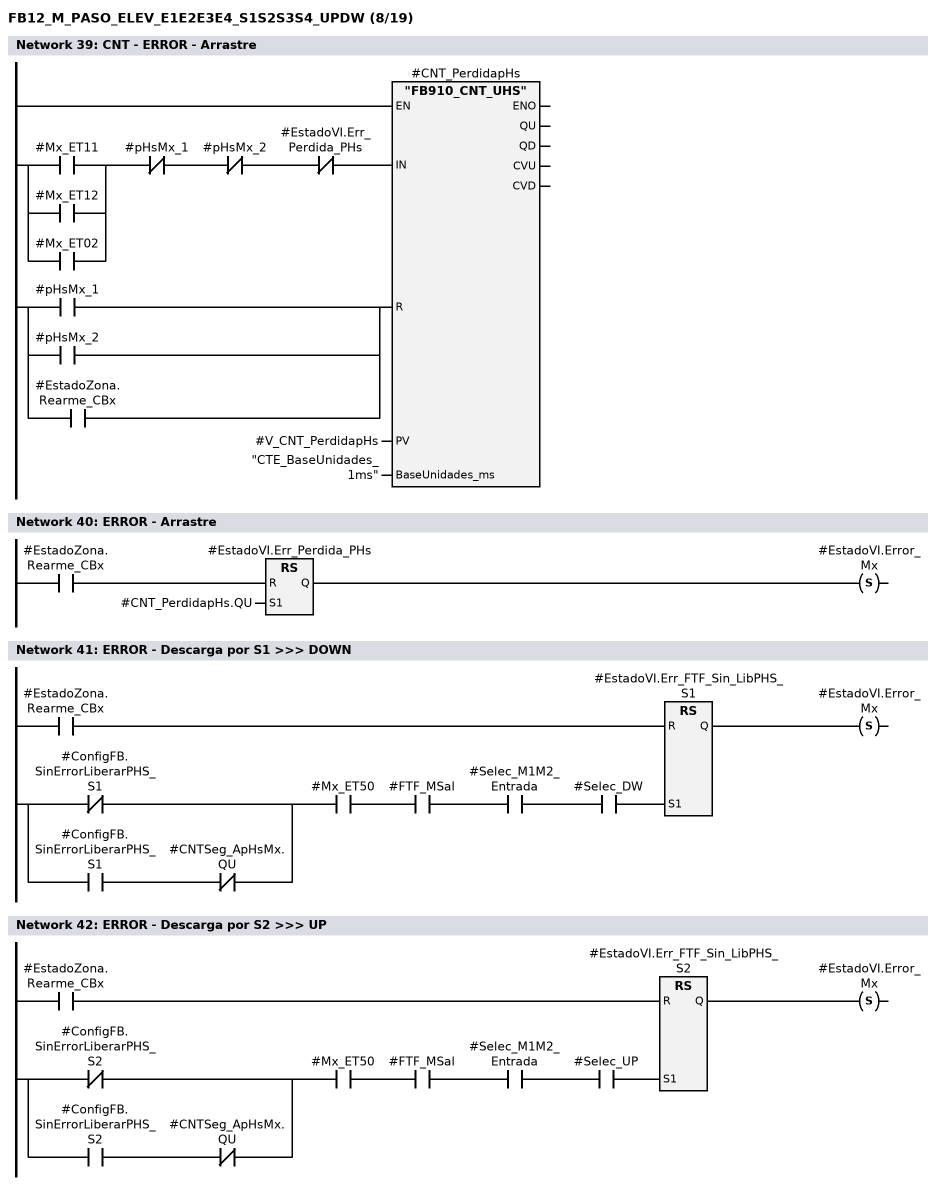
   RUNG wire#powerrail
      #CNT_PerdidapHs(IN := wire#w2, R := wire#w3, PV := #V_CNT_PerdidapHs, BaseUnidades_ms := "CTE_BaseUnidades_1ms", QU =>, QD =>, CVU =>, CVD =>)
   END_RUNG
   RUNG wire#powerrail
      Contact( #Mx_ET11 )
      wire#w1
      I_Contact( #pHsMx_1 )
      I_Contact( #pHsMx_2 )
      I_Contact( #EstadoVI.Err_Perdida_PHs )
   END_RUNG wire#w2
   RUNG wire#powerrail
      Contact( #Mx_ET12 )
   END_RUNG wire#w1
   RUNG wire#powerrail
      Contact( #Mx_ET02 )
   END_RUNG wire#w1
   RUNG wire#powerrail
      Contact( #pHsMx_1 )
   END_RUNG wire#w3
   RUNG wire#powerrail
      Contact( #pHsMx_2 )
   END_RUNG wire#w3
   RUNG wire#powerrail
      Contact( #EstadoZona.Rearme_CBx )
   END_RUNG wire#w3
   // the same network as SCL:
   #CNT_PerdidapHs(IN := (#Mx_ET11 OR #Mx_ET12 OR #Mx_ET02) AND NOT #pHsMx_1 AND NOT #pHsMx_2 AND NOT #EstadoVI.Err_Perdida_PHs,   // "FB910_CNT_UHS"
                   R := #pHsMx_1 OR #pHsMx_2 OR #EstadoZona.Rearme_CBx,
                   PV := #V_CNT_PerdidapHs,
                   BaseUnidades_ms := "CTE_BaseUnidades_1ms");
END_REGION

REGION Network 40: ERROR - Arrastre
   RUNG wire#powerrail
      Contact( #EstadoZona.Rearme_CBx )
      S_RS(operand := #EstadoVI.Err_Perdida_PHs, s1 := #CNT_PerdidapHs.QU)
      S_Coil( #EstadoVI.Error_Mx )
   END_RUNG
   // the same network as SCL:
   IF #EstadoZona.Rearme_CBx THEN
       #EstadoVI.Err_Perdida_PHs := FALSE;   // RS flip-flop
   END_IF;
   IF #CNT_PerdidapHs.QU THEN #EstadoVI.Err_Perdida_PHs := TRUE; END_IF;
   IF #EstadoVI.Err_Perdida_PHs THEN #EstadoVI.Error_Mx := TRUE; END_IF;
END_REGION

REGION Network 41: ERROR - Descarga por S1 >>> DOWN
   RUNG wire#powerrail
      Contact( #EstadoZona.Rearme_CBx )
      S_RS(operand := #EstadoVI.Err_FTF_Sin_LibPHS_S1, s1 := wire#w2)
      S_Coil( #EstadoVI.Error_Mx )
   END_RUNG
   RUNG wire#powerrail
      I_Contact( #ConfigFB.SinErrorLiberarPHS_S1 )
      wire#w1
      Contact( #Mx_ET50 )
      Contact( #FTF_MSal )
      Contact( #Selec_M1M2_Entrada )
      Contact( #Selec_DW )
   END_RUNG wire#w2
   RUNG wire#powerrail
      Contact( #ConfigFB.SinErrorLiberarPHS_S1 )
      I_Contact( #CNTSeg_ApHsMx.QU )
   END_RUNG wire#w1
   // the same network as SCL:
   IF #EstadoZona.Rearme_CBx THEN
       #EstadoVI.Err_FTF_Sin_LibPHS_S1 := FALSE;   // RS flip-flop
   END_IF;
   IF (NOT #ConfigFB.SinErrorLiberarPHS_S1 OR (#ConfigFB.SinErrorLiberarPHS_S1 AND NOT #CNTSeg_ApHsMx.QU)) AND #Mx_ET50 AND #FTF_MSal AND #Selec_M1M2_Entrada AND #Selec_DW THEN
       #EstadoVI.Err_FTF_Sin_LibPHS_S1 := TRUE;
   END_IF;
   IF #EstadoVI.Err_FTF_Sin_LibPHS_S1 THEN #EstadoVI.Error_Mx := TRUE; END_IF;
END_REGION

REGION Network 42: ERROR - Descarga por S2 >>> UP
   RUNG wire#powerrail
      Contact( #EstadoZona.Rearme_CBx )
      S_RS(operand := #EstadoVI.Err_FTF_Sin_LibPHS_S2, s1 := wire#w2)
      S_Coil( #EstadoVI.Error_Mx )
   END_RUNG
   RUNG wire#powerrail
      I_Contact( #ConfigFB.SinErrorLiberarPHS_S2 )
      wire#w1
      Contact( #Mx_ET50 )
      Contact( #FTF_MSal )
      Contact( #Selec_M1M2_Entrada )
      Contact( #Selec_UP )
   END_RUNG wire#w2
   RUNG wire#powerrail
      Contact( #ConfigFB.SinErrorLiberarPHS_S2 )
      I_Contact( #CNTSeg_ApHsMx.QU )
   END_RUNG wire#w1
   // the same network as SCL:
   IF #EstadoZona.Rearme_CBx THEN
       #EstadoVI.Err_FTF_Sin_LibPHS_S2 := FALSE;   // RS flip-flop
   END_IF;
   IF (NOT #ConfigFB.SinErrorLiberarPHS_S2 OR (#ConfigFB.SinErrorLiberarPHS_S2 AND NOT #CNTSeg_ApHsMx.QU)) AND #Mx_ET50 AND #FTF_MSal AND #Selec_M1M2_Entrada AND #Selec_UP THEN
       #EstadoVI.Err_FTF_Sin_LibPHS_S2 := TRUE;
   END_IF;
   IF #EstadoVI.Err_FTF_Sin_LibPHS_S2 THEN #EstadoVI.Error_Mx := TRUE; END_IF;
END_REGION

REGION Network 43: ERROR - Descarga por S3 >>> DOWN
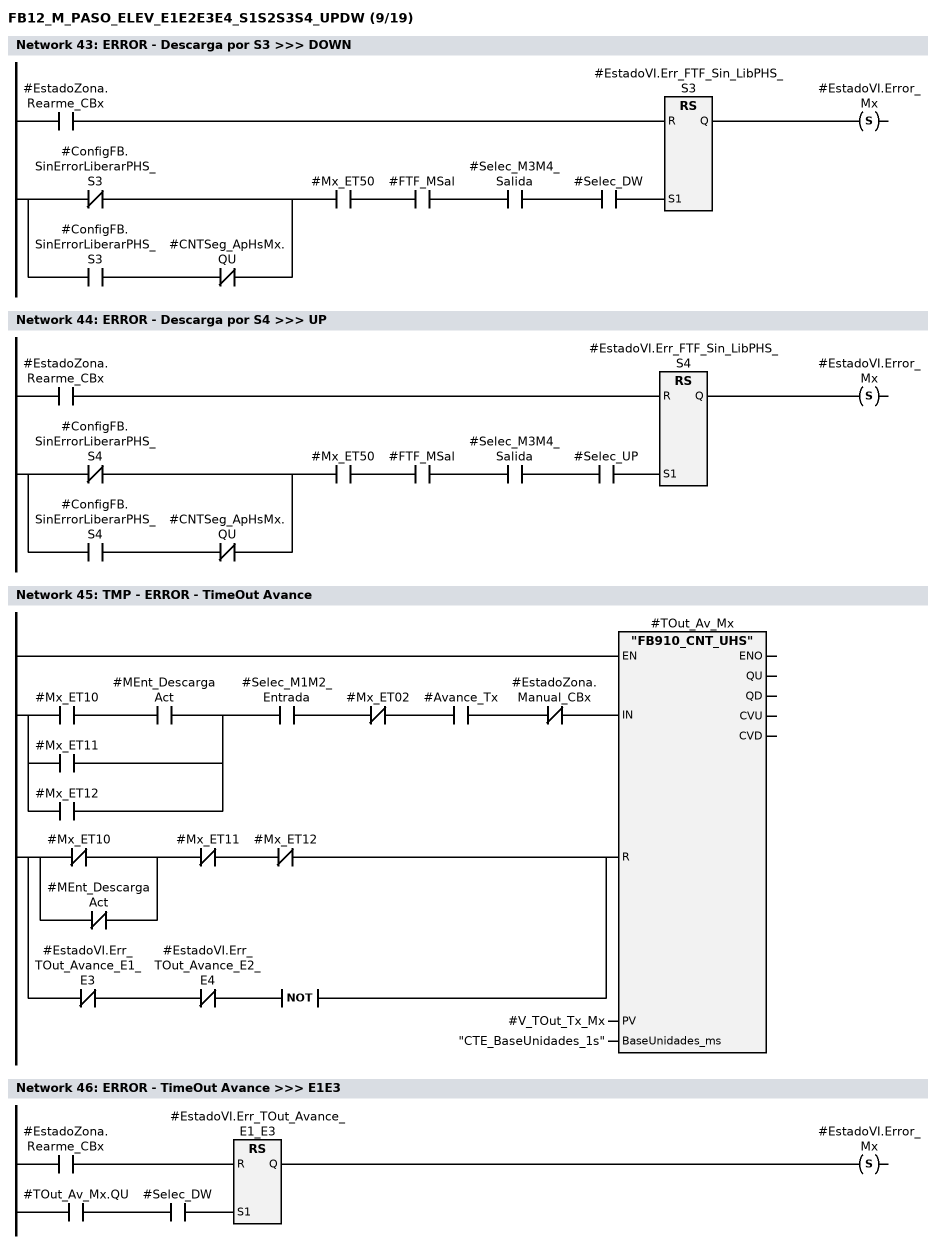
   RUNG wire#powerrail
      Contact( #EstadoZona.Rearme_CBx )
      S_RS(operand := #EstadoVI.Err_FTF_Sin_LibPHS_S3, s1 := wire#w2)
      S_Coil( #EstadoVI.Error_Mx )
   END_RUNG
   RUNG wire#powerrail
      I_Contact( #ConfigFB.SinErrorLiberarPHS_S3 )
      wire#w1
      Contact( #Mx_ET50 )
      Contact( #FTF_MSal )
      Contact( #Selec_M3M4_Salida )
      Contact( #Selec_DW )
   END_RUNG wire#w2
   RUNG wire#powerrail
      Contact( #ConfigFB.SinErrorLiberarPHS_S3 )
      I_Contact( #CNTSeg_ApHsMx.QU )
   END_RUNG wire#w1
   // the same network as SCL:
   IF #EstadoZona.Rearme_CBx THEN
       #EstadoVI.Err_FTF_Sin_LibPHS_S3 := FALSE;   // RS flip-flop
   END_IF;
   IF (NOT #ConfigFB.SinErrorLiberarPHS_S3 OR (#ConfigFB.SinErrorLiberarPHS_S3 AND NOT #CNTSeg_ApHsMx.QU)) AND #Mx_ET50 AND #FTF_MSal AND #Selec_M3M4_Salida AND #Selec_DW THEN
       #EstadoVI.Err_FTF_Sin_LibPHS_S3 := TRUE;
   END_IF;
   IF #EstadoVI.Err_FTF_Sin_LibPHS_S3 THEN #EstadoVI.Error_Mx := TRUE; END_IF;
END_REGION

REGION Network 44: ERROR - Descarga por S4 >>> UP
   RUNG wire#powerrail
      Contact( #EstadoZona.Rearme_CBx )
      S_RS(operand := #EstadoVI.Err_FTF_Sin_LibPHS_S4, s1 := wire#w2)
      S_Coil( #EstadoVI.Error_Mx )
   END_RUNG
   RUNG wire#powerrail
      I_Contact( #ConfigFB.SinErrorLiberarPHS_S4 )
      wire#w1
      Contact( #Mx_ET50 )
      Contact( #FTF_MSal )
      Contact( #Selec_M3M4_Salida )
      Contact( #Selec_UP )
   END_RUNG wire#w2
   RUNG wire#powerrail
      Contact( #ConfigFB.SinErrorLiberarPHS_S4 )
      I_Contact( #CNTSeg_ApHsMx.QU )
   END_RUNG wire#w1
   // the same network as SCL:
   IF #EstadoZona.Rearme_CBx THEN
       #EstadoVI.Err_FTF_Sin_LibPHS_S4 := FALSE;   // RS flip-flop
   END_IF;
   IF (NOT #ConfigFB.SinErrorLiberarPHS_S4 OR (#ConfigFB.SinErrorLiberarPHS_S4 AND NOT #CNTSeg_ApHsMx.QU)) AND #Mx_ET50 AND #FTF_MSal AND #Selec_M3M4_Salida AND #Selec_UP THEN
       #EstadoVI.Err_FTF_Sin_LibPHS_S4 := TRUE;
   END_IF;
   IF #EstadoVI.Err_FTF_Sin_LibPHS_S4 THEN #EstadoVI.Error_Mx := TRUE; END_IF;
END_REGION

REGION Network 45: TMP - ERROR - TimeOut Avance
   RUNG wire#powerrail
      #TOut_Av_Mx(IN := wire#w2, R := wire#w4, PV := #V_TOut_Tx_Mx, BaseUnidades_ms := "CTE_BaseUnidades_1s", QU =>, QD =>, CVU =>, CVD =>)
   END_RUNG
   RUNG wire#powerrail
      Contact( #Mx_ET10 )
      Contact( #MEnt_DescargaAct )
      wire#w1
      Contact( #Selec_M1M2_Entrada )
      I_Contact( #Mx_ET02 )
      Contact( #Avance_Tx )
      I_Contact( #EstadoZona.Manual_CBx )
   END_RUNG wire#w2
   RUNG wire#powerrail
      Contact( #Mx_ET11 )
   END_RUNG wire#w1
   RUNG wire#powerrail
      Contact( #Mx_ET12 )
   END_RUNG wire#w1
   RUNG wire#powerrail
      I_Contact( #Mx_ET10 )
      wire#w3
      I_Contact( #Mx_ET11 )
      I_Contact( #Mx_ET12 )
   END_RUNG wire#w4
   RUNG wire#powerrail
      I_Contact( #MEnt_DescargaAct )
   END_RUNG wire#w3
   RUNG wire#powerrail
      I_Contact( #EstadoVI.Err_TOut_Avance_E1_E3 )
      I_Contact( #EstadoVI.Err_TOut_Avance_E2_E4 )
      Not()
   END_RUNG wire#w4
   // the same network as SCL:
   #TOut_Av_Mx(IN := ((#Mx_ET10 AND #MEnt_DescargaAct) OR #Mx_ET11 OR #Mx_ET12) AND #Selec_M1M2_Entrada AND NOT #Mx_ET02 AND #Avance_Tx AND NOT #EstadoZona.Manual_CBx,   // "FB910_CNT_UHS"
               R := ((NOT #Mx_ET10 OR NOT #MEnt_DescargaAct) AND NOT #Mx_ET11 AND NOT #Mx_ET12) OR NOT (NOT #EstadoVI.Err_TOut_Avance_E1_E3 AND NOT #EstadoVI.Err_TOut_Avance_E2_E4),
               PV := #V_TOut_Tx_Mx,
               BaseUnidades_ms := "CTE_BaseUnidades_1s");
END_REGION

REGION Network 46: ERROR - TimeOut Avance >>> E1E3
   RUNG wire#powerrail
      Contact( #EstadoZona.Rearme_CBx )
      S_RS(operand := #EstadoVI.Err_TOut_Avance_E1_E3, s1 := wire#w1)
      S_Coil( #EstadoVI.Error_Mx )
   END_RUNG
   RUNG wire#powerrail
      Contact( #TOut_Av_Mx.QU )
      Contact( #Selec_DW )
   END_RUNG wire#w1
   // the same network as SCL:
   IF #EstadoZona.Rearme_CBx THEN
       #EstadoVI.Err_TOut_Avance_E1_E3 := FALSE;   // RS flip-flop
   END_IF;
   IF #TOut_Av_Mx.QU AND #Selec_DW THEN #EstadoVI.Err_TOut_Avance_E1_E3 := TRUE; END_IF;
   IF #EstadoVI.Err_TOut_Avance_E1_E3 THEN #EstadoVI.Error_Mx := TRUE; END_IF;
END_REGION

REGION Network 47: ERROR - TimeOut Avance >>> E2E4
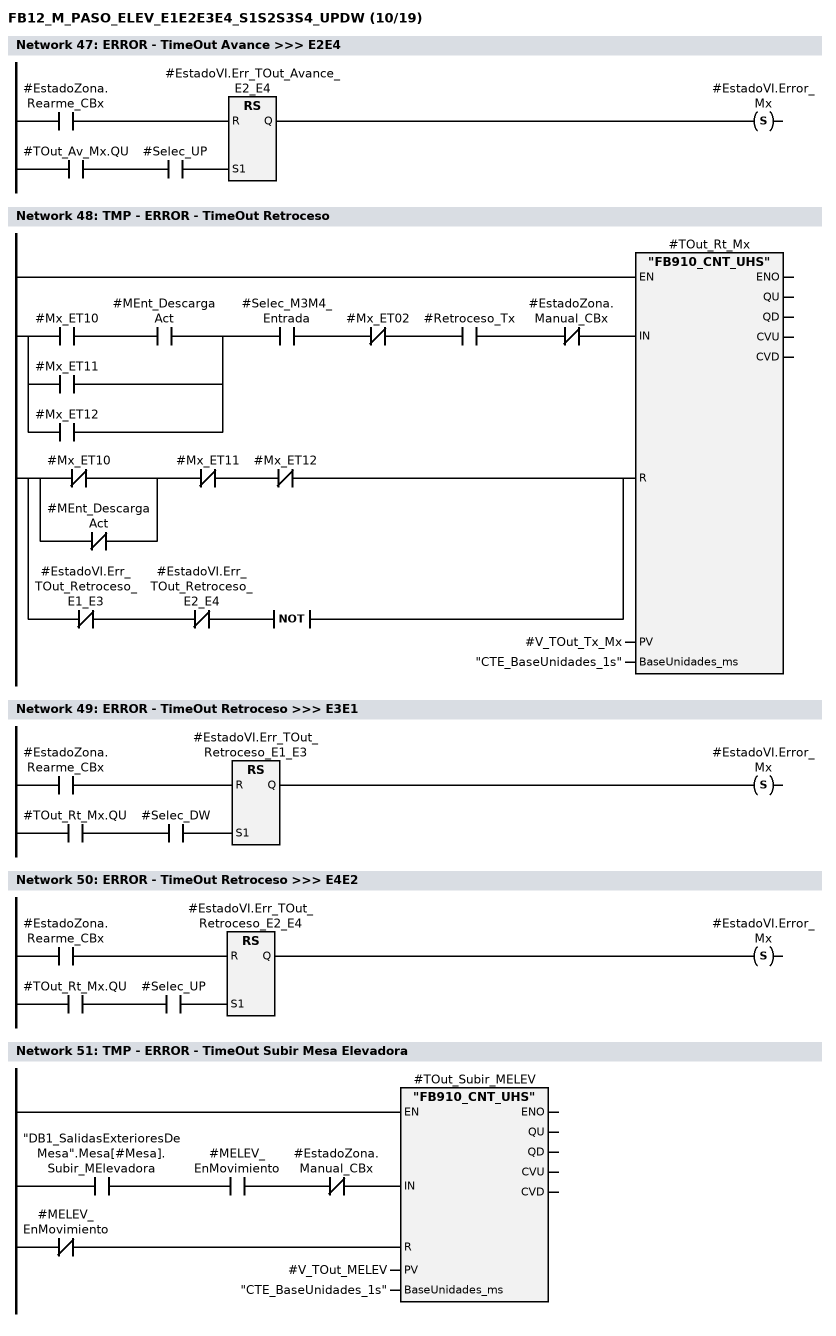
   RUNG wire#powerrail
      Contact( #EstadoZona.Rearme_CBx )
      S_RS(operand := #EstadoVI.Err_TOut_Avance_E2_E4, s1 := wire#w1)
      S_Coil( #EstadoVI.Error_Mx )
   END_RUNG
   RUNG wire#powerrail
      Contact( #TOut_Av_Mx.QU )
      Contact( #Selec_UP )
   END_RUNG wire#w1
   // the same network as SCL:
   IF #EstadoZona.Rearme_CBx THEN
       #EstadoVI.Err_TOut_Avance_E2_E4 := FALSE;   // RS flip-flop
   END_IF;
   IF #TOut_Av_Mx.QU AND #Selec_UP THEN #EstadoVI.Err_TOut_Avance_E2_E4 := TRUE; END_IF;
   IF #EstadoVI.Err_TOut_Avance_E2_E4 THEN #EstadoVI.Error_Mx := TRUE; END_IF;
END_REGION

REGION Network 48: TMP - ERROR - TimeOut Retroceso
   RUNG wire#powerrail
      #TOut_Rt_Mx(IN := wire#w2, R := wire#w4, PV := #V_TOut_Tx_Mx, BaseUnidades_ms := "CTE_BaseUnidades_1s", QU =>, QD =>, CVU =>, CVD =>)
   END_RUNG
   RUNG wire#powerrail
      Contact( #Mx_ET10 )
      Contact( #MEnt_DescargaAct )
      wire#w1
      Contact( #Selec_M3M4_Entrada )
      I_Contact( #Mx_ET02 )
      Contact( #Retroceso_Tx )
      I_Contact( #EstadoZona.Manual_CBx )
   END_RUNG wire#w2
   RUNG wire#powerrail
      Contact( #Mx_ET11 )
   END_RUNG wire#w1
   RUNG wire#powerrail
      Contact( #Mx_ET12 )
   END_RUNG wire#w1
   RUNG wire#powerrail
      I_Contact( #Mx_ET10 )
      wire#w3
      I_Contact( #Mx_ET11 )
      I_Contact( #Mx_ET12 )
   END_RUNG wire#w4
   RUNG wire#powerrail
      I_Contact( #MEnt_DescargaAct )
   END_RUNG wire#w3
   RUNG wire#powerrail
      I_Contact( #EstadoVI.Err_TOut_Retroceso_E1_E3 )
      I_Contact( #EstadoVI.Err_TOut_Retroceso_E2_E4 )
      Not()
   END_RUNG wire#w4
   // the same network as SCL:
   #TOut_Rt_Mx(IN := ((#Mx_ET10 AND #MEnt_DescargaAct) OR #Mx_ET11 OR #Mx_ET12) AND #Selec_M3M4_Entrada AND NOT #Mx_ET02 AND #Retroceso_Tx AND NOT #EstadoZona.Manual_CBx,   // "FB910_CNT_UHS"
               R := ((NOT #Mx_ET10 OR NOT #MEnt_DescargaAct) AND NOT #Mx_ET11 AND NOT #Mx_ET12) OR NOT (NOT #EstadoVI.Err_TOut_Retroceso_E1_E3 AND NOT #EstadoVI.Err_TOut_Retroceso_E2_E4),
               PV := #V_TOut_Tx_Mx,
               BaseUnidades_ms := "CTE_BaseUnidades_1s");
END_REGION

REGION Network 49: ERROR - TimeOut Retroceso >>> E3E1
   RUNG wire#powerrail
      Contact( #EstadoZona.Rearme_CBx )
      S_RS(operand := #EstadoVI.Err_TOut_Retroceso_E1_E3, s1 := wire#w1)
      S_Coil( #EstadoVI.Error_Mx )
   END_RUNG
   RUNG wire#powerrail
      Contact( #TOut_Rt_Mx.QU )
      Contact( #Selec_DW )
   END_RUNG wire#w1
   // the same network as SCL:
   IF #EstadoZona.Rearme_CBx THEN
       #EstadoVI.Err_TOut_Retroceso_E1_E3 := FALSE;   // RS flip-flop
   END_IF;
   IF #TOut_Rt_Mx.QU AND #Selec_DW THEN #EstadoVI.Err_TOut_Retroceso_E1_E3 := TRUE; END_IF;
   IF #EstadoVI.Err_TOut_Retroceso_E1_E3 THEN #EstadoVI.Error_Mx := TRUE; END_IF;
END_REGION

REGION Network 50: ERROR - TimeOut Retroceso >>> E4E2
   RUNG wire#powerrail
      Contact( #EstadoZona.Rearme_CBx )
      S_RS(operand := #EstadoVI.Err_TOut_Retroceso_E2_E4, s1 := wire#w1)
      S_Coil( #EstadoVI.Error_Mx )
   END_RUNG
   RUNG wire#powerrail
      Contact( #TOut_Rt_Mx.QU )
      Contact( #Selec_UP )
   END_RUNG wire#w1
   // the same network as SCL:
   IF #EstadoZona.Rearme_CBx THEN
       #EstadoVI.Err_TOut_Retroceso_E2_E4 := FALSE;   // RS flip-flop
   END_IF;
   IF #TOut_Rt_Mx.QU AND #Selec_UP THEN #EstadoVI.Err_TOut_Retroceso_E2_E4 := TRUE; END_IF;
   IF #EstadoVI.Err_TOut_Retroceso_E2_E4 THEN #EstadoVI.Error_Mx := TRUE; END_IF;
END_REGION

REGION Network 51: TMP - ERROR - TimeOut Subir Mesa Elevadora
   RUNG wire#powerrail
      #TOut_Subir_MELEV(IN := wire#w1, R := wire#w2, PV := #V_TOut_MELEV, BaseUnidades_ms := "CTE_BaseUnidades_1s", QU =>, QD =>, CVU =>, CVD =>)
   END_RUNG
   RUNG wire#powerrail
      Contact( "DB1_SalidasExterioresDeMesa".Mesa[#Mesa].Subir_MElevadora )
      Contact( #MELEV_EnMovimiento )
      I_Contact( #EstadoZona.Manual_CBx )
   END_RUNG wire#w1
   RUNG wire#powerrail
      I_Contact( #MELEV_EnMovimiento )
   END_RUNG wire#w2
   // the same network as SCL:
   #TOut_Subir_MELEV(IN := "DB1_SalidasExterioresDeMesa".Mesa[#Mesa].Subir_MElevadora AND #MELEV_EnMovimiento AND NOT #EstadoZona.Manual_CBx,   // "FB910_CNT_UHS"
                     R := NOT #MELEV_EnMovimiento,
                     PV := #V_TOut_MELEV,
                     BaseUnidades_ms := "CTE_BaseUnidades_1s");
END_REGION

REGION Network 52: ERROR - TimeOut Subir Mesa Elevadora
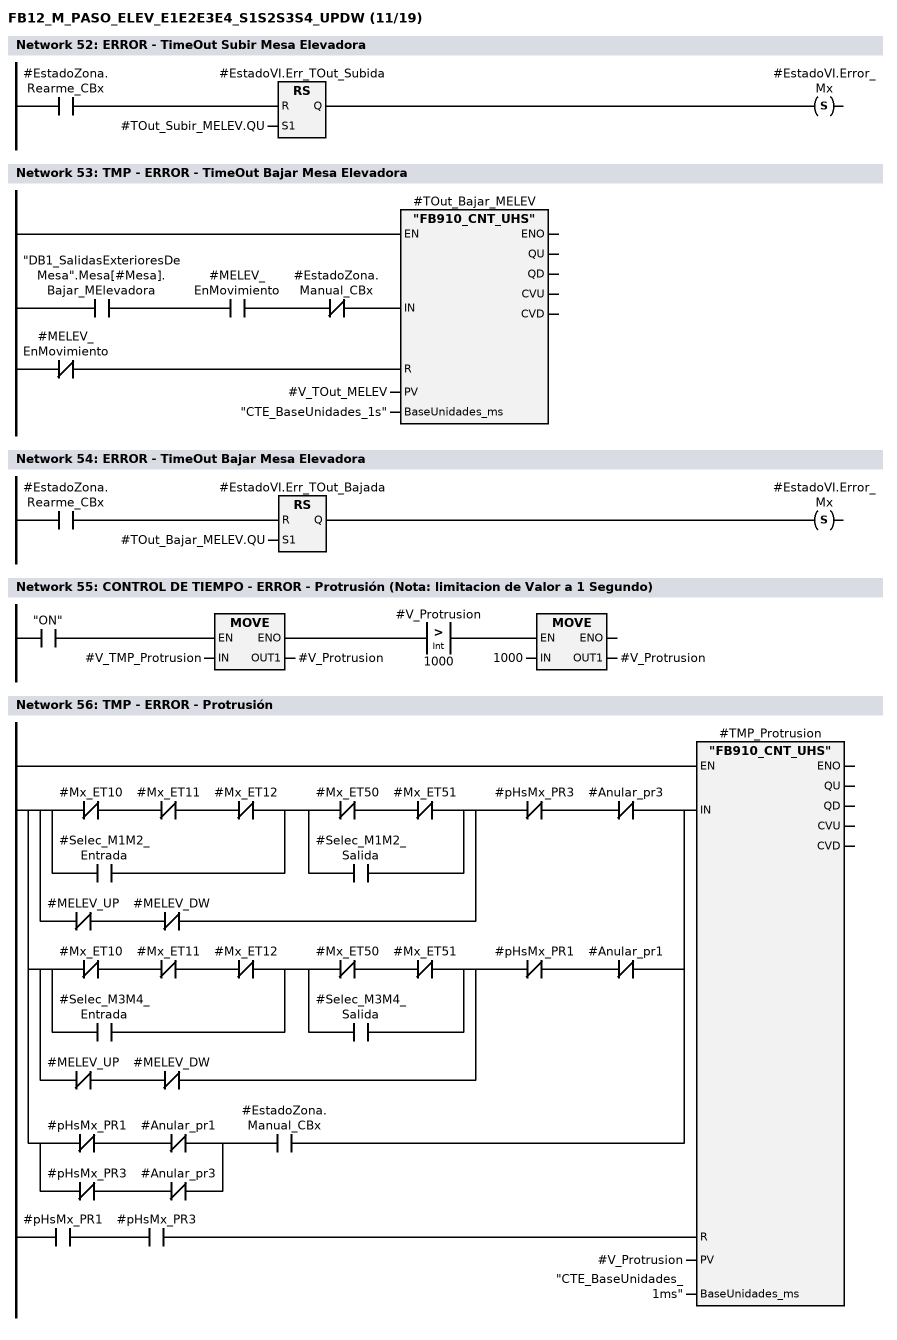
   RUNG wire#powerrail
      Contact( #EstadoZona.Rearme_CBx )
      S_RS(operand := #EstadoVI.Err_TOut_Subida, s1 := #TOut_Subir_MELEV.QU)
      S_Coil( #EstadoVI.Error_Mx )
   END_RUNG
   // the same network as SCL:
   IF #EstadoZona.Rearme_CBx THEN
       #EstadoVI.Err_TOut_Subida := FALSE;   // RS flip-flop
   END_IF;
   IF #TOut_Subir_MELEV.QU THEN #EstadoVI.Err_TOut_Subida := TRUE; END_IF;
   IF #EstadoVI.Err_TOut_Subida THEN #EstadoVI.Error_Mx := TRUE; END_IF;
END_REGION

REGION Network 53: TMP - ERROR - TimeOut Bajar Mesa Elevadora
   RUNG wire#powerrail
      #TOut_Bajar_MELEV(IN := wire#w1, R := wire#w2, PV := #V_TOut_MELEV, BaseUnidades_ms := "CTE_BaseUnidades_1s", QU =>, QD =>, CVU =>, CVD =>)
   END_RUNG
   RUNG wire#powerrail
      Contact( "DB1_SalidasExterioresDeMesa".Mesa[#Mesa].Bajar_MElevadora )
      Contact( #MELEV_EnMovimiento )
      I_Contact( #EstadoZona.Manual_CBx )
   END_RUNG wire#w1
   RUNG wire#powerrail
      I_Contact( #MELEV_EnMovimiento )
   END_RUNG wire#w2
   // the same network as SCL:
   #TOut_Bajar_MELEV(IN := "DB1_SalidasExterioresDeMesa".Mesa[#Mesa].Bajar_MElevadora AND #MELEV_EnMovimiento AND NOT #EstadoZona.Manual_CBx,   // "FB910_CNT_UHS"
                     R := NOT #MELEV_EnMovimiento,
                     PV := #V_TOut_MELEV,
                     BaseUnidades_ms := "CTE_BaseUnidades_1s");
END_REGION

REGION Network 54: ERROR - TimeOut Bajar Mesa Elevadora
   RUNG wire#powerrail
      Contact( #EstadoZona.Rearme_CBx )
      S_RS(operand := #EstadoVI.Err_TOut_Bajada, s1 := #TOut_Bajar_MELEV.QU)
      S_Coil( #EstadoVI.Error_Mx )
   END_RUNG
   // the same network as SCL:
   IF #EstadoZona.Rearme_CBx THEN
       #EstadoVI.Err_TOut_Bajada := FALSE;   // RS flip-flop
   END_IF;
   IF #TOut_Bajar_MELEV.QU THEN #EstadoVI.Err_TOut_Bajada := TRUE; END_IF;
   IF #EstadoVI.Err_TOut_Bajada THEN #EstadoVI.Error_Mx := TRUE; END_IF;
END_REGION

REGION Network 55: CONTROL DE TIEMPO - ERROR - Protrusión (Nota: limitacion de Valor a 1 Segundo)
   RUNG wire#powerrail
      Contact( "ON" )
      Move(in := #V_TMP_Protrusion, out1 => #V_Protrusion)
      { S7_Templates := "SrcType := Int" } GT_Contact(in1 := #V_Protrusion, in2 := 1000)
      Move(in := 1000, out1 => #V_Protrusion)
   END_RUNG
   // the same network as SCL:
   IF "ON" THEN #V_Protrusion := #V_TMP_Protrusion; END_IF;
   IF "ON" AND (#V_Protrusion > 1000) THEN #V_Protrusion := 1000; END_IF;
END_REGION

REGION Network 56: TMP - ERROR - Protrusión
   RUNG wire#powerrail
      #TMP_Protrusion(IN := wire#w6, R := wire#w7, PV := #V_Protrusion, BaseUnidades_ms := "CTE_BaseUnidades_1ms", QU =>, QD =>, CVU =>, CVD =>)
   END_RUNG
   RUNG wire#powerrail
      I_Contact( #Mx_ET10 )
      I_Contact( #Mx_ET11 )
      I_Contact( #Mx_ET12 )
      wire#w1
      I_Contact( #Mx_ET50 )
      I_Contact( #Mx_ET51 )
      wire#w2
      I_Contact( #pHsMx_PR3 )
      I_Contact( #Anular_pr3 )
   END_RUNG wire#w6
   RUNG wire#powerrail
      Contact( #Selec_M1M2_Entrada )
   END_RUNG wire#w1
   RUNG wire#w1
      Contact( #Selec_M1M2_Salida )
   END_RUNG wire#w2
   RUNG wire#powerrail
      I_Contact( #MELEV_UP )
      I_Contact( #MELEV_DW )
   END_RUNG wire#w2
   RUNG wire#powerrail
      I_Contact( #Mx_ET10 )
      I_Contact( #Mx_ET11 )
      I_Contact( #Mx_ET12 )
      wire#w3
      I_Contact( #Mx_ET50 )
      I_Contact( #Mx_ET51 )
      wire#w4
      I_Contact( #pHsMx_PR1 )
      I_Contact( #Anular_pr1 )
   END_RUNG wire#w6
   RUNG wire#powerrail
      Contact( #Selec_M3M4_Entrada )
   END_RUNG wire#w3
   RUNG wire#w3
      Contact( #Selec_M3M4_Salida )
   END_RUNG wire#w4
   RUNG wire#powerrail
      I_Contact( #MELEV_UP )
      I_Contact( #MELEV_DW )
   END_RUNG wire#w4
   RUNG wire#powerrail
      I_Contact( #pHsMx_PR1 )
      I_Contact( #Anular_pr1 )
      wire#w5
      Contact( #EstadoZona.Manual_CBx )
   END_RUNG wire#w6
   RUNG wire#powerrail
      I_Contact( #pHsMx_PR3 )
      I_Contact( #Anular_pr3 )
   END_RUNG wire#w5
   RUNG wire#powerrail
      Contact( #pHsMx_PR1 )
      Contact( #pHsMx_PR3 )
   END_RUNG wire#w7
   // the same network as SCL:
   #TMP_Protrusion(IN := (((((NOT #Mx_ET10 AND NOT #Mx_ET11 AND NOT #Mx_ET12) OR #Selec_M1M2_Entrada) AND ((NOT #Mx_ET50 AND NOT #Mx_ET51) OR #Selec_M1M2_Salida)) OR (NOT #MELEV_UP AND NOT #MELEV_DW)) AND NOT #pHsMx_PR3 AND NOT #Anular_pr3) OR (((((NOT #Mx_ET10 AND NOT #Mx_ET11 AND NOT #Mx_ET12) OR #Selec_M3M4_Entrada) AND ((NOT #Mx_ET50 AND NOT #Mx_ET51) OR #Selec_M3M4_Salida)) OR (NOT #MELEV_UP AND NOT #MELEV_DW)) AND NOT #pHsMx_PR1 AND NOT #Anular_pr1) OR (((NOT #pHsMx_PR1 AND NOT #Anular_pr1) OR (NOT #pHsMx_PR3 AND NOT #Anular_pr3)) AND #EstadoZona.Manual_CBx),   // "FB910_CNT_UHS"
                   R := #pHsMx_PR1 AND #pHsMx_PR3,
                   PV := #V_Protrusion,
                   BaseUnidades_ms := "CTE_BaseUnidades_1ms");
END_REGION

REGION Network 57: ERROR - Protrusión
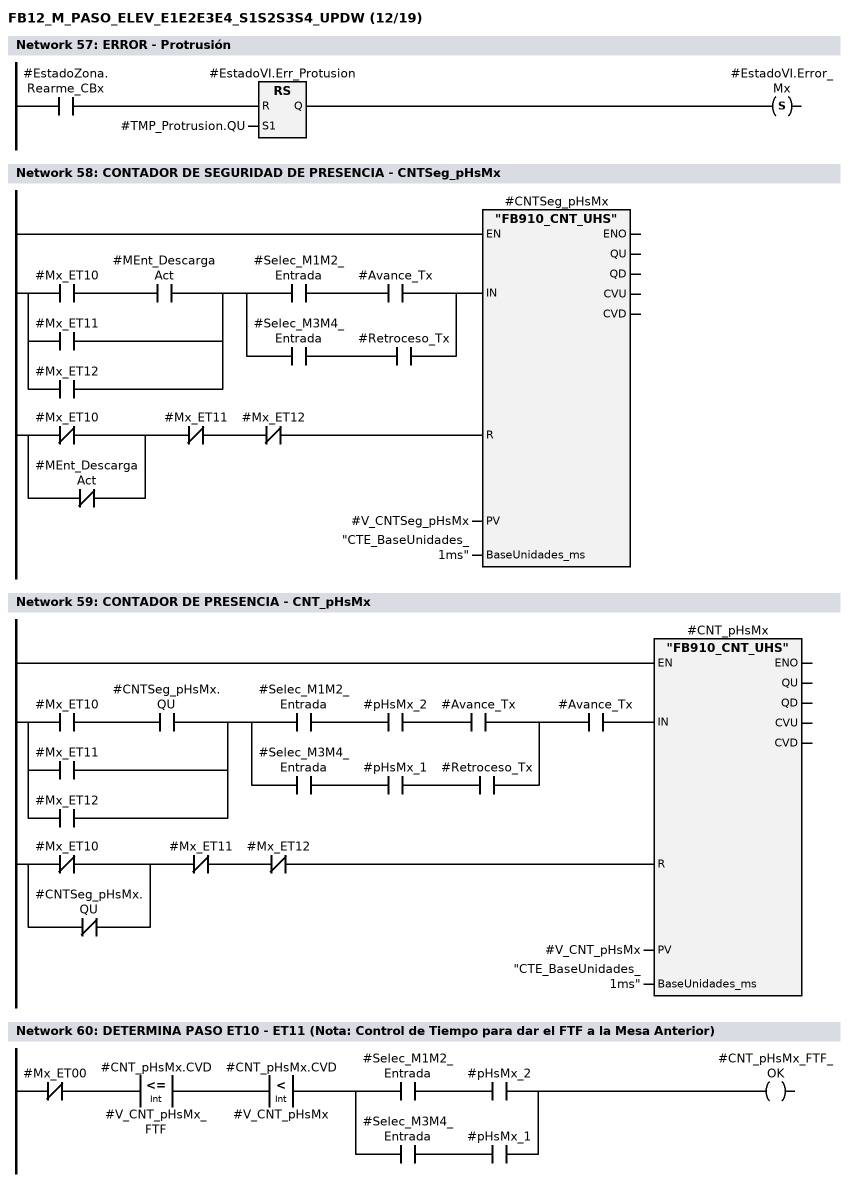
   RUNG wire#powerrail
      Contact( #EstadoZona.Rearme_CBx )
      S_RS(operand := #EstadoVI.Err_Protusion, s1 := #TMP_Protrusion.QU)
      S_Coil( #EstadoVI.Error_Mx )
   END_RUNG
   // the same network as SCL:
   IF #EstadoZona.Rearme_CBx THEN
       #EstadoVI.Err_Protusion := FALSE;   // RS flip-flop
   END_IF;
   IF #TMP_Protrusion.QU THEN #EstadoVI.Err_Protusion := TRUE; END_IF;
   IF #EstadoVI.Err_Protusion THEN #EstadoVI.Error_Mx := TRUE; END_IF;
END_REGION

